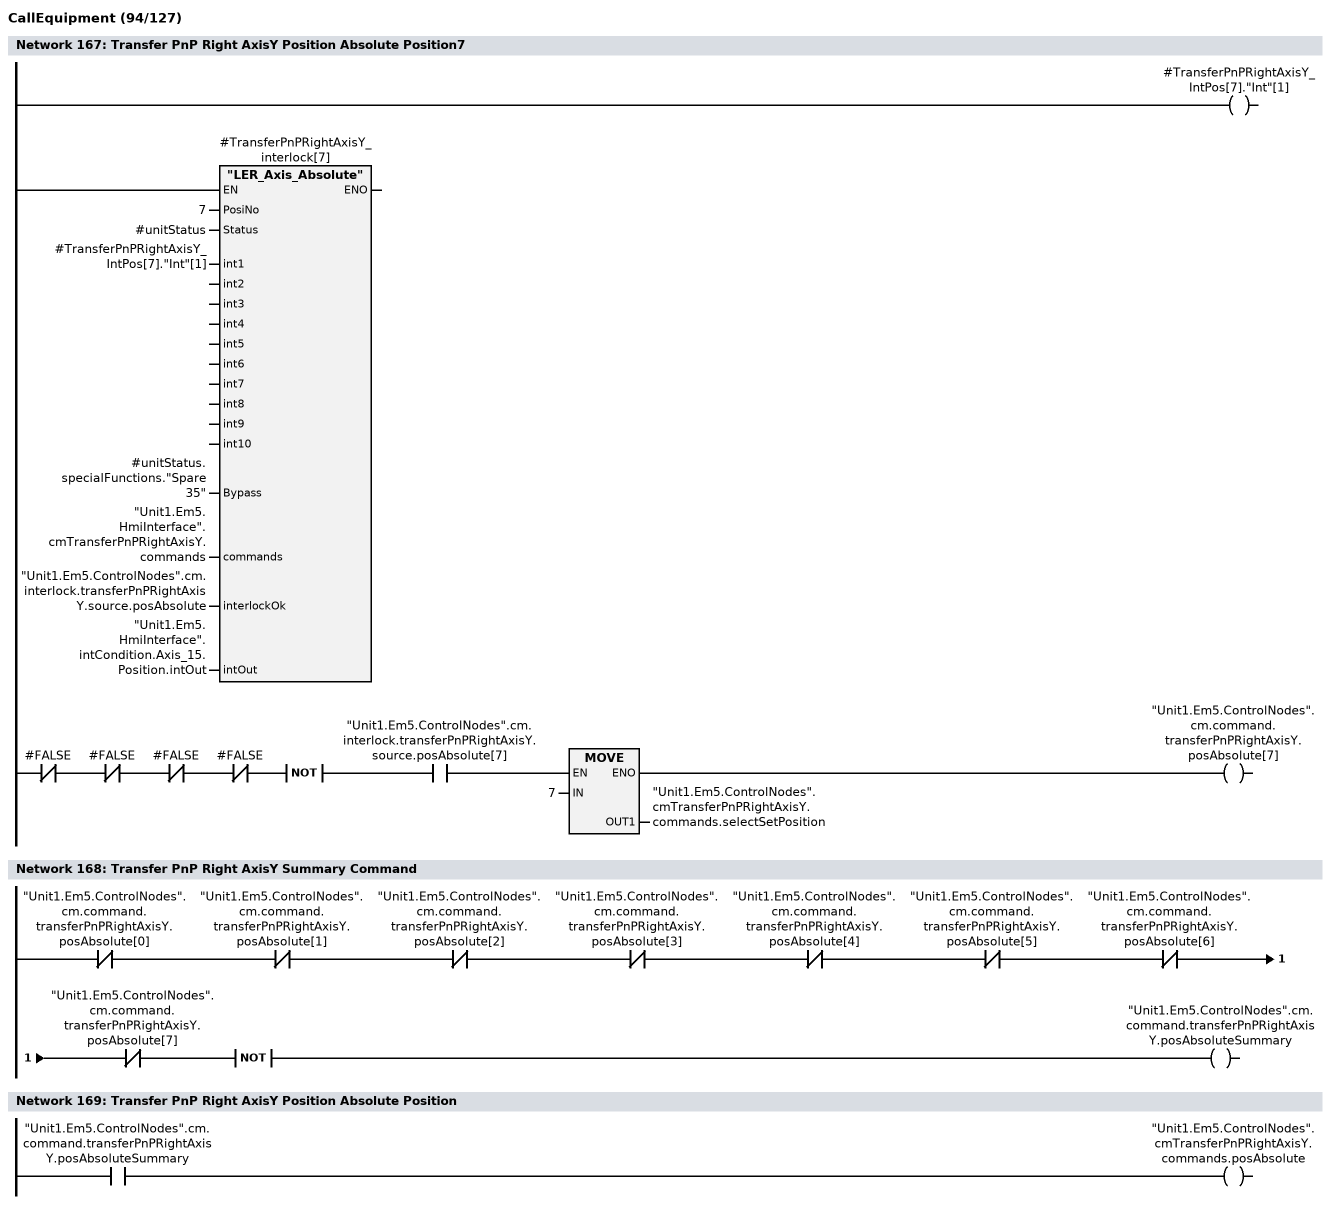
   RUNG wire#powerrail
      Coil( #TransferPnPRightAxisY_IntPos[7]."Int"[1] )
   END_RUNG
   RUNG wire#powerrail
      #TransferPnPRightAxisY_interlock[7](PosiNo := 7, Status := #unitStatus, int1 := #TransferPnPRightAxisY_IntPos[7]."Int"[1], int2 :=, int3 :=, int4 :=, int5 :=, int6 :=, int7 :=, int8 :=, int9 :=, int10 :=, Bypass := #unitStatus.specialFunctions."Spare 35", commands := "Unit1.Em5.HmiInterface".cmTransferPnPRightAxisY.commands, interlockOk := "Unit1.Em5.ControlNodes".cm.interlock.transferPnPRightAxisY.source.posAbsolute, intOut := "Unit1.Em5.HmiInterface".intCondition.Axis_15.Position.intOut)
   END_RUNG
   RUNG wire#powerrail
      I_Contact( #FALSE )
      I_Contact( #FALSE )
      I_Contact( #FALSE )
      I_Contact( #FALSE )
      Not()
      Contact( "Unit1.Em5.ControlNodes".cm.interlock.transferPnPRightAxisY.source.posAbsolute[7] )
      Move(in := 7, out1 => "Unit1.Em5.ControlNodes".cmTransferPnPRightAxisY.commands.selectSetPosition)
      Coil( "Unit1.Em5.ControlNodes".cm.command.transferPnPRightAxisY.posAbsolute[7] )
   END_RUNG
   // the same network as SCL:
   #TransferPnPRightAxisY_IntPos[7]."Int"[1] := TRUE;
   #TransferPnPRightAxisY_interlock[7](PosiNo := 7,   // "LER_Axis_Absolute"
                           Status := #unitStatus,
                           int1 := #TransferPnPRightAxisY_IntPos[7]."Int"[1],
                           Bypass := #unitStatus.specialFunctions."Spare 35",
                           commands := "Unit1.Em5.HmiInterface".cmTransferPnPRightAxisY.commands,
                           interlockOk := "Unit1.Em5.ControlNodes".cm.interlock.transferPnPRightAxisY.source.posAbsolute,
                           intOut := "Unit1.Em5.HmiInterface".intCondition.Axis_15.Position.intOut);
   #_w1 := NOT (NOT #FALSE AND NOT #FALSE AND NOT #FALSE AND NOT #FALSE) AND "Unit1.Em5.ControlNodes".cm.interlock.transferPnPRightAxisY.source.posAbsolute[7];
   IF #_w1 THEN "Unit1.Em5.ControlNodes".cmTransferPnPRightAxisY.commands.selectSetPosition := 7; END_IF;
   "Unit1.Em5.ControlNodes".cm.command.transferPnPRightAxisY.posAbsolute[7] := #_w1;
END_REGION

REGION Network 168: Transfer PnP Right AxisY Summary Command
   RUNG wire#powerrail
      I_Contact( "Unit1.Em5.ControlNodes".cm.command.transferPnPRightAxisY.posAbsolute[0] )
      I_Contact( "Unit1.Em5.ControlNodes".cm.command.transferPnPRightAxisY.posAbsolute[1] )
      I_Contact( "Unit1.Em5.ControlNodes".cm.command.transferPnPRightAxisY.posAbsolute[2] )
      I_Contact( "Unit1.Em5.ControlNodes".cm.command.transferPnPRightAxisY.posAbsolute[3] )
      I_Contact( "Unit1.Em5.ControlNodes".cm.command.transferPnPRightAxisY.posAbsolute[4] )
      I_Contact( "Unit1.Em5.ControlNodes".cm.command.transferPnPRightAxisY.posAbsolute[5] )
      I_Contact( "Unit1.Em5.ControlNodes".cm.command.transferPnPRightAxisY.posAbsolute[6] )
      I_Contact( "Unit1.Em5.ControlNodes".cm.command.transferPnPRightAxisY.posAbsolute[7] )
      Not()
      Coil( "Unit1.Em5.ControlNodes".cm.command.transferPnPRightAxisY.posAbsoluteSummary )
   END_RUNG
   // the same network as SCL:
   "Unit1.Em5.ControlNodes".cm.command.transferPnPRightAxisY.posAbsoluteSummary := NOT (NOT "Unit1.Em5.ControlNodes".cm.command.transferPnPRightAxisY.posAbsolute[0] AND NOT "Unit1.Em5.ControlNodes".cm.command.transferPnPRightAxisY.posAbsolute[1] AND NOT "Unit1.Em5.ControlNodes".cm.command.transferPnPRightAxisY.posAbsolute[2] AND NOT "Unit1.Em5.ControlNodes".cm.command.transferPnPRightAxisY.posAbsolute[3] AND NOT "Unit1.Em5.ControlNodes".cm.command.transferPnPRightAxisY.posAbsolute[4] AND NOT "Unit1.Em5.ControlNodes".cm.command.transferPnPRightAxisY.posAbsolute[5] AND NOT "Unit1.Em5.ControlNodes".cm.command.transferPnPRightAxisY.posAbsolute[6] AND NOT "Unit1.Em5.ControlNodes".cm.command.transferPnPRightAxisY.posAbsolute[7]);
END_REGION

REGION Network 169: Transfer PnP Right AxisY Position Absolute Position
   RUNG wire#powerrail
      Contact( "Unit1.Em5.ControlNodes".cm.command.transferPnPRightAxisY.posAbsoluteSummary )
      Coil( "Unit1.Em5.ControlNodes".cmTransferPnPRightAxisY.commands.posAbsolute )
   END_RUNG
   // the same network as SCL:
   "Unit1.Em5.ControlNodes".cmTransferPnPRightAxisY.commands.posAbsolute := "Unit1.Em5.ControlNodes".cm.command.transferPnPRightAxisY.posAbsoluteSummary;
END_REGION

REGION Network 170: Transfer PnP Right AxisY Interlock Summary
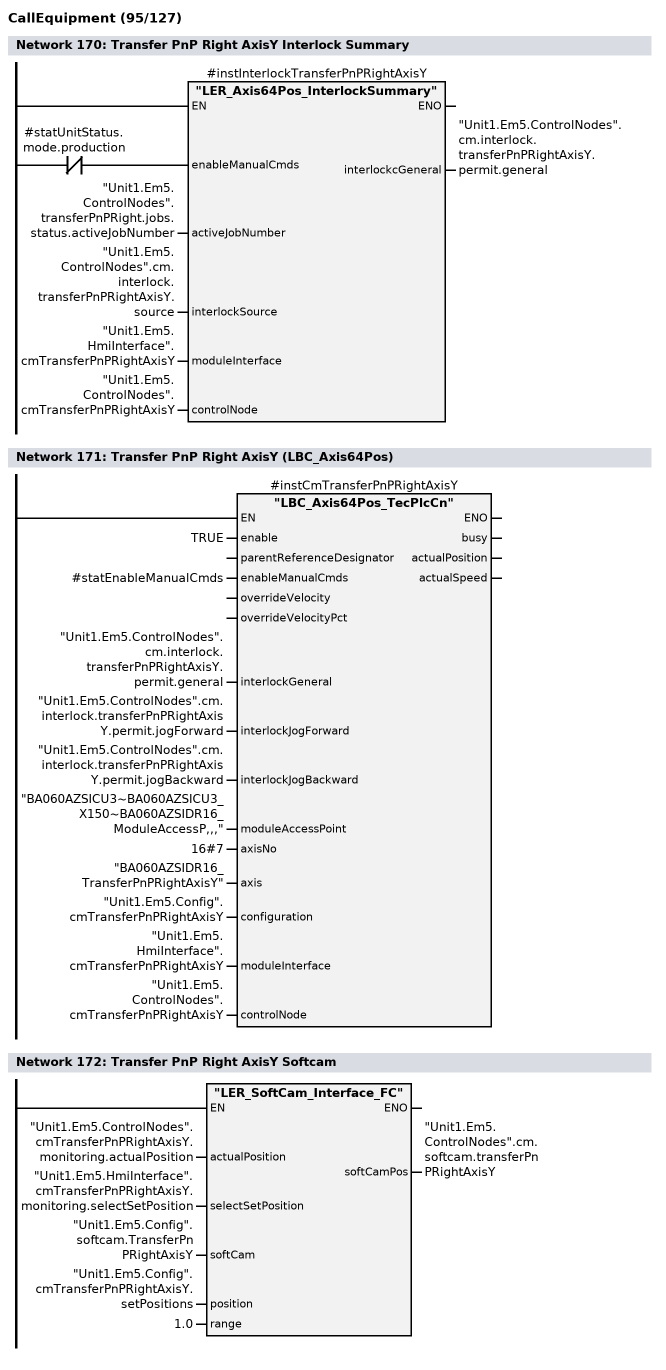
   RUNG wire#powerrail
      #instInterlockTransferPnPRightAxisY(enableManualCmds := wire#w1, activeJobNumber := "Unit1.Em5.ControlNodes".transferPnPRight.jobs.status.activeJobNumber, interlockSource := "Unit1.Em5.ControlNodes".cm.interlock.transferPnPRightAxisY.source, moduleInterface := "Unit1.Em5.HmiInterface".cmTransferPnPRightAxisY, controlNode := "Unit1.Em5.ControlNodes".cmTransferPnPRightAxisY, interlockcGeneral => "Unit1.Em5.ControlNodes".cm.interlock.transferPnPRightAxisY.permit.general)
   END_RUNG
   RUNG wire#powerrail
      I_Contact( #statUnitStatus.mode.production )
   END_RUNG wire#w1
   // the same network as SCL:
   #instInterlockTransferPnPRightAxisY(enableManualCmds := NOT #statUnitStatus.mode.production,   // "LER_Axis64Pos_InterlockSummary"
                           activeJobNumber := "Unit1.Em5.ControlNodes".transferPnPRight.jobs.status.activeJobNumber,
                           interlockSource := "Unit1.Em5.ControlNodes".cm.interlock.transferPnPRightAxisY.source,
                           moduleInterface := "Unit1.Em5.HmiInterface".cmTransferPnPRightAxisY,
                           controlNode := "Unit1.Em5.ControlNodes".cmTransferPnPRightAxisY,
                           interlockcGeneral => "Unit1.Em5.ControlNodes".cm.interlock.transferPnPRightAxisY.permit.general);
END_REGION

REGION Network 171: Transfer PnP Right AxisY (LBC_Axis64Pos)
   RUNG wire#powerrail
      #instCmTransferPnPRightAxisY(enable := TRUE, parentReferenceDesignator :=, enableManualCmds := #statEnableManualCmds, overrideVelocity :=, overrideVelocityPct :=, interlockGeneral := "Unit1.Em5.ControlNodes".cm.interlock.transferPnPRightAxisY.permit.general, interlockJogForward := "Unit1.Em5.ControlNodes".cm.interlock.transferPnPRightAxisY.permit.jogForward, interlockJogBackward := "Unit1.Em5.ControlNodes".cm.interlock.transferPnPRightAxisY.permit.jogBackward, moduleAccessPoint := "BA060AZSICU3~BA060AZSICU3_X150~BA060AZSIDR16_ModuleAccessP,,,", axisNo := 16#7, axis := "BA060AZSIDR16_TransferPnPRightAxisY", configuration := "Unit1.Em5.Config".cmTransferPnPRightAxisY, moduleInterface := "Unit1.Em5.HmiInterface".cmTransferPnPRightAxisY, controlNode := "Unit1.Em5.ControlNodes".cmTransferPnPRightAxisY, busy =>, actualPosition =>, actualSpeed =>)
   END_RUNG
   // the same network as SCL:
   #instCmTransferPnPRightAxisY(enable := TRUE,   // "LBC_Axis64Pos_TecPlcCn"
                           enableManualCmds := #statEnableManualCmds,
                           interlockGeneral := "Unit1.Em5.ControlNodes".cm.interlock.transferPnPRightAxisY.permit.general,
                           interlockJogForward := "Unit1.Em5.ControlNodes".cm.interlock.transferPnPRightAxisY.permit.jogForward,
                           interlockJogBackward := "Unit1.Em5.ControlNodes".cm.interlock.transferPnPRightAxisY.permit.jogBackward,
                           moduleAccessPoint := "BA060AZSICU3~BA060AZSICU3_X150~BA060AZSIDR16_ModuleAccessP,,,",
                           axisNo := 16#7,
                           axis := "BA060AZSIDR16_TransferPnPRightAxisY",
                           configuration := "Unit1.Em5.Config".cmTransferPnPRightAxisY,
                           moduleInterface := "Unit1.Em5.HmiInterface".cmTransferPnPRightAxisY,
                           controlNode := "Unit1.Em5.ControlNodes".cmTransferPnPRightAxisY);
END_REGION

REGION Network 172: Transfer PnP Right AxisY Softcam
   RUNG wire#powerrail
      "LER_SoftCam_Interface_FC"(actualPosition := "Unit1.Em5.ControlNodes".cmTransferPnPRightAxisY.monitoring.actualPosition, selectSetPosition := "Unit1.Em5.HmiInterface".cmTransferPnPRightAxisY.monitoring.selectSetPosition, softCam := "Unit1.Em5.Config".softcam.TransferPnPRightAxisY, position := "Unit1.Em5.Config".cmTransferPnPRightAxisY.setPositions, range := 1.0, softCamPos => "Unit1.Em5.ControlNodes".cm.softcam.transferPnPRightAxisY)
   END_RUNG
   // the same network as SCL:
   "LER_SoftCam_Interface_FC"(actualPosition := "Unit1.Em5.ControlNodes".cmTransferPnPRightAxisY.monitoring.actualPosition,
                           selectSetPosition := "Unit1.Em5.HmiInterface".cmTransferPnPRightAxisY.monitoring.selectSetPosition,
                           softCam := "Unit1.Em5.Config".softcam.TransferPnPRightAxisY,
                           position := "Unit1.Em5.Config".cmTransferPnPRightAxisY.setPositions,
                           range := 1.0,
                           softCamPos => "Unit1.Em5.ControlNodes".cm.softcam.transferPnPRightAxisY);
END_REGION

REGION Network 174: Transfer P&P Right Z-Axis Upload Actual Current And Torque Values
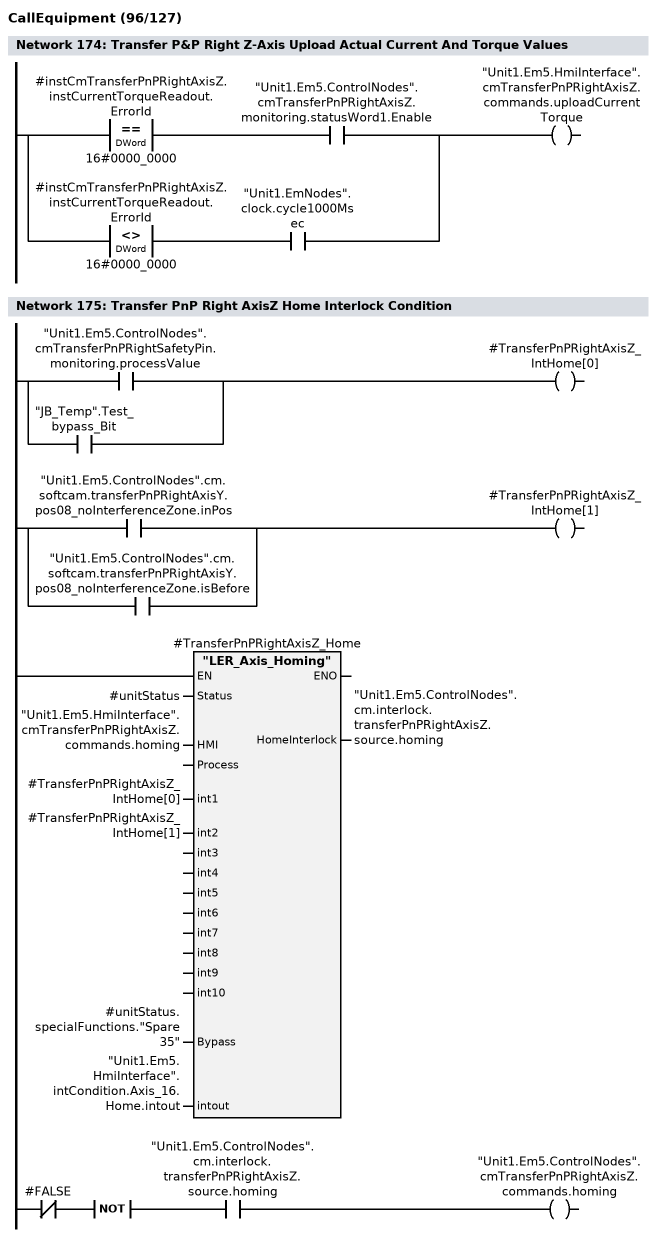
   RUNG wire#powerrail
      { S7_Templates := "SrcType := DWord" } EQ_Contact(in1 := #instCmTransferPnPRightAxisZ.instCurrentTorqueReadout.ErrorId, in2 := 16#0000_0000)
      Contact( "Unit1.Em5.ControlNodes".cmTransferPnPRightAxisZ.monitoring.statusWord1.Enable )
      wire#w1
      Coil( "Unit1.Em5.HmiInterface".cmTransferPnPRightAxisZ.commands.uploadCurrentTorque )
   END_RUNG
   RUNG wire#powerrail
      { S7_Templates := "SrcType := DWord" } NE_Contact(in1 := #instCmTransferPnPRightAxisZ.instCurrentTorqueReadout.ErrorId, in2 := 16#0000_0000)
      Contact( "Unit1.EmNodes".clock.cycle1000Msec )
   END_RUNG wire#w1
   // the same network as SCL:
   "Unit1.Em5.HmiInterface".cmTransferPnPRightAxisZ.commands.uploadCurrentTorque := ((#instCmTransferPnPRightAxisZ.instCurrentTorqueReadout.ErrorId = 16#0000_0000) AND "Unit1.Em5.ControlNodes".cmTransferPnPRightAxisZ.monitoring.statusWord1.Enable) OR ((#instCmTransferPnPRightAxisZ.instCurrentTorqueReadout.ErrorId <> 16#0000_0000) AND "Unit1.EmNodes".clock.cycle1000Msec);
END_REGION

REGION Network 175: Transfer PnP Right AxisZ Home Interlock Condition
   RUNG wire#powerrail
      Contact( "Unit1.Em5.ControlNodes".cmTransferPnPRightSafetyPin.monitoring.processValue )
      wire#w1
      Coil( #TransferPnPRightAxisZ_IntHome[0] )
   END_RUNG
   RUNG wire#powerrail
      Contact( "JB_Temp".Test_bypass_Bit )
   END_RUNG wire#w1
   RUNG wire#powerrail
      Contact( "Unit1.Em5.ControlNodes".cm.softcam.transferPnPRightAxisY.pos08_noInterferenceZone.inPos )
      wire#w2
      Coil( #TransferPnPRightAxisZ_IntHome[1] )
   END_RUNG
   RUNG wire#powerrail
      Contact( "Unit1.Em5.ControlNodes".cm.softcam.transferPnPRightAxisY.pos08_noInterferenceZone.isBefore )
   END_RUNG wire#w2
   RUNG wire#powerrail
      #TransferPnPRightAxisZ_Home(Status := #unitStatus, HMI := "Unit1.Em5.HmiInterface".cmTransferPnPRightAxisZ.commands.homing, Process :=, int1 := #TransferPnPRightAxisZ_IntHome[0], int2 := #TransferPnPRightAxisZ_IntHome[1], int3 :=, int4 :=, int5 :=, int6 :=, int7 :=, int8 :=, int9 :=, int10 :=, Bypass := #unitStatus.specialFunctions."Spare 35", intout := "Unit1.Em5.HmiInterface".intCondition.Axis_16.Home.intout, HomeInterlock => "Unit1.Em5.ControlNodes".cm.interlock.transferPnPRightAxisZ.source.homing)
   END_RUNG
   RUNG wire#powerrail
      I_Contact( #FALSE )
      Not()
      Contact( "Unit1.Em5.ControlNodes".cm.interlock.transferPnPRightAxisZ.source.homing )
      Coil( "Unit1.Em5.ControlNodes".cmTransferPnPRightAxisZ.commands.homing )
   END_RUNG
   // the same network as SCL:
   #TransferPnPRightAxisZ_IntHome[0] := "Unit1.Em5.ControlNodes".cmTransferPnPRightSafetyPin.monitoring.processValue OR "JB_Temp".Test_bypass_Bit;
   #TransferPnPRightAxisZ_IntHome[1] := "Unit1.Em5.ControlNodes".cm.softcam.transferPnPRightAxisY.pos08_noInterferenceZone.inPos OR "Unit1.Em5.ControlNodes".cm.softcam.transferPnPRightAxisY.pos08_noInterferenceZone.isBefore;
   #TransferPnPRightAxisZ_Home(Status := #unitStatus,   // "LER_Axis_Homing"
                           HMI := "Unit1.Em5.HmiInterface".cmTransferPnPRightAxisZ.commands.homing,
                           int1 := #TransferPnPRightAxisZ_IntHome[0],
                           int2 := #TransferPnPRightAxisZ_IntHome[1],
                           Bypass := #unitStatus.specialFunctions."Spare 35",
                           intout := "Unit1.Em5.HmiInterface".intCondition.Axis_16.Home.intout,
                           HomeInterlock => "Unit1.Em5.ControlNodes".cm.interlock.transferPnPRightAxisZ.source.homing);
   "Unit1.Em5.ControlNodes".cmTransferPnPRightAxisZ.commands.homing := NOT (NOT #FALSE) AND "Unit1.Em5.ControlNodes".cm.interlock.transferPnPRightAxisZ.source.homing;
END_REGION

REGION Network 176: Transfer PnP Right AxisZ JOG Interlock Condition
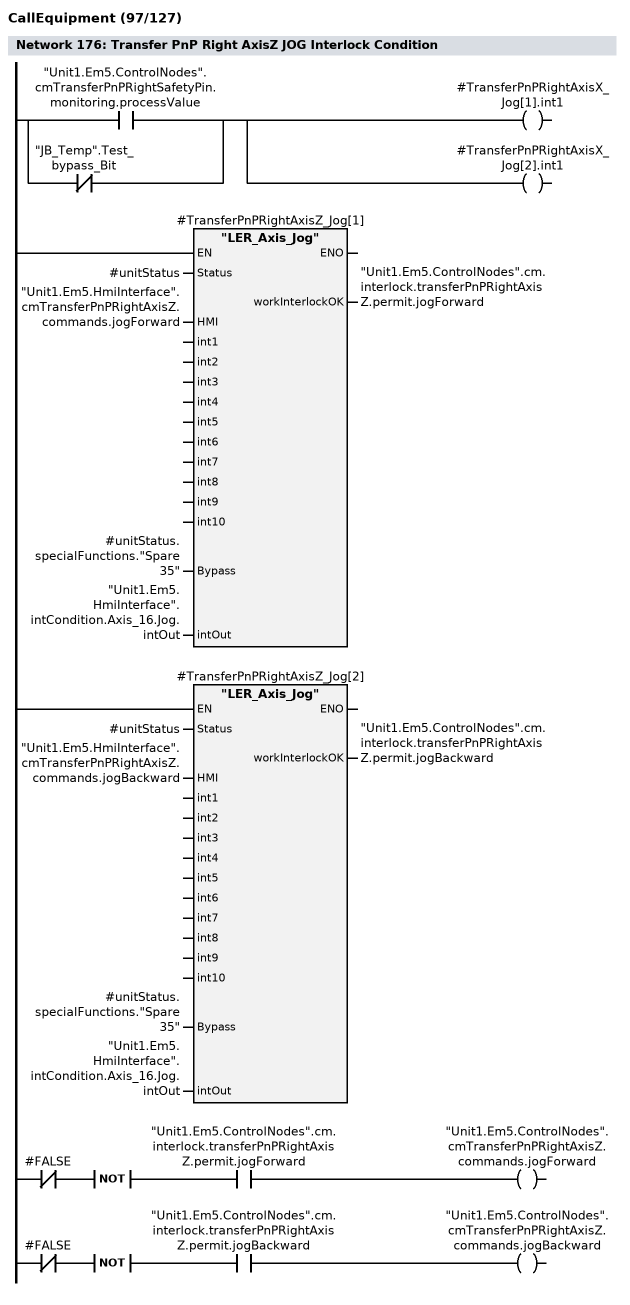
   RUNG wire#powerrail
      Contact( "Unit1.Em5.ControlNodes".cmTransferPnPRightSafetyPin.monitoring.processValue )
      wire#w1
      Coil( #TransferPnPRightAxisX_Jog[1].int1 )
   END_RUNG
   RUNG wire#powerrail
      I_Contact( "JB_Temp".Test_bypass_Bit )
   END_RUNG wire#w1
   RUNG wire#w1
      Coil( #TransferPnPRightAxisX_Jog[2].int1 )
   END_RUNG
   RUNG wire#powerrail
      #TransferPnPRightAxisZ_Jog[1](Status := #unitStatus, HMI := "Unit1.Em5.HmiInterface".cmTransferPnPRightAxisZ.commands.jogForward, int1 :=, int2 :=, int3 :=, int4 :=, int5 :=, int6 :=, int7 :=, int8 :=, int9 :=, int10 :=, Bypass := #unitStatus.specialFunctions."Spare 35", intOut := "Unit1.Em5.HmiInterface".intCondition.Axis_16.Jog.intOut, workInterlockOK => "Unit1.Em5.ControlNodes".cm.interlock.transferPnPRightAxisZ.permit.jogForward)
   END_RUNG
   RUNG wire#powerrail
      #TransferPnPRightAxisZ_Jog[2](Status := #unitStatus, HMI := "Unit1.Em5.HmiInterface".cmTransferPnPRightAxisZ.commands.jogBackward, int1 :=, int2 :=, int3 :=, int4 :=, int5 :=, int6 :=, int7 :=, int8 :=, int9 :=, int10 :=, Bypass := #unitStatus.specialFunctions."Spare 35", intOut := "Unit1.Em5.HmiInterface".intCondition.Axis_16.Jog.intOut, workInterlockOK => "Unit1.Em5.ControlNodes".cm.interlock.transferPnPRightAxisZ.permit.jogBackward)
   END_RUNG
   RUNG wire#powerrail
      I_Contact( #FALSE )
      Not()
      Contact( "Unit1.Em5.ControlNodes".cm.interlock.transferPnPRightAxisZ.permit.jogForward )
      Coil( "Unit1.Em5.ControlNodes".cmTransferPnPRightAxisZ.commands.jogForward )
   END_RUNG
   RUNG wire#powerrail
      I_Contact( #FALSE )
      Not()
      Contact( "Unit1.Em5.ControlNodes".cm.interlock.transferPnPRightAxisZ.permit.jogBackward )
      Coil( "Unit1.Em5.ControlNodes".cmTransferPnPRightAxisZ.commands.jogBackward )
   END_RUNG
   // the same network as SCL:
   #TransferPnPRightAxisX_Jog[1].int1 := "Unit1.Em5.ControlNodes".cmTransferPnPRightSafetyPin.monitoring.processValue OR NOT "JB_Temp".Test_bypass_Bit;
   #TransferPnPRightAxisX_Jog[2].int1 := "Unit1.Em5.ControlNodes".cmTransferPnPRightSafetyPin.monitoring.processValue OR NOT "JB_Temp".Test_bypass_Bit;
   #TransferPnPRightAxisZ_Jog[1](Status := #unitStatus,   // "LER_Axis_Jog"
                           HMI := "Unit1.Em5.HmiInterface".cmTransferPnPRightAxisZ.commands.jogForward,
                           Bypass := #unitStatus.specialFunctions."Spare 35",
                           intOut := "Unit1.Em5.HmiInterface".intCondition.Axis_16.Jog.intOut,
                           workInterlockOK => "Unit1.Em5.ControlNodes".cm.interlock.transferPnPRightAxisZ.permit.jogForward);
   #TransferPnPRightAxisZ_Jog[2](Status := #unitStatus,   // "LER_Axis_Jog"
                           HMI := "Unit1.Em5.HmiInterface".cmTransferPnPRightAxisZ.commands.jogBackward,
                           Bypass := #unitStatus.specialFunctions."Spare 35",
                           intOut := "Unit1.Em5.HmiInterface".intCondition.Axis_16.Jog.intOut,
                           workInterlockOK => "Unit1.Em5.ControlNodes".cm.interlock.transferPnPRightAxisZ.permit.jogBackward);
   "Unit1.Em5.ControlNodes".cmTransferPnPRightAxisZ.commands.jogForward := NOT (NOT #FALSE) AND "Unit1.Em5.ControlNodes".cm.interlock.transferPnPRightAxisZ.permit.jogForward;
   "Unit1.Em5.ControlNodes".cmTransferPnPRightAxisZ.commands.jogBackward := NOT (NOT #FALSE) AND "Unit1.Em5.ControlNodes".cm.interlock.transferPnPRightAxisZ.permit.jogBackward;
END_REGION

REGION Network 177: Transfer PnP Right AxisZ Position Absolute Position0
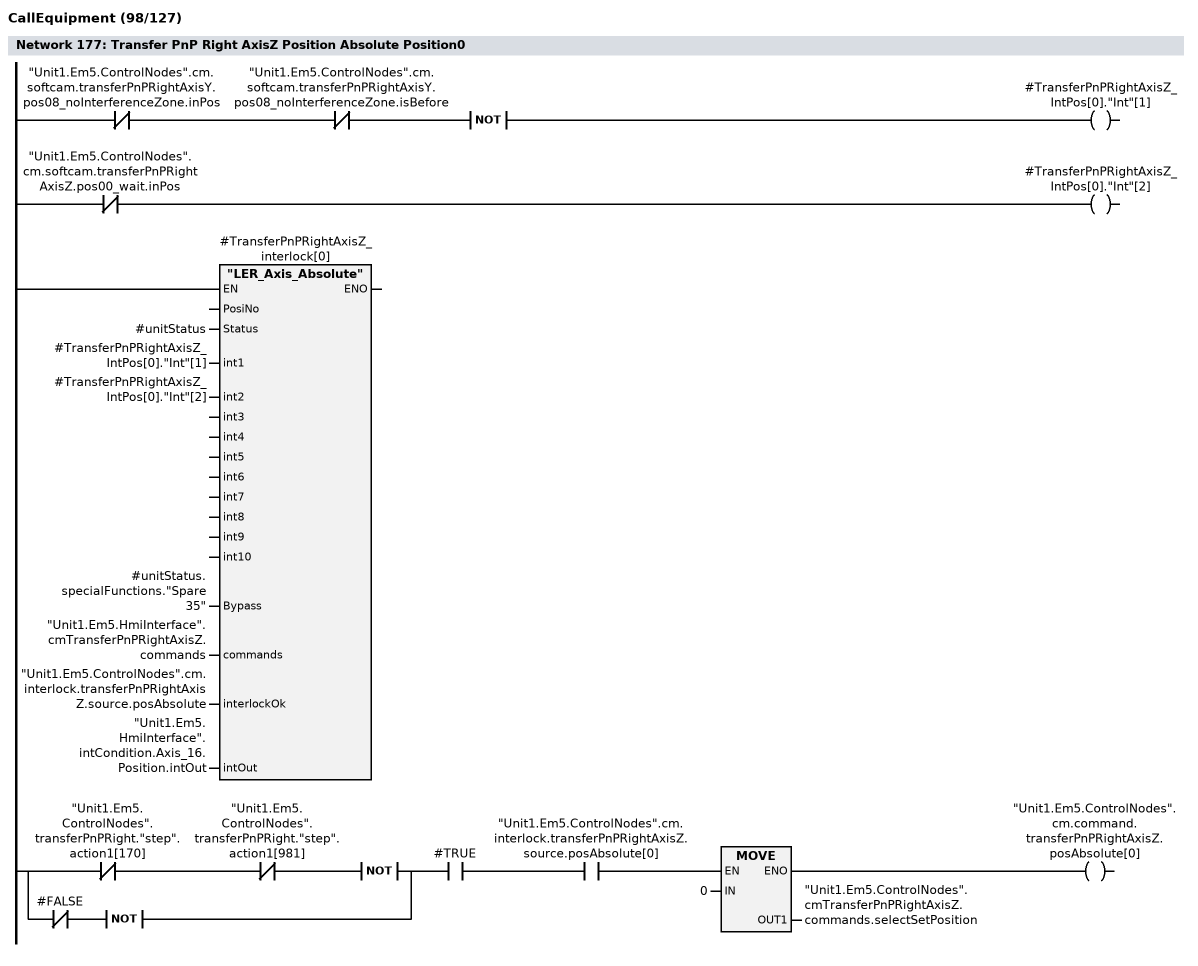
   RUNG wire#powerrail
      I_Contact( "Unit1.Em5.ControlNodes".cm.softcam.transferPnPRightAxisY.pos08_noInterferenceZone.inPos )
      I_Contact( "Unit1.Em5.ControlNodes".cm.softcam.transferPnPRightAxisY.pos08_noInterferenceZone.isBefore )
      Not()
      Coil( #TransferPnPRightAxisZ_IntPos[0]."Int"[1] )
   END_RUNG
   RUNG wire#powerrail
      I_Contact( "Unit1.Em5.ControlNodes".cm.softcam.transferPnPRightAxisZ.pos00_wait.inPos )
      Coil( #TransferPnPRightAxisZ_IntPos[0]."Int"[2] )
   END_RUNG
   RUNG wire#powerrail
      #TransferPnPRightAxisZ_interlock[0](PosiNo :=, Status := #unitStatus, int1 := #TransferPnPRightAxisZ_IntPos[0]."Int"[1], int2 := #TransferPnPRightAxisZ_IntPos[0]."Int"[2], int3 :=, int4 :=, int5 :=, int6 :=, int7 :=, int8 :=, int9 :=, int10 :=, Bypass := #unitStatus.specialFunctions."Spare 35", commands := "Unit1.Em5.HmiInterface".cmTransferPnPRightAxisZ.commands, interlockOk := "Unit1.Em5.ControlNodes".cm.interlock.transferPnPRightAxisZ.source.posAbsolute, intOut := "Unit1.Em5.HmiInterface".intCondition.Axis_16.Position.intOut)
   END_RUNG
   RUNG wire#powerrail
      I_Contact( "Unit1.Em5.ControlNodes".transferPnPRight."step".action1[170] )
      I_Contact( "Unit1.Em5.ControlNodes".transferPnPRight."step".action1[981] )
      Not()
      wire#w1
      Contact( #TRUE )
      Contact( "Unit1.Em5.ControlNodes".cm.interlock.transferPnPRightAxisZ.source.posAbsolute[0] )
      Move(in := 0, out1 => "Unit1.Em5.ControlNodes".cmTransferPnPRightAxisZ.commands.selectSetPosition)
      Coil( "Unit1.Em5.ControlNodes".cm.command.transferPnPRightAxisZ.posAbsolute[0] )
   END_RUNG
   RUNG wire#powerrail
      I_Contact( #FALSE )
      Not()
   END_RUNG wire#w1
   // the same network as SCL:
   #TransferPnPRightAxisZ_IntPos[0]."Int"[1] := NOT (NOT "Unit1.Em5.ControlNodes".cm.softcam.transferPnPRightAxisY.pos08_noInterferenceZone.inPos AND NOT "Unit1.Em5.ControlNodes".cm.softcam.transferPnPRightAxisY.pos08_noInterferenceZone.isBefore);
   #TransferPnPRightAxisZ_IntPos[0]."Int"[2] := NOT "Unit1.Em5.ControlNodes".cm.softcam.transferPnPRightAxisZ.pos00_wait.inPos;
   #TransferPnPRightAxisZ_interlock[0](Status := #unitStatus,   // "LER_Axis_Absolute"
                           int1 := #TransferPnPRightAxisZ_IntPos[0]."Int"[1],
                           int2 := #TransferPnPRightAxisZ_IntPos[0]."Int"[2],
                           Bypass := #unitStatus.specialFunctions."Spare 35",
                           commands := "Unit1.Em5.HmiInterface".cmTransferPnPRightAxisZ.commands,
                           interlockOk := "Unit1.Em5.ControlNodes".cm.interlock.transferPnPRightAxisZ.source.posAbsolute,
                           intOut := "Unit1.Em5.HmiInterface".intCondition.Axis_16.Position.intOut);
   #_w1 := (NOT (NOT "Unit1.Em5.ControlNodes".transferPnPRight."step".action1[170] AND NOT "Unit1.Em5.ControlNodes".transferPnPRight."step".action1[981]) OR NOT (NOT #FALSE)) AND #TRUE AND "Unit1.Em5.ControlNodes".cm.interlock.transferPnPRightAxisZ.source.posAbsolute[0];
   IF #_w1 THEN "Unit1.Em5.ControlNodes".cmTransferPnPRightAxisZ.commands.selectSetPosition := 0; END_IF;
   "Unit1.Em5.ControlNodes".cm.command.transferPnPRightAxisZ.posAbsolute[0] := #_w1;
END_REGION

REGION Network 178: Transfer PnP Right AxisZ Position Absolute Position1
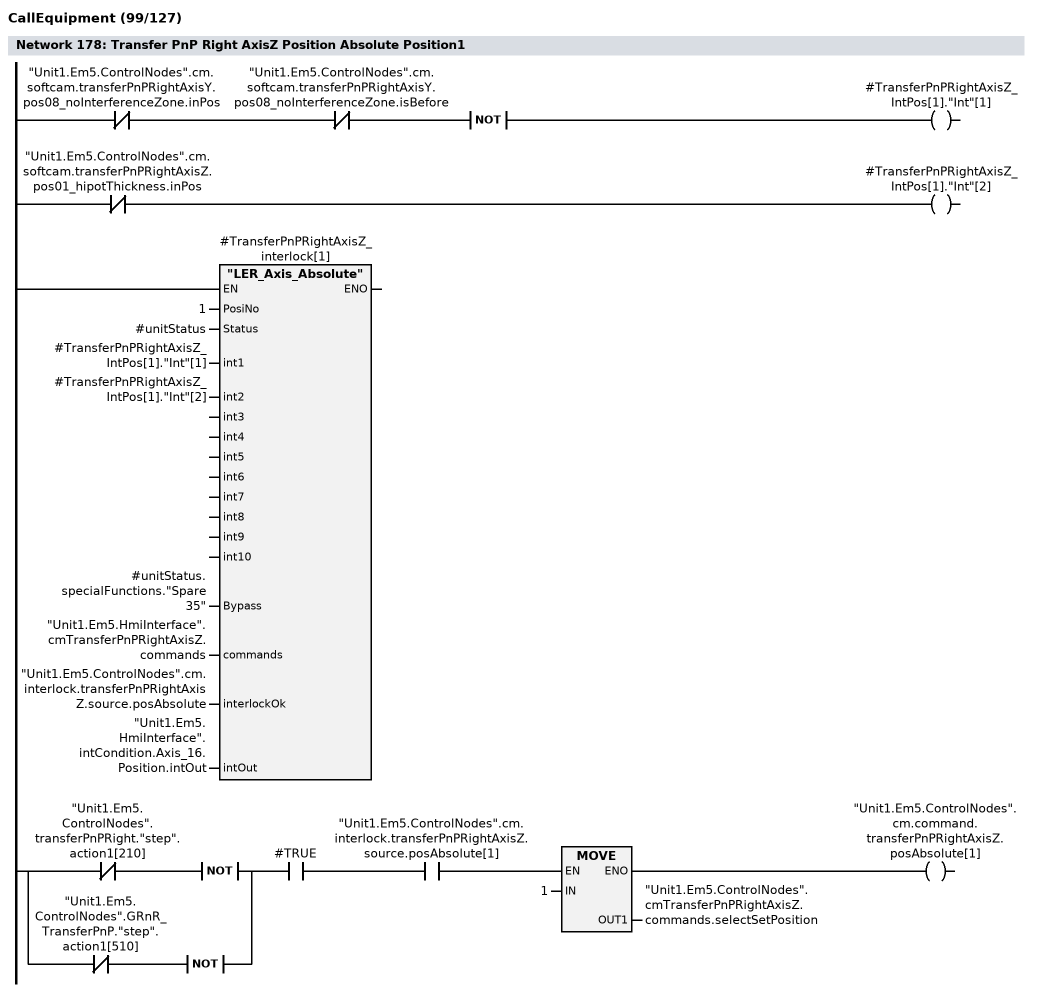
   RUNG wire#powerrail
      I_Contact( "Unit1.Em5.ControlNodes".cm.softcam.transferPnPRightAxisY.pos08_noInterferenceZone.inPos )
      I_Contact( "Unit1.Em5.ControlNodes".cm.softcam.transferPnPRightAxisY.pos08_noInterferenceZone.isBefore )
      Not()
      Coil( #TransferPnPRightAxisZ_IntPos[1]."Int"[1] )
   END_RUNG
   RUNG wire#powerrail
      I_Contact( "Unit1.Em5.ControlNodes".cm.softcam.transferPnPRightAxisZ.pos01_hipotThickness.inPos )
      Coil( #TransferPnPRightAxisZ_IntPos[1]."Int"[2] )
   END_RUNG
   RUNG wire#powerrail
      #TransferPnPRightAxisZ_interlock[1](PosiNo := 1, Status := #unitStatus, int1 := #TransferPnPRightAxisZ_IntPos[1]."Int"[1], int2 := #TransferPnPRightAxisZ_IntPos[1]."Int"[2], int3 :=, int4 :=, int5 :=, int6 :=, int7 :=, int8 :=, int9 :=, int10 :=, Bypass := #unitStatus.specialFunctions."Spare 35", commands := "Unit1.Em5.HmiInterface".cmTransferPnPRightAxisZ.commands, interlockOk := "Unit1.Em5.ControlNodes".cm.interlock.transferPnPRightAxisZ.source.posAbsolute, intOut := "Unit1.Em5.HmiInterface".intCondition.Axis_16.Position.intOut)
   END_RUNG
   RUNG wire#powerrail
      I_Contact( "Unit1.Em5.ControlNodes".transferPnPRight."step".action1[210] )
      Not()
      wire#w1
      Contact( #TRUE )
      Contact( "Unit1.Em5.ControlNodes".cm.interlock.transferPnPRightAxisZ.source.posAbsolute[1] )
      Move(in := 1, out1 => "Unit1.Em5.ControlNodes".cmTransferPnPRightAxisZ.commands.selectSetPosition)
      Coil( "Unit1.Em5.ControlNodes".cm.command.transferPnPRightAxisZ.posAbsolute[1] )
   END_RUNG
   RUNG wire#powerrail
      I_Contact( "Unit1.Em5.ControlNodes".GRnR_TransferPnP."step".action1[510] )
      Not()
   END_RUNG wire#w1
   // the same network as SCL:
   #TransferPnPRightAxisZ_IntPos[1]."Int"[1] := NOT (NOT "Unit1.Em5.ControlNodes".cm.softcam.transferPnPRightAxisY.pos08_noInterferenceZone.inPos AND NOT "Unit1.Em5.ControlNodes".cm.softcam.transferPnPRightAxisY.pos08_noInterferenceZone.isBefore);
   #TransferPnPRightAxisZ_IntPos[1]."Int"[2] := NOT "Unit1.Em5.ControlNodes".cm.softcam.transferPnPRightAxisZ.pos01_hipotThickness.inPos;
   #TransferPnPRightAxisZ_interlock[1](PosiNo := 1,   // "LER_Axis_Absolute"
                           Status := #unitStatus,
                           int1 := #TransferPnPRightAxisZ_IntPos[1]."Int"[1],
                           int2 := #TransferPnPRightAxisZ_IntPos[1]."Int"[2],
                           Bypass := #unitStatus.specialFunctions."Spare 35",
                           commands := "Unit1.Em5.HmiInterface".cmTransferPnPRightAxisZ.commands,
                           interlockOk := "Unit1.Em5.ControlNodes".cm.interlock.transferPnPRightAxisZ.source.posAbsolute,
                           intOut := "Unit1.Em5.HmiInterface".intCondition.Axis_16.Position.intOut);
   #_w1 := (NOT (NOT "Unit1.Em5.ControlNodes".transferPnPRight."step".action1[210]) OR NOT (NOT "Unit1.Em5.ControlNodes".GRnR_TransferPnP."step".action1[510])) AND #TRUE AND "Unit1.Em5.ControlNodes".cm.interlock.transferPnPRightAxisZ.source.posAbsolute[1];
   IF #_w1 THEN "Unit1.Em5.ControlNodes".cmTransferPnPRightAxisZ.commands.selectSetPosition := 1; END_IF;
   "Unit1.Em5.ControlNodes".cm.command.transferPnPRightAxisZ.posAbsolute[1] := #_w1;
END_REGION

REGION Network 179: Transfer PnP Right AxisZ Position Absolute Position2
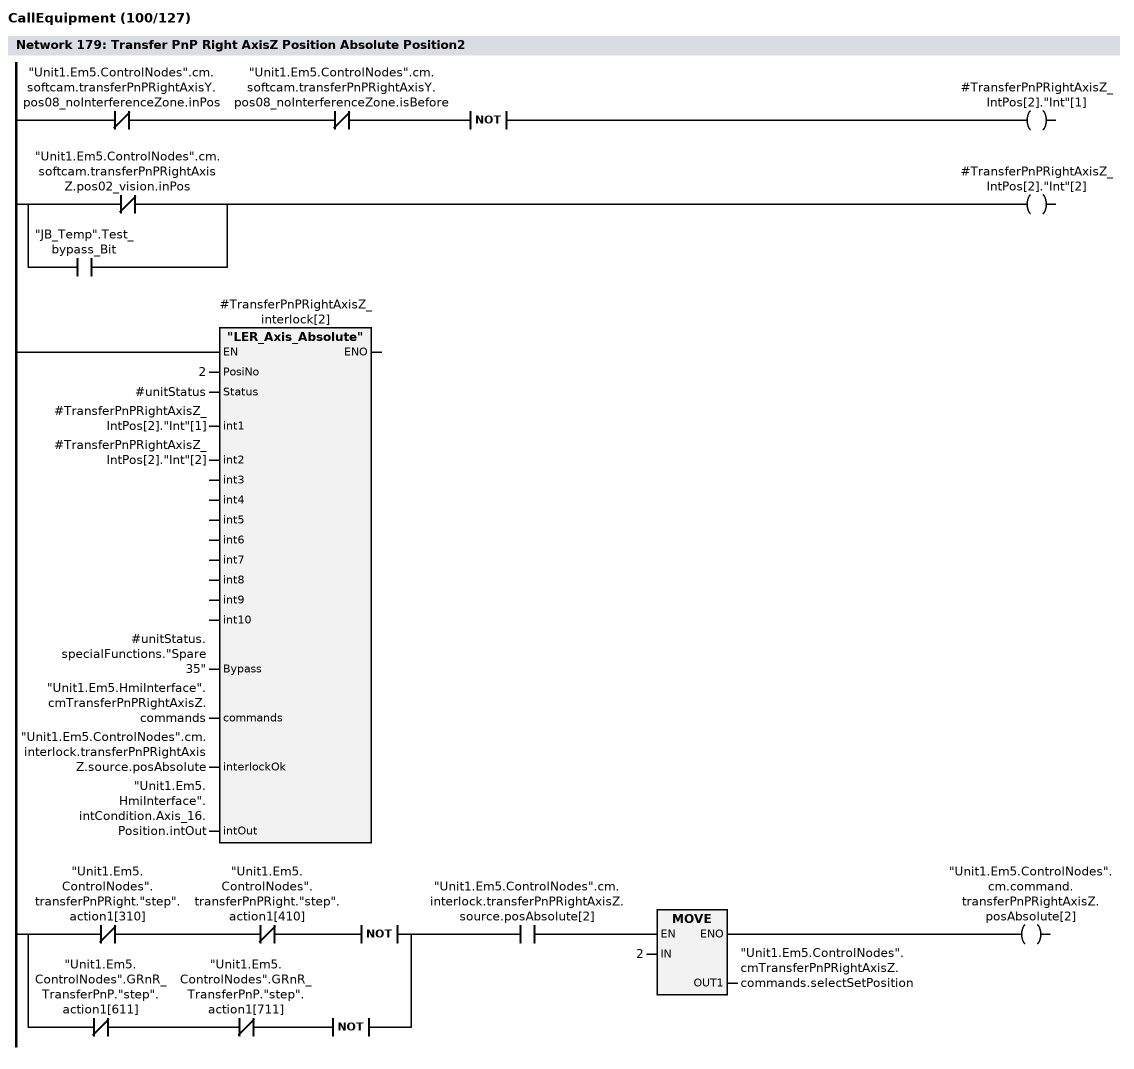
   RUNG wire#powerrail
      I_Contact( "Unit1.Em5.ControlNodes".cm.softcam.transferPnPRightAxisY.pos08_noInterferenceZone.inPos )
      I_Contact( "Unit1.Em5.ControlNodes".cm.softcam.transferPnPRightAxisY.pos08_noInterferenceZone.isBefore )
      Not()
      Coil( #TransferPnPRightAxisZ_IntPos[2]."Int"[1] )
   END_RUNG
   RUNG wire#powerrail
      I_Contact( "Unit1.Em5.ControlNodes".cm.softcam.transferPnPRightAxisZ.pos02_vision.inPos )
      wire#w1
      Coil( #TransferPnPRightAxisZ_IntPos[2]."Int"[2] )
   END_RUNG
   RUNG wire#powerrail
      Contact( "JB_Temp".Test_bypass_Bit )
   END_RUNG wire#w1
   RUNG wire#powerrail
      #TransferPnPRightAxisZ_interlock[2](PosiNo := 2, Status := #unitStatus, int1 := #TransferPnPRightAxisZ_IntPos[2]."Int"[1], int2 := #TransferPnPRightAxisZ_IntPos[2]."Int"[2], int3 :=, int4 :=, int5 :=, int6 :=, int7 :=, int8 :=, int9 :=, int10 :=, Bypass := #unitStatus.specialFunctions."Spare 35", commands := "Unit1.Em5.HmiInterface".cmTransferPnPRightAxisZ.commands, interlockOk := "Unit1.Em5.ControlNodes".cm.interlock.transferPnPRightAxisZ.source.posAbsolute, intOut := "Unit1.Em5.HmiInterface".intCondition.Axis_16.Position.intOut)
   END_RUNG
   RUNG wire#powerrail
      I_Contact( "Unit1.Em5.ControlNodes".transferPnPRight."step".action1[310] )
      I_Contact( "Unit1.Em5.ControlNodes".transferPnPRight."step".action1[410] )
      Not()
      wire#w2
      Contact( "Unit1.Em5.ControlNodes".cm.interlock.transferPnPRightAxisZ.source.posAbsolute[2] )
      Move(in := 2, out1 => "Unit1.Em5.ControlNodes".cmTransferPnPRightAxisZ.commands.selectSetPosition)
      Coil( "Unit1.Em5.ControlNodes".cm.command.transferPnPRightAxisZ.posAbsolute[2] )
   END_RUNG
   RUNG wire#powerrail
      I_Contact( "Unit1.Em5.ControlNodes".GRnR_TransferPnP."step".action1[611] )
      I_Contact( "Unit1.Em5.ControlNodes".GRnR_TransferPnP."step".action1[711] )
      Not()
   END_RUNG wire#w2
   // the same network as SCL:
   #TransferPnPRightAxisZ_IntPos[2]."Int"[1] := NOT (NOT "Unit1.Em5.ControlNodes".cm.softcam.transferPnPRightAxisY.pos08_noInterferenceZone.inPos AND NOT "Unit1.Em5.ControlNodes".cm.softcam.transferPnPRightAxisY.pos08_noInterferenceZone.isBefore);
   #TransferPnPRightAxisZ_IntPos[2]."Int"[2] := NOT "Unit1.Em5.ControlNodes".cm.softcam.transferPnPRightAxisZ.pos02_vision.inPos OR "JB_Temp".Test_bypass_Bit;
   #TransferPnPRightAxisZ_interlock[2](PosiNo := 2,   // "LER_Axis_Absolute"
                           Status := #unitStatus,
                           int1 := #TransferPnPRightAxisZ_IntPos[2]."Int"[1],
                           int2 := #TransferPnPRightAxisZ_IntPos[2]."Int"[2],
                           Bypass := #unitStatus.specialFunctions."Spare 35",
                           commands := "Unit1.Em5.HmiInterface".cmTransferPnPRightAxisZ.commands,
                           interlockOk := "Unit1.Em5.ControlNodes".cm.interlock.transferPnPRightAxisZ.source.posAbsolute,
                           intOut := "Unit1.Em5.HmiInterface".intCondition.Axis_16.Position.intOut);
   #_w1 := (NOT (NOT "Unit1.Em5.ControlNodes".transferPnPRight."step".action1[310] AND NOT "Unit1.Em5.ControlNodes".transferPnPRight."step".action1[410]) OR NOT (NOT "Unit1.Em5.ControlNodes".GRnR_TransferPnP."step".action1[611] AND NOT "Unit1.Em5.ControlNodes".GRnR_TransferPnP."step".action1[711])) AND "Unit1.Em5.ControlNodes".cm.interlock.transferPnPRightAxisZ.source.posAbsolute[2];
   IF #_w1 THEN "Unit1.Em5.ControlNodes".cmTransferPnPRightAxisZ.commands.selectSetPosition := 2; END_IF;
   "Unit1.Em5.ControlNodes".cm.command.transferPnPRightAxisZ.posAbsolute[2] := #_w1;
END_REGION

REGION Network 180: Transfer PnP Right AxisZ Position Absolute Position3
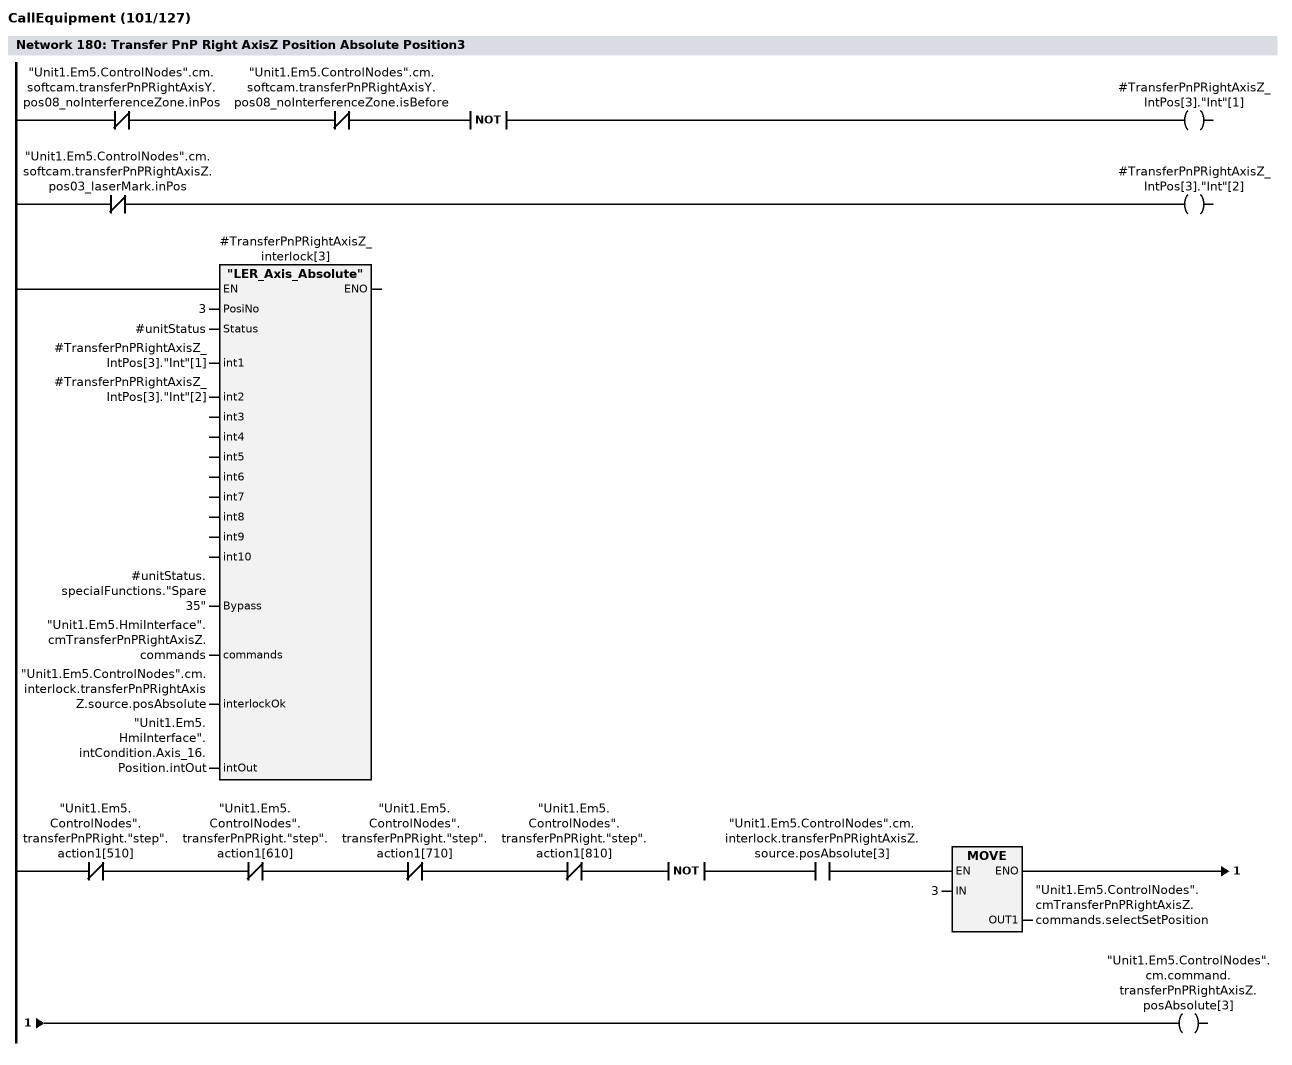
   RUNG wire#powerrail
      I_Contact( "Unit1.Em5.ControlNodes".cm.softcam.transferPnPRightAxisY.pos08_noInterferenceZone.inPos )
      I_Contact( "Unit1.Em5.ControlNodes".cm.softcam.transferPnPRightAxisY.pos08_noInterferenceZone.isBefore )
      Not()
      Coil( #TransferPnPRightAxisZ_IntPos[3]."Int"[1] )
   END_RUNG
   RUNG wire#powerrail
      I_Contact( "Unit1.Em5.ControlNodes".cm.softcam.transferPnPRightAxisZ.pos03_laserMark.inPos )
      Coil( #TransferPnPRightAxisZ_IntPos[3]."Int"[2] )
   END_RUNG
   RUNG wire#powerrail
      #TransferPnPRightAxisZ_interlock[3](PosiNo := 3, Status := #unitStatus, int1 := #TransferPnPRightAxisZ_IntPos[3]."Int"[1], int2 := #TransferPnPRightAxisZ_IntPos[3]."Int"[2], int3 :=, int4 :=, int5 :=, int6 :=, int7 :=, int8 :=, int9 :=, int10 :=, Bypass := #unitStatus.specialFunctions."Spare 35", commands := "Unit1.Em5.HmiInterface".cmTransferPnPRightAxisZ.commands, interlockOk := "Unit1.Em5.ControlNodes".cm.interlock.transferPnPRightAxisZ.source.posAbsolute, intOut := "Unit1.Em5.HmiInterface".intCondition.Axis_16.Position.intOut)
   END_RUNG
   RUNG wire#powerrail
      I_Contact( "Unit1.Em5.ControlNodes".transferPnPRight."step".action1[510] )
      I_Contact( "Unit1.Em5.ControlNodes".transferPnPRight."step".action1[610] )
      I_Contact( "Unit1.Em5.ControlNodes".transferPnPRight."step".action1[710] )
      I_Contact( "Unit1.Em5.ControlNodes".transferPnPRight."step".action1[810] )
      Not()
      Contact( "Unit1.Em5.ControlNodes".cm.interlock.transferPnPRightAxisZ.source.posAbsolute[3] )
      Move(in := 3, out1 => "Unit1.Em5.ControlNodes".cmTransferPnPRightAxisZ.commands.selectSetPosition)
      Coil( "Unit1.Em5.ControlNodes".cm.command.transferPnPRightAxisZ.posAbsolute[3] )
   END_RUNG
   // the same network as SCL:
   #TransferPnPRightAxisZ_IntPos[3]."Int"[1] := NOT (NOT "Unit1.Em5.ControlNodes".cm.softcam.transferPnPRightAxisY.pos08_noInterferenceZone.inPos AND NOT "Unit1.Em5.ControlNodes".cm.softcam.transferPnPRightAxisY.pos08_noInterferenceZone.isBefore);
   #TransferPnPRightAxisZ_IntPos[3]."Int"[2] := NOT "Unit1.Em5.ControlNodes".cm.softcam.transferPnPRightAxisZ.pos03_laserMark.inPos;
   #TransferPnPRightAxisZ_interlock[3](PosiNo := 3,   // "LER_Axis_Absolute"
                           Status := #unitStatus,
                           int1 := #TransferPnPRightAxisZ_IntPos[3]."Int"[1],
                           int2 := #TransferPnPRightAxisZ_IntPos[3]."Int"[2],
                           Bypass := #unitStatus.specialFunctions."Spare 35",
                           commands := "Unit1.Em5.HmiInterface".cmTransferPnPRightAxisZ.commands,
                           interlockOk := "Unit1.Em5.ControlNodes".cm.interlock.transferPnPRightAxisZ.source.posAbsolute,
                           intOut := "Unit1.Em5.HmiInterface".intCondition.Axis_16.Position.intOut);
   #_w1 := NOT (NOT "Unit1.Em5.ControlNodes".transferPnPRight."step".action1[510] AND NOT "Unit1.Em5.ControlNodes".transferPnPRight."step".action1[610] AND NOT "Unit1.Em5.ControlNodes".transferPnPRight."step".action1[710] AND NOT "Unit1.Em5.ControlNodes".transferPnPRight."step".action1[810]) AND "Unit1.Em5.ControlNodes".cm.interlock.transferPnPRightAxisZ.source.posAbsolute[3];
   IF #_w1 THEN "Unit1.Em5.ControlNodes".cmTransferPnPRightAxisZ.commands.selectSetPosition := 3; END_IF;
   "Unit1.Em5.ControlNodes".cm.command.transferPnPRightAxisZ.posAbsolute[3] := #_w1;
END_REGION

REGION Network 181: Transfer PnP Right AxisZ Position Absolute Position4
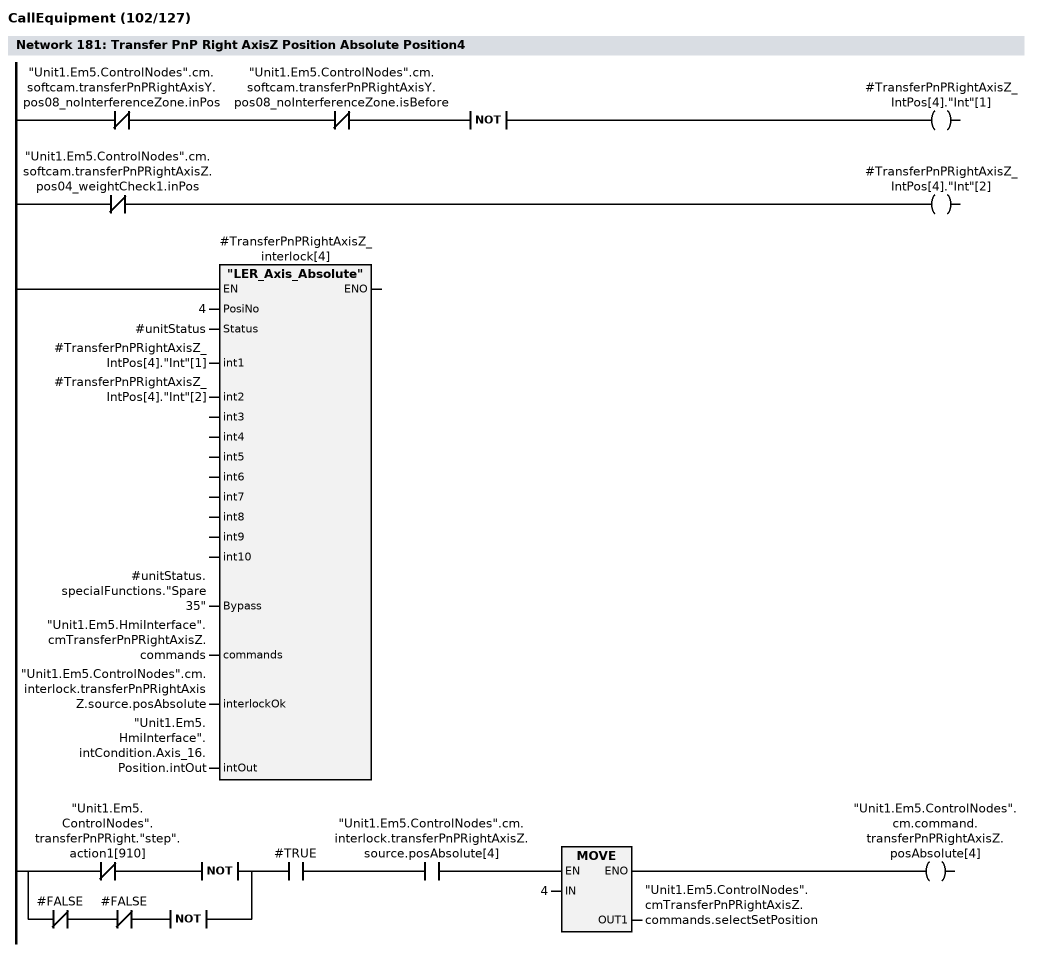
   RUNG wire#powerrail
      I_Contact( "Unit1.Em5.ControlNodes".cm.softcam.transferPnPRightAxisY.pos08_noInterferenceZone.inPos )
      I_Contact( "Unit1.Em5.ControlNodes".cm.softcam.transferPnPRightAxisY.pos08_noInterferenceZone.isBefore )
      Not()
      Coil( #TransferPnPRightAxisZ_IntPos[4]."Int"[1] )
   END_RUNG
   RUNG wire#powerrail
      I_Contact( "Unit1.Em5.ControlNodes".cm.softcam.transferPnPRightAxisZ.pos04_weightCheck1.inPos )
      Coil( #TransferPnPRightAxisZ_IntPos[4]."Int"[2] )
   END_RUNG
   RUNG wire#powerrail
      #TransferPnPRightAxisZ_interlock[4](PosiNo := 4, Status := #unitStatus, int1 := #TransferPnPRightAxisZ_IntPos[4]."Int"[1], int2 := #TransferPnPRightAxisZ_IntPos[4]."Int"[2], int3 :=, int4 :=, int5 :=, int6 :=, int7 :=, int8 :=, int9 :=, int10 :=, Bypass := #unitStatus.specialFunctions."Spare 35", commands := "Unit1.Em5.HmiInterface".cmTransferPnPRightAxisZ.commands, interlockOk := "Unit1.Em5.ControlNodes".cm.interlock.transferPnPRightAxisZ.source.posAbsolute, intOut := "Unit1.Em5.HmiInterface".intCondition.Axis_16.Position.intOut)
   END_RUNG
   RUNG wire#powerrail
      I_Contact( "Unit1.Em5.ControlNodes".transferPnPRight."step".action1[910] )
      Not()
      wire#w1
      Contact( #TRUE )
      Contact( "Unit1.Em5.ControlNodes".cm.interlock.transferPnPRightAxisZ.source.posAbsolute[4] )
      Move(in := 4, out1 => "Unit1.Em5.ControlNodes".cmTransferPnPRightAxisZ.commands.selectSetPosition)
      Coil( "Unit1.Em5.ControlNodes".cm.command.transferPnPRightAxisZ.posAbsolute[4] )
   END_RUNG
   RUNG wire#powerrail
      I_Contact( #FALSE )
      I_Contact( #FALSE )
      Not()
   END_RUNG wire#w1
   // the same network as SCL:
   #TransferPnPRightAxisZ_IntPos[4]."Int"[1] := NOT (NOT "Unit1.Em5.ControlNodes".cm.softcam.transferPnPRightAxisY.pos08_noInterferenceZone.inPos AND NOT "Unit1.Em5.ControlNodes".cm.softcam.transferPnPRightAxisY.pos08_noInterferenceZone.isBefore);
   #TransferPnPRightAxisZ_IntPos[4]."Int"[2] := NOT "Unit1.Em5.ControlNodes".cm.softcam.transferPnPRightAxisZ.pos04_weightCheck1.inPos;
   #TransferPnPRightAxisZ_interlock[4](PosiNo := 4,   // "LER_Axis_Absolute"
                           Status := #unitStatus,
                           int1 := #TransferPnPRightAxisZ_IntPos[4]."Int"[1],
                           int2 := #TransferPnPRightAxisZ_IntPos[4]."Int"[2],
                           Bypass := #unitStatus.specialFunctions."Spare 35",
                           commands := "Unit1.Em5.HmiInterface".cmTransferPnPRightAxisZ.commands,
                           interlockOk := "Unit1.Em5.ControlNodes".cm.interlock.transferPnPRightAxisZ.source.posAbsolute,
                           intOut := "Unit1.Em5.HmiInterface".intCondition.Axis_16.Position.intOut);
   #_w1 := (NOT (NOT "Unit1.Em5.ControlNodes".transferPnPRight."step".action1[910]) OR NOT (NOT #FALSE AND NOT #FALSE)) AND #TRUE AND "Unit1.Em5.ControlNodes".cm.interlock.transferPnPRightAxisZ.source.posAbsolute[4];
   IF #_w1 THEN "Unit1.Em5.ControlNodes".cmTransferPnPRightAxisZ.commands.selectSetPosition := 4; END_IF;
   "Unit1.Em5.ControlNodes".cm.command.transferPnPRightAxisZ.posAbsolute[4] := #_w1;
END_REGION

REGION Network 182: Transfer PnP Right AxisZ Position Absolute Position5
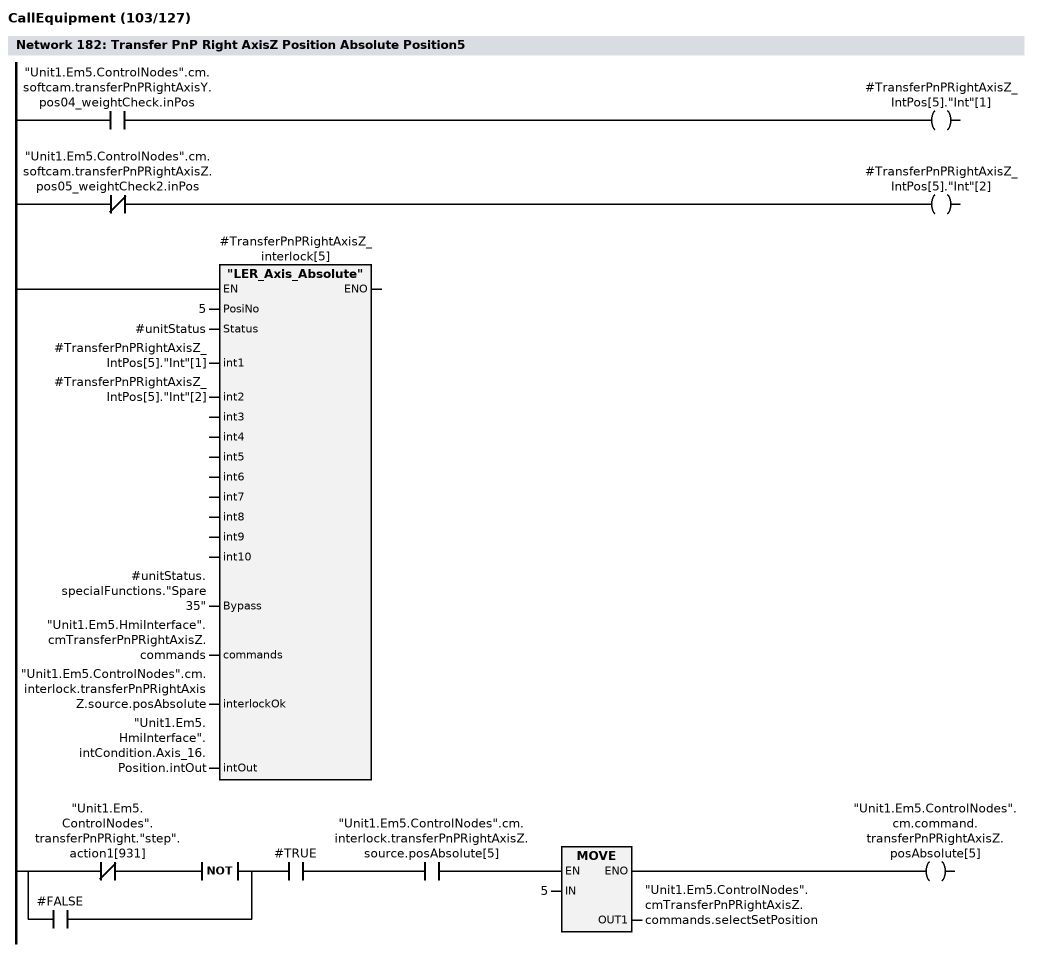
   RUNG wire#powerrail
      Contact( "Unit1.Em5.ControlNodes".cm.softcam.transferPnPRightAxisY.pos04_weightCheck.inPos )
      Coil( #TransferPnPRightAxisZ_IntPos[5]."Int"[1] )
   END_RUNG
   RUNG wire#powerrail
      I_Contact( "Unit1.Em5.ControlNodes".cm.softcam.transferPnPRightAxisZ.pos05_weightCheck2.inPos )
      Coil( #TransferPnPRightAxisZ_IntPos[5]."Int"[2] )
   END_RUNG
   RUNG wire#powerrail
      #TransferPnPRightAxisZ_interlock[5](PosiNo := 5, Status := #unitStatus, int1 := #TransferPnPRightAxisZ_IntPos[5]."Int"[1], int2 := #TransferPnPRightAxisZ_IntPos[5]."Int"[2], int3 :=, int4 :=, int5 :=, int6 :=, int7 :=, int8 :=, int9 :=, int10 :=, Bypass := #unitStatus.specialFunctions."Spare 35", commands := "Unit1.Em5.HmiInterface".cmTransferPnPRightAxisZ.commands, interlockOk := "Unit1.Em5.ControlNodes".cm.interlock.transferPnPRightAxisZ.source.posAbsolute, intOut := "Unit1.Em5.HmiInterface".intCondition.Axis_16.Position.intOut)
   END_RUNG
   RUNG wire#powerrail
      I_Contact( "Unit1.Em5.ControlNodes".transferPnPRight."step".action1[931] )
      Not()
      wire#w1
      Contact( #TRUE )
      Contact( "Unit1.Em5.ControlNodes".cm.interlock.transferPnPRightAxisZ.source.posAbsolute[5] )
      Move(in := 5, out1 => "Unit1.Em5.ControlNodes".cmTransferPnPRightAxisZ.commands.selectSetPosition)
      Coil( "Unit1.Em5.ControlNodes".cm.command.transferPnPRightAxisZ.posAbsolute[5] )
   END_RUNG
   RUNG wire#powerrail
      Contact( #FALSE )
   END_RUNG wire#w1
   // the same network as SCL:
   #TransferPnPRightAxisZ_IntPos[5]."Int"[1] := "Unit1.Em5.ControlNodes".cm.softcam.transferPnPRightAxisY.pos04_weightCheck.inPos;
   #TransferPnPRightAxisZ_IntPos[5]."Int"[2] := NOT "Unit1.Em5.ControlNodes".cm.softcam.transferPnPRightAxisZ.pos05_weightCheck2.inPos;
   #TransferPnPRightAxisZ_interlock[5](PosiNo := 5,   // "LER_Axis_Absolute"
                           Status := #unitStatus,
                           int1 := #TransferPnPRightAxisZ_IntPos[5]."Int"[1],
                           int2 := #TransferPnPRightAxisZ_IntPos[5]."Int"[2],
                           Bypass := #unitStatus.specialFunctions."Spare 35",
                           commands := "Unit1.Em5.HmiInterface".cmTransferPnPRightAxisZ.commands,
                           interlockOk := "Unit1.Em5.ControlNodes".cm.interlock.transferPnPRightAxisZ.source.posAbsolute,
                           intOut := "Unit1.Em5.HmiInterface".intCondition.Axis_16.Position.intOut);
   #_w1 := (NOT (NOT "Unit1.Em5.ControlNodes".transferPnPRight."step".action1[931]) OR #FALSE) AND #TRUE AND "Unit1.Em5.ControlNodes".cm.interlock.transferPnPRightAxisZ.source.posAbsolute[5];
   IF #_w1 THEN "Unit1.Em5.ControlNodes".cmTransferPnPRightAxisZ.commands.selectSetPosition := 5; END_IF;
   "Unit1.Em5.ControlNodes".cm.command.transferPnPRightAxisZ.posAbsolute[5] := #_w1;
END_REGION

REGION Network 183: Transfer PnP Right AxisZ Position Absolute Position7
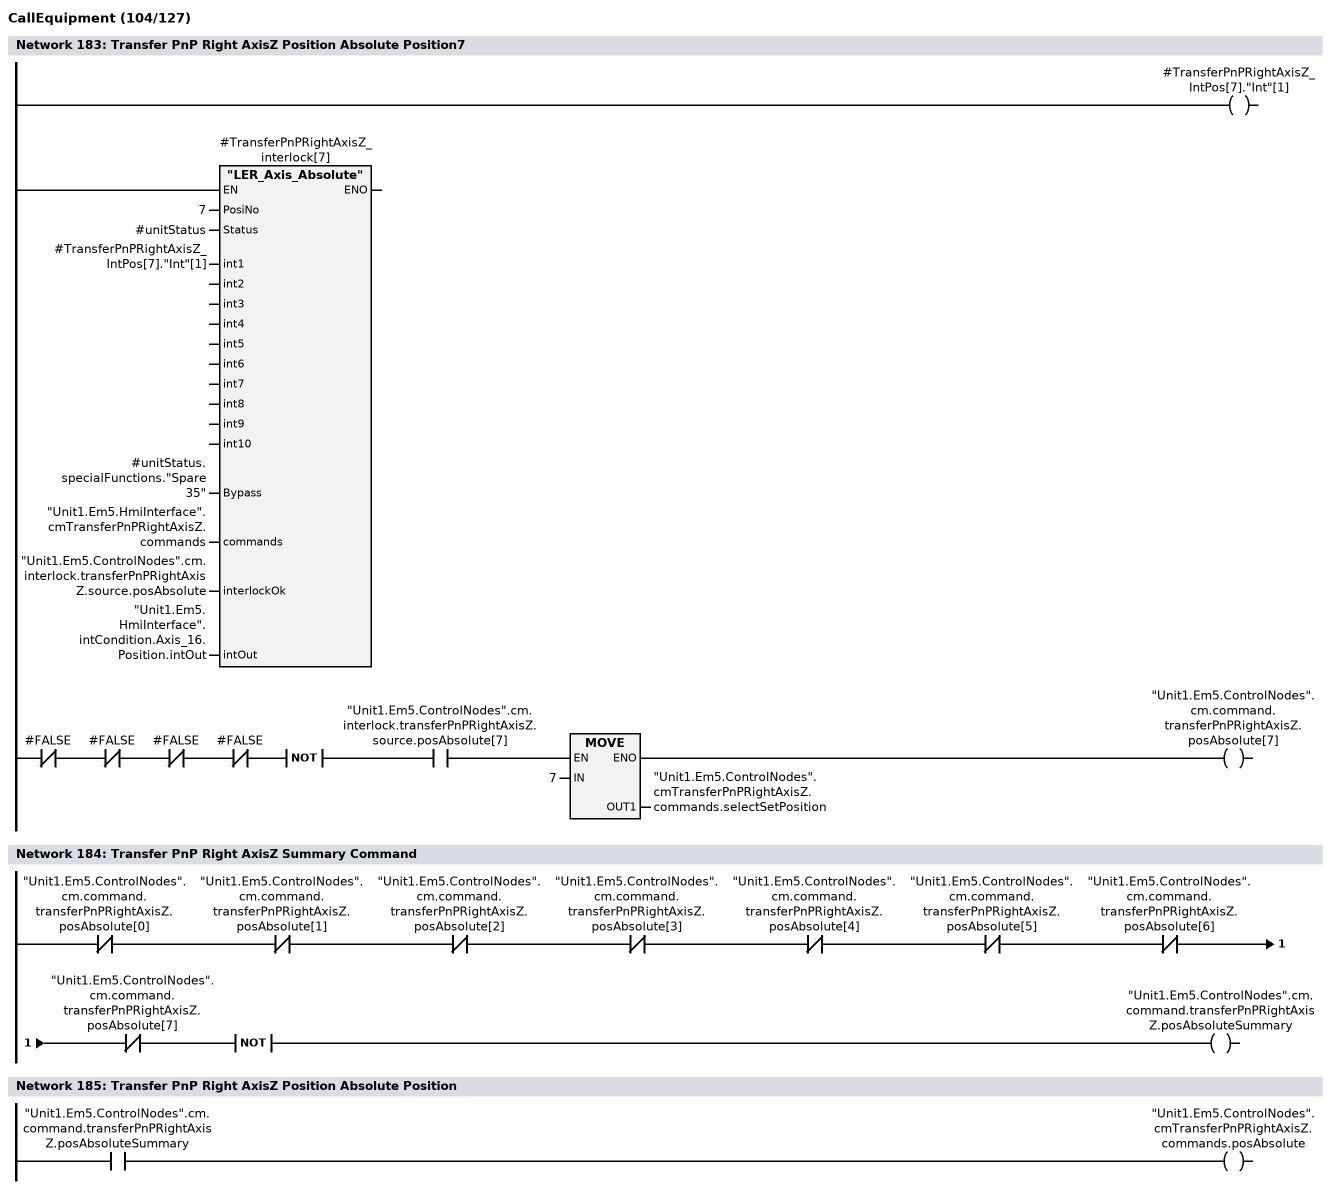
   RUNG wire#powerrail
      Coil( #TransferPnPRightAxisZ_IntPos[7]."Int"[1] )
   END_RUNG
   RUNG wire#powerrail
      #TransferPnPRightAxisZ_interlock[7](PosiNo := 7, Status := #unitStatus, int1 := #TransferPnPRightAxisZ_IntPos[7]."Int"[1], int2 :=, int3 :=, int4 :=, int5 :=, int6 :=, int7 :=, int8 :=, int9 :=, int10 :=, Bypass := #unitStatus.specialFunctions."Spare 35", commands := "Unit1.Em5.HmiInterface".cmTransferPnPRightAxisZ.commands, interlockOk := "Unit1.Em5.ControlNodes".cm.interlock.transferPnPRightAxisZ.source.posAbsolute, intOut := "Unit1.Em5.HmiInterface".intCondition.Axis_16.Position.intOut)
   END_RUNG
   RUNG wire#powerrail
      I_Contact( #FALSE )
      I_Contact( #FALSE )
      I_Contact( #FALSE )
      I_Contact( #FALSE )
      Not()
      Contact( "Unit1.Em5.ControlNodes".cm.interlock.transferPnPRightAxisZ.source.posAbsolute[7] )
      Move(in := 7, out1 => "Unit1.Em5.ControlNodes".cmTransferPnPRightAxisZ.commands.selectSetPosition)
      Coil( "Unit1.Em5.ControlNodes".cm.command.transferPnPRightAxisZ.posAbsolute[7] )
   END_RUNG
   // the same network as SCL:
   #TransferPnPRightAxisZ_IntPos[7]."Int"[1] := TRUE;
   #TransferPnPRightAxisZ_interlock[7](PosiNo := 7,   // "LER_Axis_Absolute"
                           Status := #unitStatus,
                           int1 := #TransferPnPRightAxisZ_IntPos[7]."Int"[1],
                           Bypass := #unitStatus.specialFunctions."Spare 35",
                           commands := "Unit1.Em5.HmiInterface".cmTransferPnPRightAxisZ.commands,
                           interlockOk := "Unit1.Em5.ControlNodes".cm.interlock.transferPnPRightAxisZ.source.posAbsolute,
                           intOut := "Unit1.Em5.HmiInterface".intCondition.Axis_16.Position.intOut);
   #_w1 := NOT (NOT #FALSE AND NOT #FALSE AND NOT #FALSE AND NOT #FALSE) AND "Unit1.Em5.ControlNodes".cm.interlock.transferPnPRightAxisZ.source.posAbsolute[7];
   IF #_w1 THEN "Unit1.Em5.ControlNodes".cmTransferPnPRightAxisZ.commands.selectSetPosition := 7; END_IF;
   "Unit1.Em5.ControlNodes".cm.command.transferPnPRightAxisZ.posAbsolute[7] := #_w1;
END_REGION

REGION Network 184: Transfer PnP Right AxisZ Summary Command
   RUNG wire#powerrail
      I_Contact( "Unit1.Em5.ControlNodes".cm.command.transferPnPRightAxisZ.posAbsolute[0] )
      I_Contact( "Unit1.Em5.ControlNodes".cm.command.transferPnPRightAxisZ.posAbsolute[1] )
      I_Contact( "Unit1.Em5.ControlNodes".cm.command.transferPnPRightAxisZ.posAbsolute[2] )
      I_Contact( "Unit1.Em5.ControlNodes".cm.command.transferPnPRightAxisZ.posAbsolute[3] )
      I_Contact( "Unit1.Em5.ControlNodes".cm.command.transferPnPRightAxisZ.posAbsolute[4] )
      I_Contact( "Unit1.Em5.ControlNodes".cm.command.transferPnPRightAxisZ.posAbsolute[5] )
      I_Contact( "Unit1.Em5.ControlNodes".cm.command.transferPnPRightAxisZ.posAbsolute[6] )
      I_Contact( "Unit1.Em5.ControlNodes".cm.command.transferPnPRightAxisZ.posAbsolute[7] )
      Not()
      Coil( "Unit1.Em5.ControlNodes".cm.command.transferPnPRightAxisZ.posAbsoluteSummary )
   END_RUNG
   // the same network as SCL:
   "Unit1.Em5.ControlNodes".cm.command.transferPnPRightAxisZ.posAbsoluteSummary := NOT (NOT "Unit1.Em5.ControlNodes".cm.command.transferPnPRightAxisZ.posAbsolute[0] AND NOT "Unit1.Em5.ControlNodes".cm.command.transferPnPRightAxisZ.posAbsolute[1] AND NOT "Unit1.Em5.ControlNodes".cm.command.transferPnPRightAxisZ.posAbsolute[2] AND NOT "Unit1.Em5.ControlNodes".cm.command.transferPnPRightAxisZ.posAbsolute[3] AND NOT "Unit1.Em5.ControlNodes".cm.command.transferPnPRightAxisZ.posAbsolute[4] AND NOT "Unit1.Em5.ControlNodes".cm.command.transferPnPRightAxisZ.posAbsolute[5] AND NOT "Unit1.Em5.ControlNodes".cm.command.transferPnPRightAxisZ.posAbsolute[6] AND NOT "Unit1.Em5.ControlNodes".cm.command.transferPnPRightAxisZ.posAbsolute[7]);
END_REGION

REGION Network 185: Transfer PnP Right AxisZ Position Absolute Position
   RUNG wire#powerrail
      Contact( "Unit1.Em5.ControlNodes".cm.command.transferPnPRightAxisZ.posAbsoluteSummary )
      Coil( "Unit1.Em5.ControlNodes".cmTransferPnPRightAxisZ.commands.posAbsolute )
   END_RUNG
   // the same network as SCL:
   "Unit1.Em5.ControlNodes".cmTransferPnPRightAxisZ.commands.posAbsolute := "Unit1.Em5.ControlNodes".cm.command.transferPnPRightAxisZ.posAbsoluteSummary;
END_REGION

REGION Network 186: Transfer PnP Right AxisZ Interlock Summary
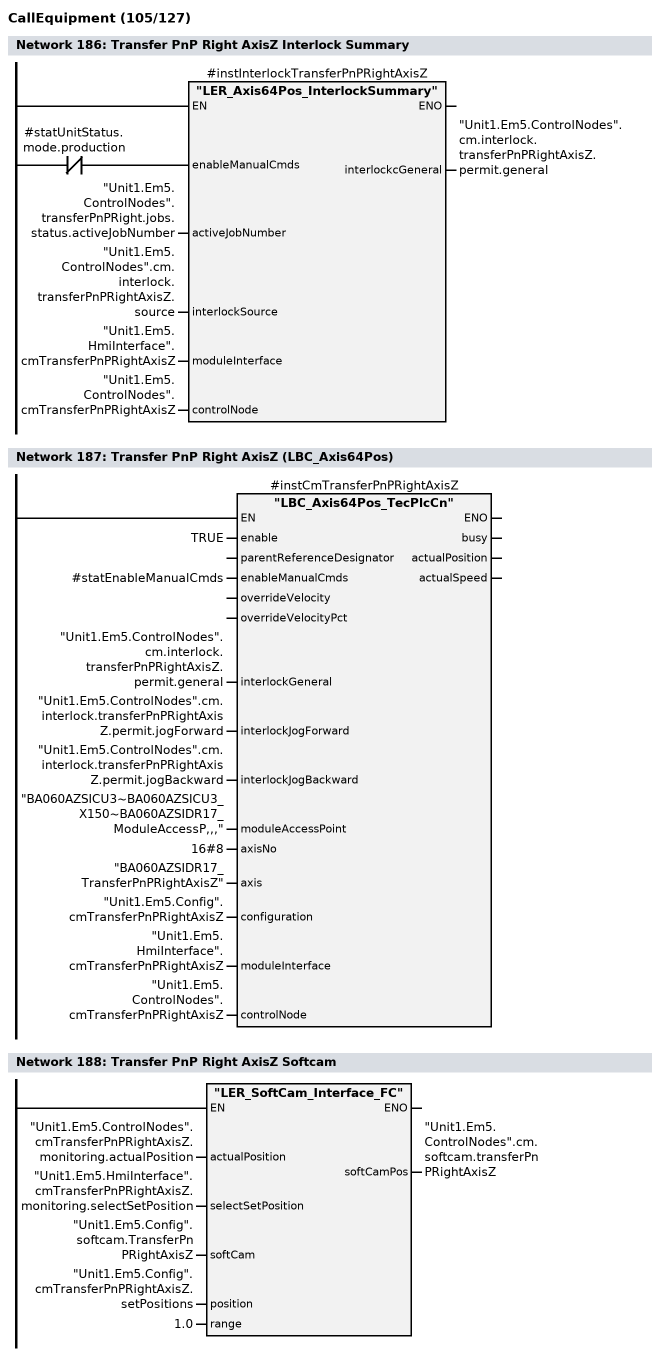
   RUNG wire#powerrail
      #instInterlockTransferPnPRightAxisZ(enableManualCmds := wire#w1, activeJobNumber := "Unit1.Em5.ControlNodes".transferPnPRight.jobs.status.activeJobNumber, interlockSource := "Unit1.Em5.ControlNodes".cm.interlock.transferPnPRightAxisZ.source, moduleInterface := "Unit1.Em5.HmiInterface".cmTransferPnPRightAxisZ, controlNode := "Unit1.Em5.ControlNodes".cmTransferPnPRightAxisZ, interlockcGeneral => "Unit1.Em5.ControlNodes".cm.interlock.transferPnPRightAxisZ.permit.general)
   END_RUNG
   RUNG wire#powerrail
      I_Contact( #statUnitStatus.mode.production )
   END_RUNG wire#w1
   // the same network as SCL:
   #instInterlockTransferPnPRightAxisZ(enableManualCmds := NOT #statUnitStatus.mode.production,   // "LER_Axis64Pos_InterlockSummary"
                           activeJobNumber := "Unit1.Em5.ControlNodes".transferPnPRight.jobs.status.activeJobNumber,
                           interlockSource := "Unit1.Em5.ControlNodes".cm.interlock.transferPnPRightAxisZ.source,
                           moduleInterface := "Unit1.Em5.HmiInterface".cmTransferPnPRightAxisZ,
                           controlNode := "Unit1.Em5.ControlNodes".cmTransferPnPRightAxisZ,
                           interlockcGeneral => "Unit1.Em5.ControlNodes".cm.interlock.transferPnPRightAxisZ.permit.general);
END_REGION

REGION Network 187: Transfer PnP Right AxisZ (LBC_Axis64Pos)
   RUNG wire#powerrail
      #instCmTransferPnPRightAxisZ(enable := TRUE, parentReferenceDesignator :=, enableManualCmds := #statEnableManualCmds, overrideVelocity :=, overrideVelocityPct :=, interlockGeneral := "Unit1.Em5.ControlNodes".cm.interlock.transferPnPRightAxisZ.permit.general, interlockJogForward := "Unit1.Em5.ControlNodes".cm.interlock.transferPnPRightAxisZ.permit.jogForward, interlockJogBackward := "Unit1.Em5.ControlNodes".cm.interlock.transferPnPRightAxisZ.permit.jogBackward, moduleAccessPoint := "BA060AZSICU3~BA060AZSICU3_X150~BA060AZSIDR17_ModuleAccessP,,,", axisNo := 16#8, axis := "BA060AZSIDR17_TransferPnPRightAxisZ", configuration := "Unit1.Em5.Config".cmTransferPnPRightAxisZ, moduleInterface := "Unit1.Em5.HmiInterface".cmTransferPnPRightAxisZ, controlNode := "Unit1.Em5.ControlNodes".cmTransferPnPRightAxisZ, busy =>, actualPosition =>, actualSpeed =>)
   END_RUNG
   // the same network as SCL:
   #instCmTransferPnPRightAxisZ(enable := TRUE,   // "LBC_Axis64Pos_TecPlcCn"
                           enableManualCmds := #statEnableManualCmds,
                           interlockGeneral := "Unit1.Em5.ControlNodes".cm.interlock.transferPnPRightAxisZ.permit.general,
                           interlockJogForward := "Unit1.Em5.ControlNodes".cm.interlock.transferPnPRightAxisZ.permit.jogForward,
                           interlockJogBackward := "Unit1.Em5.ControlNodes".cm.interlock.transferPnPRightAxisZ.permit.jogBackward,
                           moduleAccessPoint := "BA060AZSICU3~BA060AZSICU3_X150~BA060AZSIDR17_ModuleAccessP,,,",
                           axisNo := 16#8,
                           axis := "BA060AZSIDR17_TransferPnPRightAxisZ",
                           configuration := "Unit1.Em5.Config".cmTransferPnPRightAxisZ,
                           moduleInterface := "Unit1.Em5.HmiInterface".cmTransferPnPRightAxisZ,
                           controlNode := "Unit1.Em5.ControlNodes".cmTransferPnPRightAxisZ);
END_REGION

REGION Network 188: Transfer PnP Right AxisZ Softcam
   RUNG wire#powerrail
      "LER_SoftCam_Interface_FC"(actualPosition := "Unit1.Em5.ControlNodes".cmTransferPnPRightAxisZ.monitoring.actualPosition, selectSetPosition := "Unit1.Em5.HmiInterface".cmTransferPnPRightAxisZ.monitoring.selectSetPosition, softCam := "Unit1.Em5.Config".softcam.TransferPnPRightAxisZ, position := "Unit1.Em5.Config".cmTransferPnPRightAxisZ.setPositions, range := 1.0, softCamPos => "Unit1.Em5.ControlNodes".cm.softcam.transferPnPRightAxisZ)
   END_RUNG
   // the same network as SCL:
   "LER_SoftCam_Interface_FC"(actualPosition := "Unit1.Em5.ControlNodes".cmTransferPnPRightAxisZ.monitoring.actualPosition,
                           selectSetPosition := "Unit1.Em5.HmiInterface".cmTransferPnPRightAxisZ.monitoring.selectSetPosition,
                           softCam := "Unit1.Em5.Config".softcam.TransferPnPRightAxisZ,
                           position := "Unit1.Em5.Config".cmTransferPnPRightAxisZ.setPositions,
                           range := 1.0,
                           softCamPos => "Unit1.Em5.ControlNodes".cm.softcam.transferPnPRightAxisZ);
END_REGION

REGION Network 190: Transfer P&P Right Z-Axis Interlock Condition
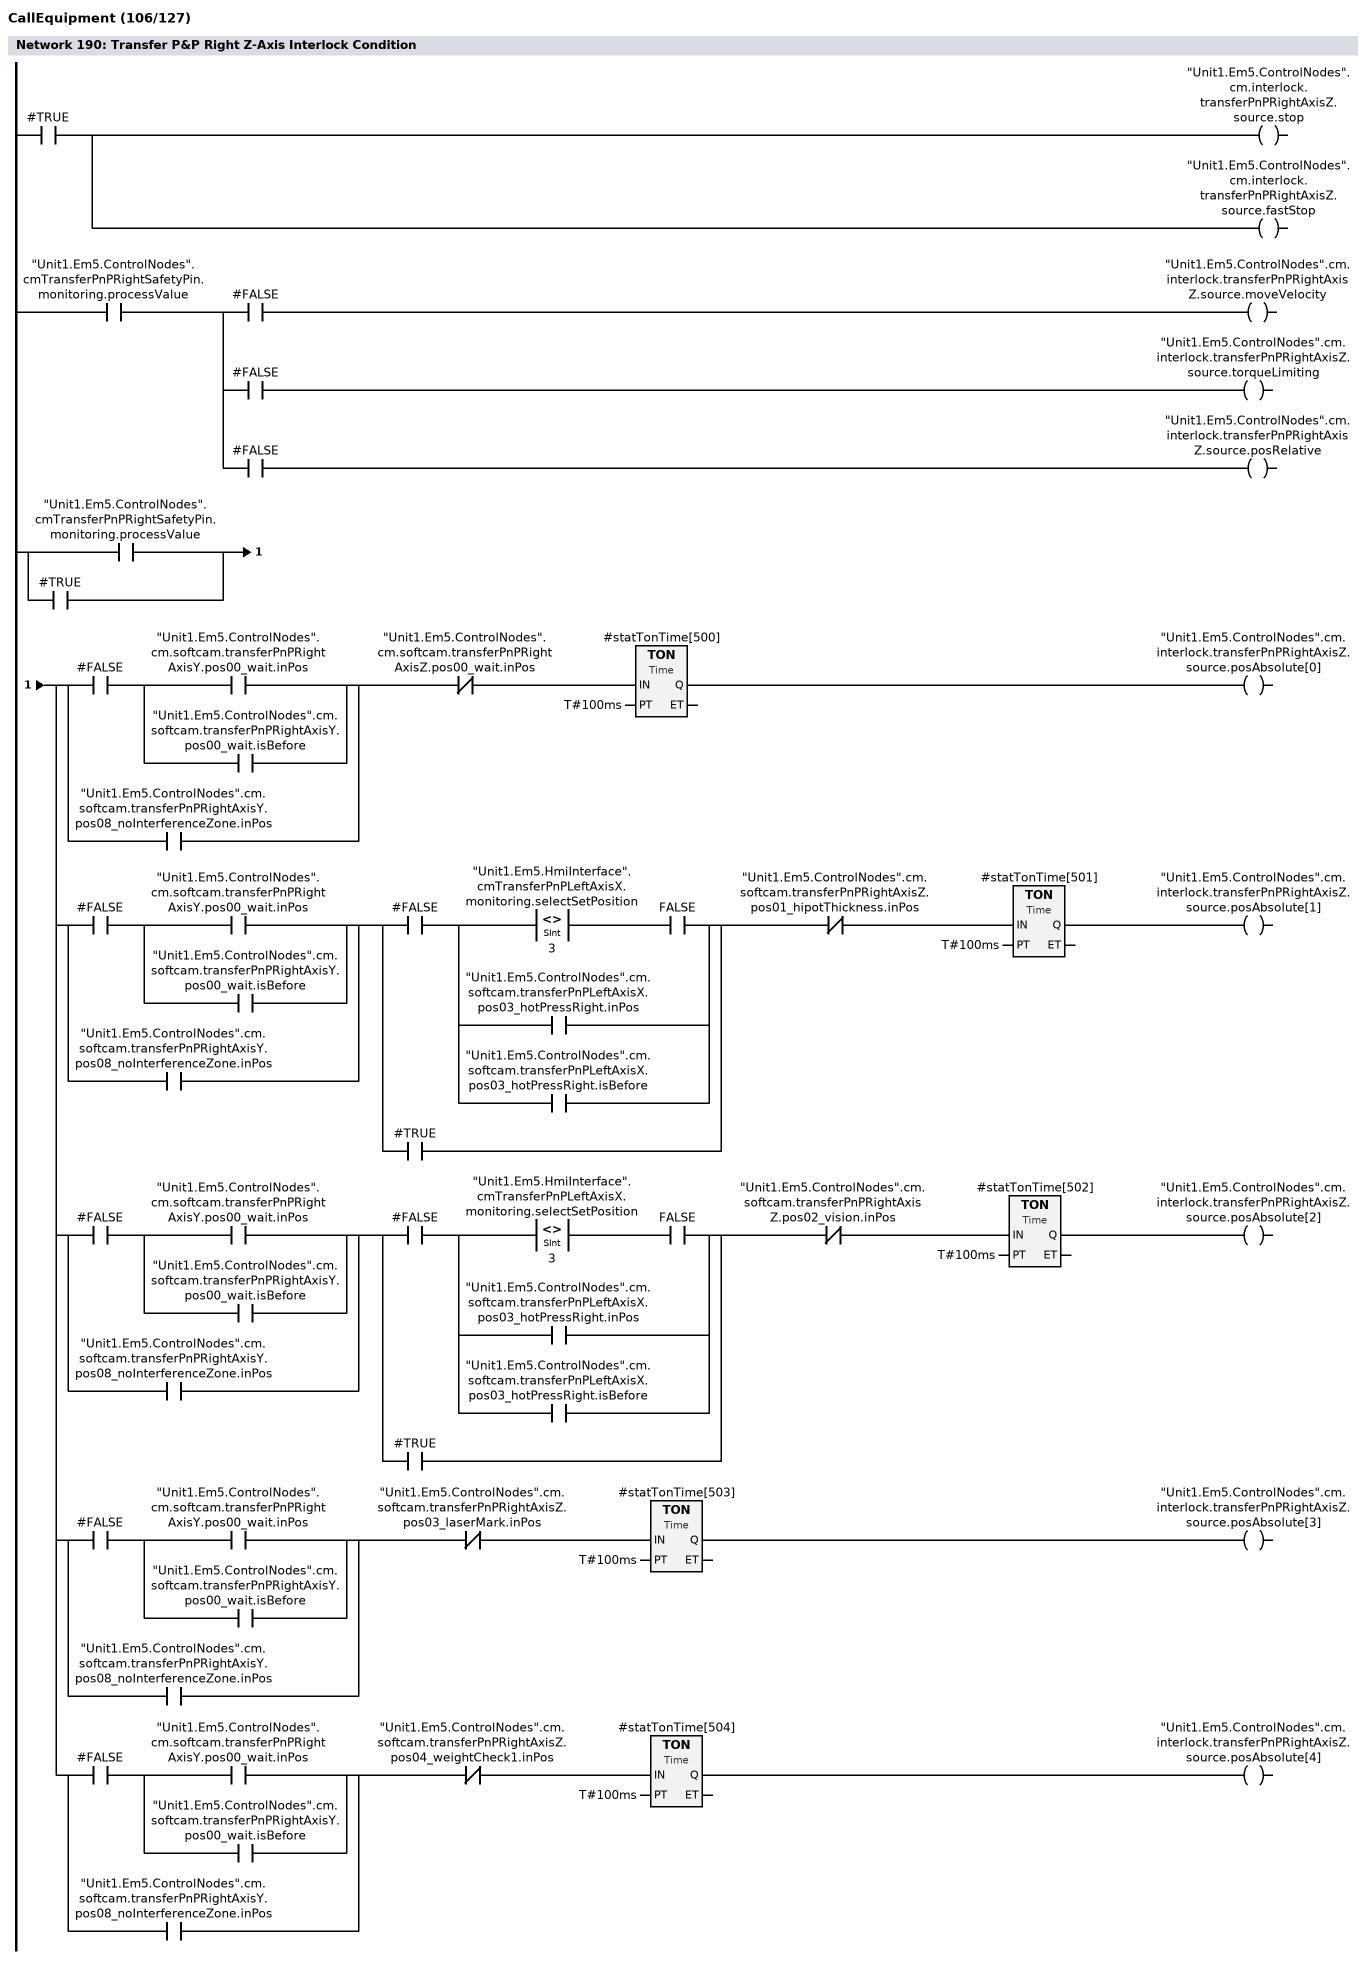
   RUNG wire#powerrail
      Contact( #TRUE )
      wire#w1
      Coil( "Unit1.Em5.ControlNodes".cm.interlock.transferPnPRightAxisZ.source.stop )
   END_RUNG
   RUNG wire#w1
      Coil( "Unit1.Em5.ControlNodes".cm.interlock.transferPnPRightAxisZ.source.fastStop )
   END_RUNG
   RUNG wire#powerrail
      Contact( "Unit1.Em5.ControlNodes".cmTransferPnPRightSafetyPin.monitoring.processValue )
      wire#w2
      Contact( #FALSE )
      Coil( "Unit1.Em5.ControlNodes".cm.interlock.transferPnPRightAxisZ.source.moveVelocity )
   END_RUNG
   RUNG wire#w2
      Contact( #FALSE )
      Coil( "Unit1.Em5.ControlNodes".cm.interlock.transferPnPRightAxisZ.source.torqueLimiting )
   END_RUNG
   RUNG wire#w2
      Contact( #FALSE )
      Coil( "Unit1.Em5.ControlNodes".cm.interlock.transferPnPRightAxisZ.source.posRelative )
   END_RUNG
   RUNG wire#powerrail
      Contact( "Unit1.Em5.ControlNodes".cmTransferPnPRightSafetyPin.monitoring.processValue )
      wire#w3
      Contact( #FALSE )
      wire#w4
      Contact( "Unit1.Em5.ControlNodes".cm.softcam.transferPnPRightAxisY.pos00_wait.inPos )
      wire#w5
      I_Contact( "Unit1.Em5.ControlNodes".cm.softcam.transferPnPRightAxisZ.pos00_wait.inPos )
      { S7_Templates := "time_type := Time" } #statTonTime[500].TON(pt := T#100ms, et =>)
      Coil( "Unit1.Em5.ControlNodes".cm.interlock.transferPnPRightAxisZ.source.posAbsolute[0] )
   END_RUNG
   RUNG wire#powerrail
      Contact( #TRUE )
   END_RUNG wire#w3
   RUNG wire#w4
      Contact( "Unit1.Em5.ControlNodes".cm.softcam.transferPnPRightAxisY.pos00_wait.isBefore )
   END_RUNG wire#w5
   RUNG wire#w3
      Contact( "Unit1.Em5.ControlNodes".cm.softcam.transferPnPRightAxisY.pos08_noInterferenceZone.inPos )
   END_RUNG wire#w5
   RUNG wire#w3
      Contact( #FALSE )
      wire#w6
      Contact( "Unit1.Em5.ControlNodes".cm.softcam.transferPnPRightAxisY.pos00_wait.inPos )
      wire#w7
      Contact( #FALSE )
      wire#w8
      { S7_Templates := "SrcType := SInt" } NE_Contact(in1 := "Unit1.Em5.HmiInterface".cmTransferPnPLeftAxisX.monitoring.selectSetPosition, in2 := 3)
      Contact( FALSE )
      wire#w9
      I_Contact( "Unit1.Em5.ControlNodes".cm.softcam.transferPnPRightAxisZ.pos01_hipotThickness.inPos )
      { S7_Templates := "time_type := Time" } #statTonTime[501].TON(pt := T#100ms, et =>)
      Coil( "Unit1.Em5.ControlNodes".cm.interlock.transferPnPRightAxisZ.source.posAbsolute[1] )
   END_RUNG
   RUNG wire#w6
      Contact( "Unit1.Em5.ControlNodes".cm.softcam.transferPnPRightAxisY.pos00_wait.isBefore )
   END_RUNG wire#w7
   RUNG wire#w3
      Contact( "Unit1.Em5.ControlNodes".cm.softcam.transferPnPRightAxisY.pos08_noInterferenceZone.inPos )
   END_RUNG wire#w7
   RUNG wire#w8
      Contact( "Unit1.Em5.ControlNodes".cm.softcam.transferPnPLeftAxisX.pos03_hotPressRight.inPos )
   END_RUNG wire#w9
   RUNG wire#w8
      Contact( "Unit1.Em5.ControlNodes".cm.softcam.transferPnPLeftAxisX.pos03_hotPressRight.isBefore )
   END_RUNG wire#w9
   RUNG wire#w7
      Contact( #TRUE )
   END_RUNG wire#w9
   RUNG wire#w3
      Contact( #FALSE )
      wire#w10
      Contact( "Unit1.Em5.ControlNodes".cm.softcam.transferPnPRightAxisY.pos00_wait.inPos )
      wire#w11
      Contact( #FALSE )
      wire#w12
      { S7_Templates := "SrcType := SInt" } NE_Contact(in1 := "Unit1.Em5.HmiInterface".cmTransferPnPLeftAxisX.monitoring.selectSetPosition, in2 := 3)
      Contact( FALSE )
      wire#w13
      I_Contact( "Unit1.Em5.ControlNodes".cm.softcam.transferPnPRightAxisZ.pos02_vision.inPos )
      { S7_Templates := "time_type := Time" } #statTonTime[502].TON(pt := T#100ms, et =>)
      Coil( "Unit1.Em5.ControlNodes".cm.interlock.transferPnPRightAxisZ.source.posAbsolute[2] )
   END_RUNG
   RUNG wire#w10
      Contact( "Unit1.Em5.ControlNodes".cm.softcam.transferPnPRightAxisY.pos00_wait.isBefore )
   END_RUNG wire#w11
   RUNG wire#w3
      Contact( "Unit1.Em5.ControlNodes".cm.softcam.transferPnPRightAxisY.pos08_noInterferenceZone.inPos )
   END_RUNG wire#w11
   RUNG wire#w12
      Contact( "Unit1.Em5.ControlNodes".cm.softcam.transferPnPLeftAxisX.pos03_hotPressRight.inPos )
   END_RUNG wire#w13
   RUNG wire#w12
      Contact( "Unit1.Em5.ControlNodes".cm.softcam.transferPnPLeftAxisX.pos03_hotPressRight.isBefore )
   END_RUNG wire#w13
   RUNG wire#w11
      Contact( #TRUE )
   END_RUNG wire#w13
   RUNG wire#w3
      Contact( #FALSE )
      wire#w14
      Contact( "Unit1.Em5.ControlNodes".cm.softcam.transferPnPRightAxisY.pos00_wait.inPos )
      wire#w15
      I_Contact( "Unit1.Em5.ControlNodes".cm.softcam.transferPnPRightAxisZ.pos03_laserMark.inPos )
      { S7_Templates := "time_type := Time" } #statTonTime[503].TON(pt := T#100ms, et =>)
      Coil( "Unit1.Em5.ControlNodes".cm.interlock.transferPnPRightAxisZ.source.posAbsolute[3] )
   END_RUNG
   RUNG wire#w14
      Contact( "Unit1.Em5.ControlNodes".cm.softcam.transferPnPRightAxisY.pos00_wait.isBefore )
   END_RUNG wire#w15
   RUNG wire#w3
      Contact( "Unit1.Em5.ControlNodes".cm.softcam.transferPnPRightAxisY.pos08_noInterferenceZone.inPos )
   END_RUNG wire#w15
   RUNG wire#w3
      Contact( #FALSE )
      wire#w16
      Contact( "Unit1.Em5.ControlNodes".cm.softcam.transferPnPRightAxisY.pos00_wait.inPos )
      wire#w17
      I_Contact( "Unit1.Em5.ControlNodes".cm.softcam.transferPnPRightAxisZ.pos04_weightCheck1.inPos )
      { S7_Templates := "time_type := Time" } #statTonTime[504].TON(pt := T#100ms, et =>)
      Coil( "Unit1.Em5.ControlNodes".cm.interlock.transferPnPRightAxisZ.source.posAbsolute[4] )
   END_RUNG
   RUNG wire#w16
      Contact( "Unit1.Em5.ControlNodes".cm.softcam.transferPnPRightAxisY.pos00_wait.isBefore )
   END_RUNG wire#w17
   RUNG wire#w3
      Contact( "Unit1.Em5.ControlNodes".cm.softcam.transferPnPRightAxisY.pos08_noInterferenceZone.inPos )
   END_RUNG wire#w17
   // the same network as SCL:
   "Unit1.Em5.ControlNodes".cm.interlock.transferPnPRightAxisZ.source.stop := #TRUE;
   "Unit1.Em5.ControlNodes".cm.interlock.transferPnPRightAxisZ.source.fastStop := #TRUE;
   "Unit1.Em5.ControlNodes".cm.interlock.transferPnPRightAxisZ.source.moveVelocity := "Unit1.Em5.ControlNodes".cmTransferPnPRightSafetyPin.monitoring.processValue AND #FALSE;
   "Unit1.Em5.ControlNodes".cm.interlock.transferPnPRightAxisZ.source.torqueLimiting := "Unit1.Em5.ControlNodes".cmTransferPnPRightSafetyPin.monitoring.processValue AND #FALSE;
   "Unit1.Em5.ControlNodes".cm.interlock.transferPnPRightAxisZ.source.posRelative := "Unit1.Em5.ControlNodes".cmTransferPnPRightSafetyPin.monitoring.processValue AND #FALSE;
   #_w1 := "Unit1.Em5.ControlNodes".cmTransferPnPRightSafetyPin.monitoring.processValue OR #TRUE;
   #statTonTime[500].TON(IN := #_w1 AND ((#FALSE AND ("Unit1.Em5.ControlNodes".cm.softcam.transferPnPRightAxisY.pos00_wait.inPos OR "Unit1.Em5.ControlNodes".cm.softcam.transferPnPRightAxisY.pos00_wait.isBefore)) OR "Unit1.Em5.ControlNodes".cm.softcam.transferPnPRightAxisY.pos08_noInterferenceZone.inPos) AND NOT "Unit1.Em5.ControlNodes".cm.softcam.transferPnPRightAxisZ.pos00_wait.inPos,
                         PT := T#100ms);
   "Unit1.Em5.ControlNodes".cm.interlock.transferPnPRightAxisZ.source.posAbsolute[0] := #statTonTime[500].Q;
   #statTonTime[501].TON(IN := #_w1 AND ((#FALSE AND ("Unit1.Em5.ControlNodes".cm.softcam.transferPnPRightAxisY.pos00_wait.inPos OR "Unit1.Em5.ControlNodes".cm.softcam.transferPnPRightAxisY.pos00_wait.isBefore)) OR "Unit1.Em5.ControlNodes".cm.softcam.transferPnPRightAxisY.pos08_noInterferenceZone.inPos) AND ((#FALSE AND ((("Unit1.Em5.HmiInterface".cmTransferPnPLeftAxisX.monitoring.selectSetPosition <> 3) AND FALSE) OR "Unit1.Em5.ControlNodes".cm.softcam.transferPnPLeftAxisX.pos03_hotPressRight.inPos OR "Unit1.Em5.ControlNodes".cm.softcam.transferPnPLeftAxisX.pos03_hotPressRight.isBefore)) OR #TRUE) AND NOT "Unit1.Em5.ControlNodes".cm.softcam.transferPnPRightAxisZ.pos01_hipotThickness.inPos,
                         PT := T#100ms);
   "Unit1.Em5.ControlNodes".cm.interlock.transferPnPRightAxisZ.source.posAbsolute[1] := #statTonTime[501].Q;
   #statTonTime[502].TON(IN := #_w1 AND ((#FALSE AND ("Unit1.Em5.ControlNodes".cm.softcam.transferPnPRightAxisY.pos00_wait.inPos OR "Unit1.Em5.ControlNodes".cm.softcam.transferPnPRightAxisY.pos00_wait.isBefore)) OR "Unit1.Em5.ControlNodes".cm.softcam.transferPnPRightAxisY.pos08_noInterferenceZone.inPos) AND ((#FALSE AND ((("Unit1.Em5.HmiInterface".cmTransferPnPLeftAxisX.monitoring.selectSetPosition <> 3) AND FALSE) OR "Unit1.Em5.ControlNodes".cm.softcam.transferPnPLeftAxisX.pos03_hotPressRight.inPos OR "Unit1.Em5.ControlNodes".cm.softcam.transferPnPLeftAxisX.pos03_hotPressRight.isBefore)) OR #TRUE) AND NOT "Unit1.Em5.ControlNodes".cm.softcam.transferPnPRightAxisZ.pos02_vision.inPos,
                         PT := T#100ms);
   "Unit1.Em5.ControlNodes".cm.interlock.transferPnPRightAxisZ.source.posAbsolute[2] := #statTonTime[502].Q;
   #statTonTime[503].TON(IN := #_w1 AND ((#FALSE AND ("Unit1.Em5.ControlNodes".cm.softcam.transferPnPRightAxisY.pos00_wait.inPos OR "Unit1.Em5.ControlNodes".cm.softcam.transferPnPRightAxisY.pos00_wait.isBefore)) OR "Unit1.Em5.ControlNodes".cm.softcam.transferPnPRightAxisY.pos08_noInterferenceZone.inPos) AND NOT "Unit1.Em5.ControlNodes".cm.softcam.transferPnPRightAxisZ.pos03_laserMark.inPos,
                         PT := T#100ms);
   "Unit1.Em5.ControlNodes".cm.interlock.transferPnPRightAxisZ.source.posAbsolute[3] := #statTonTime[503].Q;
   #statTonTime[504].TON(IN := #_w1 AND ((#FALSE AND ("Unit1.Em5.ControlNodes".cm.softcam.transferPnPRightAxisY.pos00_wait.inPos OR "Unit1.Em5.ControlNodes".cm.softcam.transferPnPRightAxisY.pos00_wait.isBefore)) OR "Unit1.Em5.ControlNodes".cm.softcam.transferPnPRightAxisY.pos08_noInterferenceZone.inPos) AND NOT "Unit1.Em5.ControlNodes".cm.softcam.transferPnPRightAxisZ.pos04_weightCheck1.inPos,
                         PT := T#100ms);
   "Unit1.Em5.ControlNodes".cm.interlock.transferPnPRightAxisZ.source.posAbsolute[4] := #statTonTime[504].Q;
END_REGION

REGION Network 192: ******************** Brake Test (Axis) ********************
END_REGION

REGION Network 193: Transfer P&P Left Z-Axis Brake Test Error
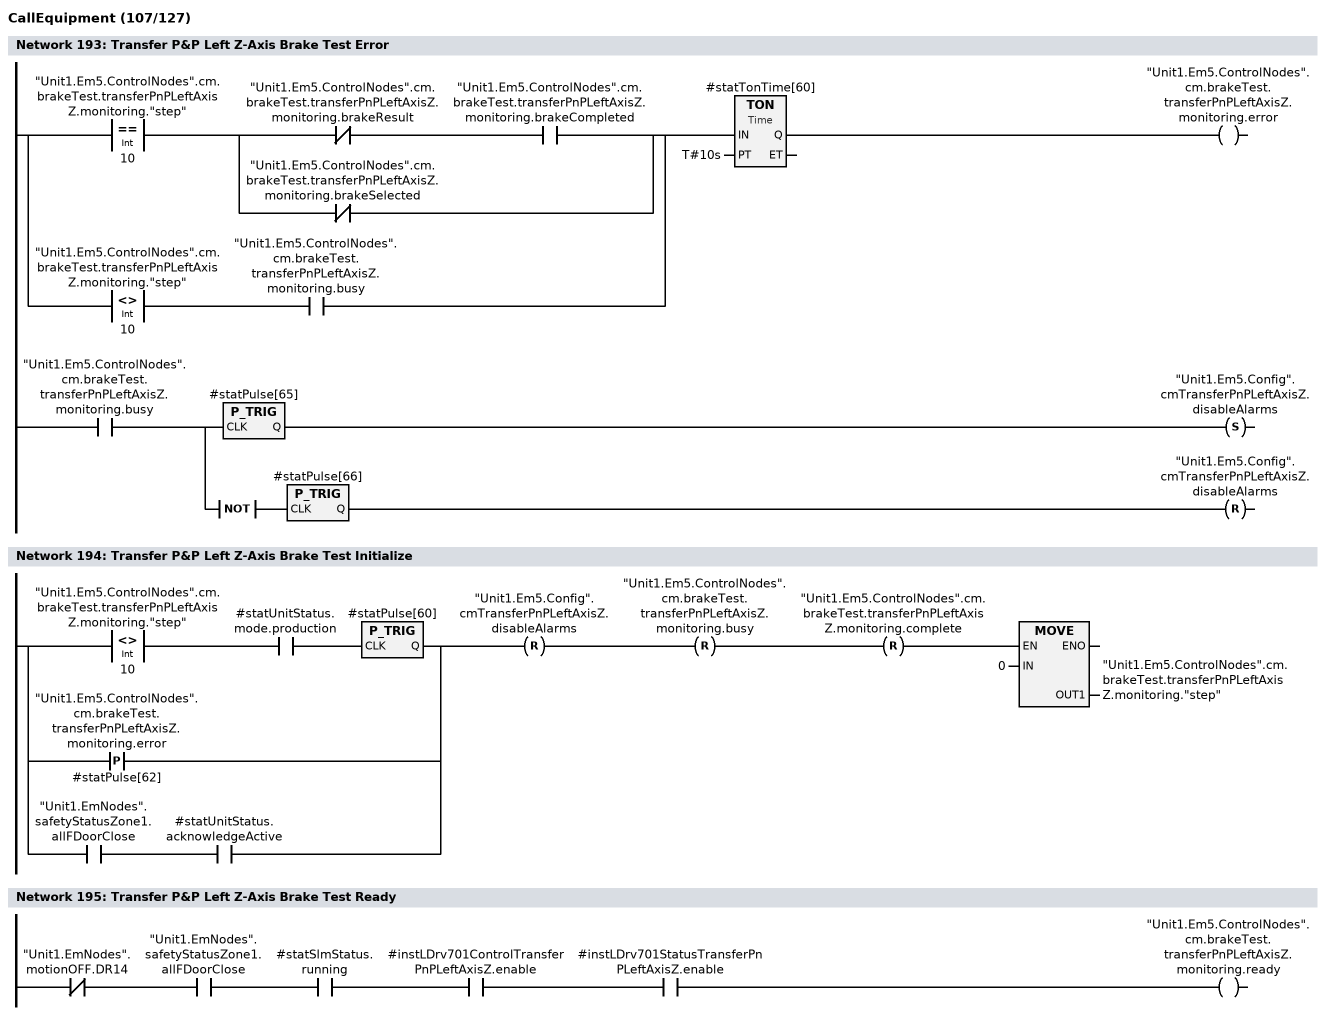
   RUNG wire#powerrail
      { S7_Templates := "SrcType := Int" } EQ_Contact(in1 := "Unit1.Em5.ControlNodes".cm.brakeTest.transferPnPLeftAxisZ.monitoring."step", in2 := 10)
      wire#w1
      I_Contact( "Unit1.Em5.ControlNodes".cm.brakeTest.transferPnPLeftAxisZ.monitoring.brakeResult )
      Contact( "Unit1.Em5.ControlNodes".cm.brakeTest.transferPnPLeftAxisZ.monitoring.brakeCompleted )
      wire#w2
      { S7_Templates := "time_type := Time" } #statTonTime[60].TON(pt := T#10s, et =>)
      Coil( "Unit1.Em5.ControlNodes".cm.brakeTest.transferPnPLeftAxisZ.monitoring.error )
   END_RUNG
   RUNG wire#w1
      I_Contact( "Unit1.Em5.ControlNodes".cm.brakeTest.transferPnPLeftAxisZ.monitoring.brakeSelected )
   END_RUNG wire#w2
   RUNG wire#powerrail
      { S7_Templates := "SrcType := Int" } NE_Contact(in1 := "Unit1.Em5.ControlNodes".cm.brakeTest.transferPnPLeftAxisZ.monitoring."step", in2 := 10)
      Contact( "Unit1.Em5.ControlNodes".cm.brakeTest.transferPnPLeftAxisZ.monitoring.busy )
   END_RUNG wire#w2
   RUNG wire#powerrail
      Contact( "Unit1.Em5.ControlNodes".cm.brakeTest.transferPnPLeftAxisZ.monitoring.busy )
      wire#w3
      P_Trig( #statPulse[65] )
      S_Coil( "Unit1.Em5.Config".cmTransferPnPLeftAxisZ.disableAlarms )
   END_RUNG
   RUNG wire#w3
      Not()
      P_Trig( #statPulse[66] )
      R_Coil( "Unit1.Em5.Config".cmTransferPnPLeftAxisZ.disableAlarms )
   END_RUNG
   // the same network as SCL:
   #statTonTime[60].TON(IN := (("Unit1.Em5.ControlNodes".cm.brakeTest.transferPnPLeftAxisZ.monitoring."step" = 10) AND ((NOT "Unit1.Em5.ControlNodes".cm.brakeTest.transferPnPLeftAxisZ.monitoring.brakeResult AND "Unit1.Em5.ControlNodes".cm.brakeTest.transferPnPLeftAxisZ.monitoring.brakeCompleted) OR NOT "Unit1.Em5.ControlNodes".cm.brakeTest.transferPnPLeftAxisZ.monitoring.brakeSelected)) OR (("Unit1.Em5.ControlNodes".cm.brakeTest.transferPnPLeftAxisZ.monitoring."step" <> 10) AND "Unit1.Em5.ControlNodes".cm.brakeTest.transferPnPLeftAxisZ.monitoring.busy),
                        PT := T#10s);
   "Unit1.Em5.ControlNodes".cm.brakeTest.transferPnPLeftAxisZ.monitoring.error := #statTonTime[60].Q;
   #_w1 := "Unit1.Em5.ControlNodes".cm.brakeTest.transferPnPLeftAxisZ.monitoring.busy AND NOT #statPulse[65];   // rising edge
   #statPulse[65] := "Unit1.Em5.ControlNodes".cm.brakeTest.transferPnPLeftAxisZ.monitoring.busy;
   IF #_w1 THEN "Unit1.Em5.Config".cmTransferPnPLeftAxisZ.disableAlarms := TRUE; END_IF;
   #_w2 := NOT "Unit1.Em5.ControlNodes".cm.brakeTest.transferPnPLeftAxisZ.monitoring.busy AND NOT #statPulse[66];   // rising edge
   #statPulse[66] := NOT "Unit1.Em5.ControlNodes".cm.brakeTest.transferPnPLeftAxisZ.monitoring.busy;
   IF #_w2 THEN "Unit1.Em5.Config".cmTransferPnPLeftAxisZ.disableAlarms := FALSE; END_IF;
END_REGION

REGION Network 194: Transfer P&P Left Z-Axis Brake Test Initialize
   RUNG wire#powerrail
      { S7_Templates := "SrcType := Int" } NE_Contact(in1 := "Unit1.Em5.ControlNodes".cm.brakeTest.transferPnPLeftAxisZ.monitoring."step", in2 := 10)
      Contact( #statUnitStatus.mode.production )
      P_Trig( #statPulse[60] )
      wire#w1
      R_Coil( "Unit1.Em5.Config".cmTransferPnPLeftAxisZ.disableAlarms )
      R_Coil( "Unit1.Em5.ControlNodes".cm.brakeTest.transferPnPLeftAxisZ.monitoring.busy )
      R_Coil( "Unit1.Em5.ControlNodes".cm.brakeTest.transferPnPLeftAxisZ.monitoring.complete )
      Move(in := 0, out1 => "Unit1.Em5.ControlNodes".cm.brakeTest.transferPnPLeftAxisZ.monitoring."step")
   END_RUNG
   RUNG wire#powerrail
      P_Contact(operand := "Unit1.Em5.ControlNodes".cm.brakeTest.transferPnPLeftAxisZ.monitoring.error, bit := #statPulse[62])
   END_RUNG wire#w1
   RUNG wire#powerrail
      Contact( "Unit1.EmNodes".safetyStatusZone1.allFDoorClose )
      Contact( #statUnitStatus.acknowledgeActive )
   END_RUNG wire#w1
   // the same network as SCL:
   #_w1 := ("Unit1.Em5.ControlNodes".cm.brakeTest.transferPnPLeftAxisZ.monitoring."step" <> 10) AND #statUnitStatus.mode.production;
   #_w2 := #_w1 AND NOT #statPulse[60];   // rising edge
   #statPulse[60] := #_w1;
   #_w3 := "Unit1.Em5.ControlNodes".cm.brakeTest.transferPnPLeftAxisZ.monitoring.error AND NOT #statPulse[62];   // rising edge of "Unit1.Em5.ControlNodes".cm.brakeTest.transferPnPLeftAxisZ.monitoring.error
   #statPulse[62] := "Unit1.Em5.ControlNodes".cm.brakeTest.transferPnPLeftAxisZ.monitoring.error;
   IF #_w2 OR #_w3 OR ("Unit1.EmNodes".safetyStatusZone1.allFDoorClose AND #statUnitStatus.acknowledgeActive) THEN
       "Unit1.Em5.Config".cmTransferPnPLeftAxisZ.disableAlarms := FALSE;
       "Unit1.Em5.ControlNodes".cm.brakeTest.transferPnPLeftAxisZ.monitoring.busy := FALSE;
       "Unit1.Em5.ControlNodes".cm.brakeTest.transferPnPLeftAxisZ.monitoring.complete := FALSE;
       "Unit1.Em5.ControlNodes".cm.brakeTest.transferPnPLeftAxisZ.monitoring."step" := 0;
   END_IF;
END_REGION

REGION Network 195: Transfer P&P Left Z-Axis Brake Test Ready
   RUNG wire#powerrail
      I_Contact( "Unit1.EmNodes".motionOFF.DR14 )
      Contact( "Unit1.EmNodes".safetyStatusZone1.allFDoorClose )
      Contact( #statSlmStatus.running )
      Contact( #instLDrv701ControlTransferPnPLeftAxisZ.enable )
      Contact( #instLDrv701StatusTransferPnPLeftAxisZ.enable )
      Coil( "Unit1.Em5.ControlNodes".cm.brakeTest.transferPnPLeftAxisZ.monitoring.ready )
   END_RUNG
   // the same network as SCL:
   "Unit1.Em5.ControlNodes".cm.brakeTest.transferPnPLeftAxisZ.monitoring.ready := NOT "Unit1.EmNodes".motionOFF.DR14 AND "Unit1.EmNodes".safetyStatusZone1.allFDoorClose AND #statSlmStatus.running AND #instLDrv701ControlTransferPnPLeftAxisZ.enable AND #instLDrv701StatusTransferPnPLeftAxisZ.enable;
END_REGION

REGION Network 196: Transfer P&P Left Z-Axis Brake Test Commands
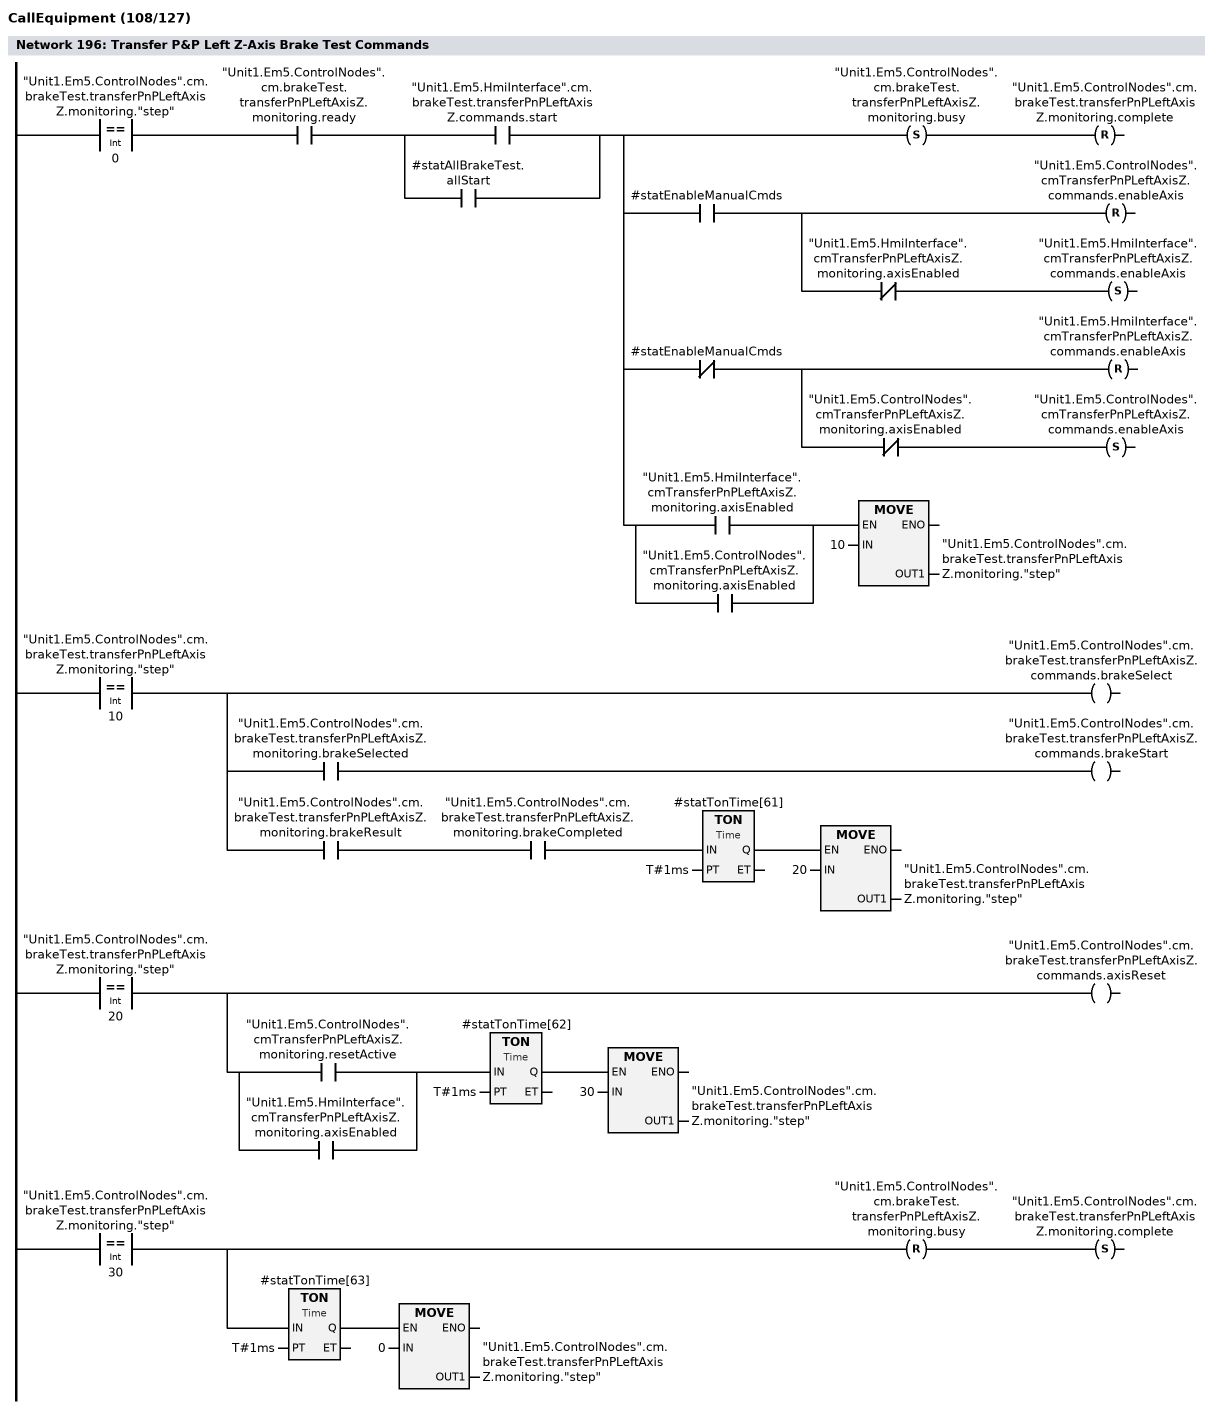
   RUNG wire#powerrail
      { S7_Templates := "SrcType := Int" } EQ_Contact(in1 := "Unit1.Em5.ControlNodes".cm.brakeTest.transferPnPLeftAxisZ.monitoring."step", in2 := 0)
      Contact( "Unit1.Em5.ControlNodes".cm.brakeTest.transferPnPLeftAxisZ.monitoring.ready )
      wire#w1
      Contact( "Unit1.Em5.HmiInterface".cm.brakeTest.transferPnPLeftAxisZ.commands.start )
      wire#w2
      S_Coil( "Unit1.Em5.ControlNodes".cm.brakeTest.transferPnPLeftAxisZ.monitoring.busy )
      R_Coil( "Unit1.Em5.ControlNodes".cm.brakeTest.transferPnPLeftAxisZ.monitoring.complete )
   END_RUNG
   RUNG wire#w1
      Contact( #statAllBrakeTest.allStart )
   END_RUNG wire#w2
   RUNG wire#w2
      Contact( #statEnableManualCmds )
      wire#w3
      R_Coil( "Unit1.Em5.ControlNodes".cmTransferPnPLeftAxisZ.commands.enableAxis )
   END_RUNG
   RUNG wire#w3
      I_Contact( "Unit1.Em5.HmiInterface".cmTransferPnPLeftAxisZ.monitoring.axisEnabled )
      S_Coil( "Unit1.Em5.HmiInterface".cmTransferPnPLeftAxisZ.commands.enableAxis )
   END_RUNG
   RUNG wire#w2
      I_Contact( #statEnableManualCmds )
      wire#w4
      R_Coil( "Unit1.Em5.HmiInterface".cmTransferPnPLeftAxisZ.commands.enableAxis )
   END_RUNG
   RUNG wire#w4
      I_Contact( "Unit1.Em5.ControlNodes".cmTransferPnPLeftAxisZ.monitoring.axisEnabled )
      S_Coil( "Unit1.Em5.ControlNodes".cmTransferPnPLeftAxisZ.commands.enableAxis )
   END_RUNG
   RUNG wire#w2
      Contact( "Unit1.Em5.HmiInterface".cmTransferPnPLeftAxisZ.monitoring.axisEnabled )
      wire#w5
      Move(in := 10, out1 => "Unit1.Em5.ControlNodes".cm.brakeTest.transferPnPLeftAxisZ.monitoring."step")
   END_RUNG
   RUNG wire#w2
      Contact( "Unit1.Em5.ControlNodes".cmTransferPnPLeftAxisZ.monitoring.axisEnabled )
   END_RUNG wire#w5
   RUNG wire#powerrail
      { S7_Templates := "SrcType := Int" } EQ_Contact(in1 := "Unit1.Em5.ControlNodes".cm.brakeTest.transferPnPLeftAxisZ.monitoring."step", in2 := 10)
      wire#w6
      Coil( "Unit1.Em5.ControlNodes".cm.brakeTest.transferPnPLeftAxisZ.commands.brakeSelect )
   END_RUNG
   RUNG wire#w6
      Contact( "Unit1.Em5.ControlNodes".cm.brakeTest.transferPnPLeftAxisZ.monitoring.brakeSelected )
      Coil( "Unit1.Em5.ControlNodes".cm.brakeTest.transferPnPLeftAxisZ.commands.brakeStart )
   END_RUNG
   RUNG wire#w6
      Contact( "Unit1.Em5.ControlNodes".cm.brakeTest.transferPnPLeftAxisZ.monitoring.brakeResult )
      Contact( "Unit1.Em5.ControlNodes".cm.brakeTest.transferPnPLeftAxisZ.monitoring.brakeCompleted )
      { S7_Templates := "time_type := Time" } #statTonTime[61].TON(pt := T#1ms, et =>)
      Move(in := 20, out1 => "Unit1.Em5.ControlNodes".cm.brakeTest.transferPnPLeftAxisZ.monitoring."step")
   END_RUNG
   RUNG wire#powerrail
      { S7_Templates := "SrcType := Int" } EQ_Contact(in1 := "Unit1.Em5.ControlNodes".cm.brakeTest.transferPnPLeftAxisZ.monitoring."step", in2 := 20)
      wire#w7
      Coil( "Unit1.Em5.ControlNodes".cm.brakeTest.transferPnPLeftAxisZ.commands.axisReset )
   END_RUNG
   RUNG wire#w7
      Contact( "Unit1.Em5.ControlNodes".cmTransferPnPLeftAxisZ.monitoring.resetActive )
      wire#w8
      { S7_Templates := "time_type := Time" } #statTonTime[62].TON(pt := T#1ms, et =>)
      Move(in := 30, out1 => "Unit1.Em5.ControlNodes".cm.brakeTest.transferPnPLeftAxisZ.monitoring."step")
   END_RUNG
   RUNG wire#w7
      Contact( "Unit1.Em5.HmiInterface".cmTransferPnPLeftAxisZ.monitoring.axisEnabled )
   END_RUNG wire#w8
   RUNG wire#powerrail
      { S7_Templates := "SrcType := Int" } EQ_Contact(in1 := "Unit1.Em5.ControlNodes".cm.brakeTest.transferPnPLeftAxisZ.monitoring."step", in2 := 30)
      wire#w9
      R_Coil( "Unit1.Em5.ControlNodes".cm.brakeTest.transferPnPLeftAxisZ.monitoring.busy )
      S_Coil( "Unit1.Em5.ControlNodes".cm.brakeTest.transferPnPLeftAxisZ.monitoring.complete )
   END_RUNG
   RUNG wire#w9
      { S7_Templates := "time_type := Time" } #statTonTime[63].TON(pt := T#1ms, et =>)
      Move(in := 0, out1 => "Unit1.Em5.ControlNodes".cm.brakeTest.transferPnPLeftAxisZ.monitoring."step")
   END_RUNG
   // the same network as SCL:
   #_w1 := ("Unit1.Em5.ControlNodes".cm.brakeTest.transferPnPLeftAxisZ.monitoring."step" = 0) AND "Unit1.Em5.ControlNodes".cm.brakeTest.transferPnPLeftAxisZ.monitoring.ready AND ("Unit1.Em5.HmiInterface".cm.brakeTest.transferPnPLeftAxisZ.commands.start OR #statAllBrakeTest.allStart);
   IF #_w1 THEN
       "Unit1.Em5.ControlNodes".cm.brakeTest.transferPnPLeftAxisZ.monitoring.busy := TRUE;
       "Unit1.Em5.ControlNodes".cm.brakeTest.transferPnPLeftAxisZ.monitoring.complete := FALSE;
   END_IF;
   #_w2 := #_w1 AND #statEnableManualCmds;
   IF #_w2 THEN "Unit1.Em5.ControlNodes".cmTransferPnPLeftAxisZ.commands.enableAxis := FALSE; END_IF;
   IF #_w2 AND NOT "Unit1.Em5.HmiInterface".cmTransferPnPLeftAxisZ.monitoring.axisEnabled THEN
       "Unit1.Em5.HmiInterface".cmTransferPnPLeftAxisZ.commands.enableAxis := TRUE;
   END_IF;
   #_w3 := #_w1 AND NOT #statEnableManualCmds;
   IF #_w3 THEN "Unit1.Em5.HmiInterface".cmTransferPnPLeftAxisZ.commands.enableAxis := FALSE; END_IF;
   IF #_w3 AND NOT "Unit1.Em5.ControlNodes".cmTransferPnPLeftAxisZ.monitoring.axisEnabled THEN
       "Unit1.Em5.ControlNodes".cmTransferPnPLeftAxisZ.commands.enableAxis := TRUE;
   END_IF;
   IF #_w1 AND ("Unit1.Em5.HmiInterface".cmTransferPnPLeftAxisZ.monitoring.axisEnabled OR "Unit1.Em5.ControlNodes".cmTransferPnPLeftAxisZ.monitoring.axisEnabled) THEN
       "Unit1.Em5.ControlNodes".cm.brakeTest.transferPnPLeftAxisZ.monitoring."step" := 10;
   END_IF;
   "Unit1.Em5.ControlNodes".cm.brakeTest.transferPnPLeftAxisZ.commands.brakeSelect := "Unit1.Em5.ControlNodes".cm.brakeTest.transferPnPLeftAxisZ.monitoring."step" = 10;
   "Unit1.Em5.ControlNodes".cm.brakeTest.transferPnPLeftAxisZ.commands.brakeStart := "Unit1.Em5.ControlNodes".cm.brakeTest.transferPnPLeftAxisZ.commands.brakeSelect AND "Unit1.Em5.ControlNodes".cm.brakeTest.transferPnPLeftAxisZ.monitoring.brakeSelected;
   #statTonTime[61].TON(IN := "Unit1.Em5.ControlNodes".cm.brakeTest.transferPnPLeftAxisZ.commands.brakeSelect AND "Unit1.Em5.ControlNodes".cm.brakeTest.transferPnPLeftAxisZ.monitoring.brakeResult AND "Unit1.Em5.ControlNodes".cm.brakeTest.transferPnPLeftAxisZ.monitoring.brakeCompleted,
                        PT := T#1ms);
   IF #statTonTime[61].Q THEN
       "Unit1.Em5.ControlNodes".cm.brakeTest.transferPnPLeftAxisZ.monitoring."step" := 20;
   END_IF;
   "Unit1.Em5.ControlNodes".cm.brakeTest.transferPnPLeftAxisZ.commands.axisReset := "Unit1.Em5.ControlNodes".cm.brakeTest.transferPnPLeftAxisZ.monitoring."step" = 20;
   #statTonTime[62].TON(IN := "Unit1.Em5.ControlNodes".cm.brakeTest.transferPnPLeftAxisZ.commands.axisReset AND ("Unit1.Em5.ControlNodes".cmTransferPnPLeftAxisZ.monitoring.resetActive OR "Unit1.Em5.HmiInterface".cmTransferPnPLeftAxisZ.monitoring.axisEnabled),
                        PT := T#1ms);
   IF #statTonTime[62].Q THEN
       "Unit1.Em5.ControlNodes".cm.brakeTest.transferPnPLeftAxisZ.monitoring."step" := 30;
   END_IF;
   #_w4 := "Unit1.Em5.ControlNodes".cm.brakeTest.transferPnPLeftAxisZ.monitoring."step" = 30;
   IF #_w4 THEN
       "Unit1.Em5.ControlNodes".cm.brakeTest.transferPnPLeftAxisZ.monitoring.busy := FALSE;
       "Unit1.Em5.ControlNodes".cm.brakeTest.transferPnPLeftAxisZ.monitoring.complete := TRUE;
   END_IF;
   #statTonTime[63].TON(IN := #_w4, PT := T#1ms);
   IF #statTonTime[63].Q THEN
       "Unit1.Em5.ControlNodes".cm.brakeTest.transferPnPLeftAxisZ.monitoring."step" := 0;
   END_IF;
END_REGION

REGION Network 197: Transfer P&P Left Z-Axis Brake Test Monitoring
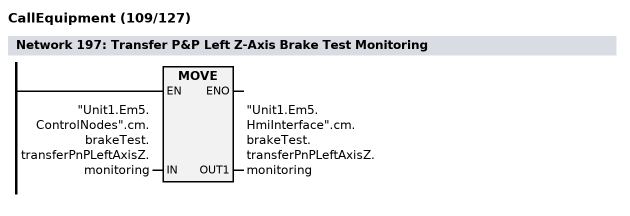
   RUNG wire#powerrail
      Move(in := "Unit1.Em5.ControlNodes".cm.brakeTest.transferPnPLeftAxisZ.monitoring, out1 => "Unit1.Em5.HmiInterface".cm.brakeTest.transferPnPLeftAxisZ.monitoring)
   END_RUNG
   // the same network as SCL:
   "Unit1.Em5.HmiInterface".cm.brakeTest.transferPnPLeftAxisZ.monitoring := "Unit1.Em5.ControlNodes".cm.brakeTest.transferPnPLeftAxisZ.monitoring;
END_REGION

REGION Network 198: Call Transfer Left Z-Axis Telegram 701
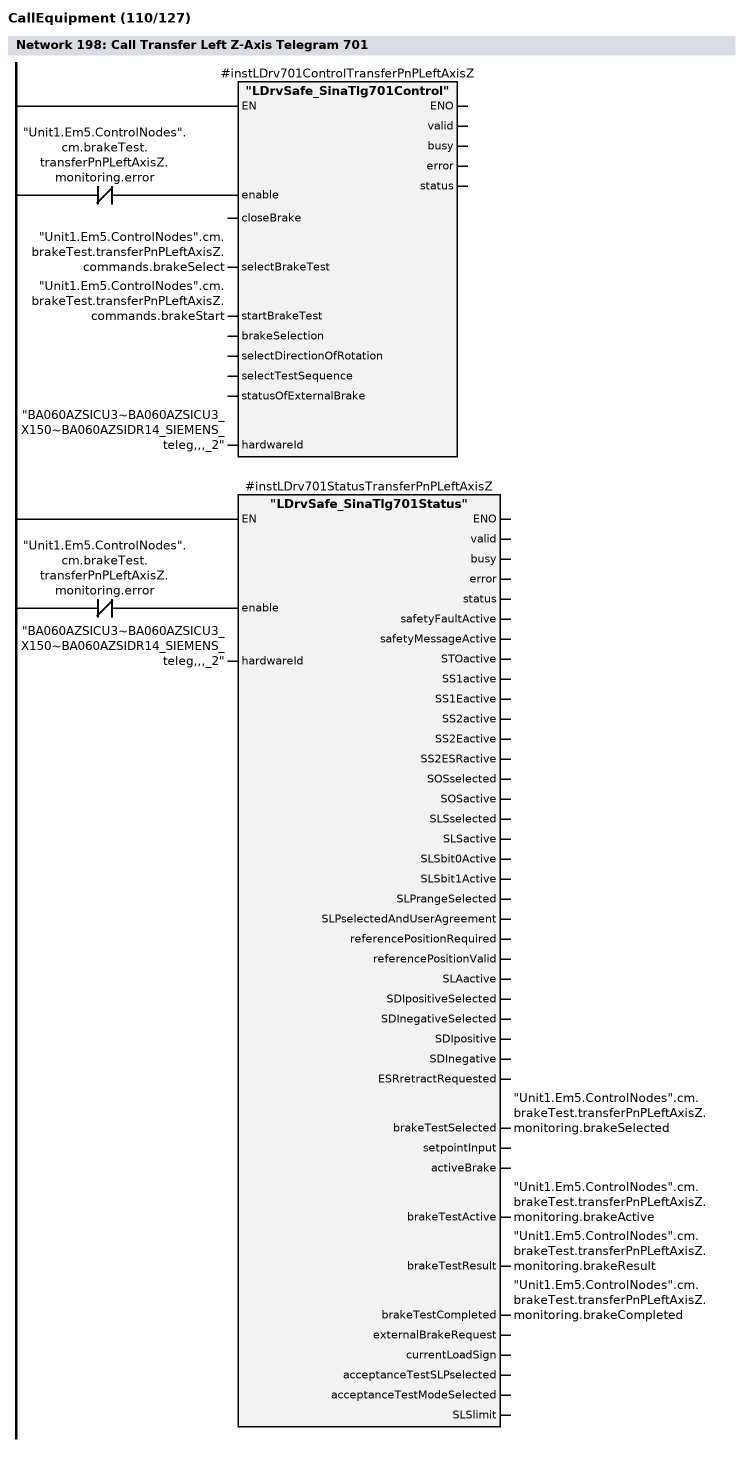
   RUNG wire#powerrail
      #instLDrv701ControlTransferPnPLeftAxisZ(enable := wire#w1, closeBrake :=, selectBrakeTest := "Unit1.Em5.ControlNodes".cm.brakeTest.transferPnPLeftAxisZ.commands.brakeSelect, startBrakeTest := "Unit1.Em5.ControlNodes".cm.brakeTest.transferPnPLeftAxisZ.commands.brakeStart, brakeSelection :=, selectDirectionOfRotation :=, selectTestSequence :=, statusOfExternalBrake :=, hardwareId := "BA060AZSICU3~BA060AZSICU3_X150~BA060AZSIDR14_SIEMENS_teleg,,,_2", valid =>, busy =>, error =>, status =>)
   END_RUNG
   RUNG wire#powerrail
      I_Contact( "Unit1.Em5.ControlNodes".cm.brakeTest.transferPnPLeftAxisZ.monitoring.error )
   END_RUNG wire#w1
   RUNG wire#powerrail
      #instLDrv701StatusTransferPnPLeftAxisZ(enable := wire#w2, hardwareId := "BA060AZSICU3~BA060AZSICU3_X150~BA060AZSIDR14_SIEMENS_teleg,,,_2", valid =>, busy =>, error =>, status =>, safetyFaultActive =>, safetyMessageActive =>, STOactive =>, SS1active =>, SS1Eactive =>, SS2active =>, SS2Eactive =>, SS2ESRactive =>, SOSselected =>, SOSactive =>, SLSselected =>, SLSactive =>, SLSbit0Active =>, SLSbit1Active =>, SLPrangeSelected =>, SLPselectedAndUserAgreement =>, referencePositionRequired =>, referencePositionValid =>, SLAactive =>, SDIpositiveSelected =>, SDInegativeSelected =>, SDIpositive =>, SDInegative =>, ESRretractRequested =>, brakeTestSelected => "Unit1.Em5.ControlNodes".cm.brakeTest.transferPnPLeftAxisZ.monitoring.brakeSelected, setpointInput =>, activeBrake =>, brakeTestActive => "Unit1.Em5.ControlNodes".cm.brakeTest.transferPnPLeftAxisZ.monitoring.brakeActive, brakeTestResult => "Unit1.Em5.ControlNodes".cm.brakeTest.transferPnPLeftAxisZ.monitoring.brakeResult, brakeTestCompleted => "Unit1.Em5.ControlNodes".cm.brakeTest.transferPnPLeftAxisZ.monitoring.brakeCompleted, externalBrakeRequest =>, currentLoadSign =>, acceptanceTestSLPselected =>, acceptanceTestModeSelected =>, SLSlimit =>)
   END_RUNG
   RUNG wire#powerrail
      I_Contact( "Unit1.Em5.ControlNodes".cm.brakeTest.transferPnPLeftAxisZ.monitoring.error )
   END_RUNG wire#w2
   // the same network as SCL:
   #instLDrv701ControlTransferPnPLeftAxisZ(enable := NOT "Unit1.Em5.ControlNodes".cm.brakeTest.transferPnPLeftAxisZ.monitoring.error,   // "LDrvSafe_SinaTlg701Control"
                           selectBrakeTest := "Unit1.Em5.ControlNodes".cm.brakeTest.transferPnPLeftAxisZ.commands.brakeSelect,
                           startBrakeTest := "Unit1.Em5.ControlNodes".cm.brakeTest.transferPnPLeftAxisZ.commands.brakeStart,
                           hardwareId := "BA060AZSICU3~BA060AZSICU3_X150~BA060AZSIDR14_SIEMENS_teleg,,,_2");
   #instLDrv701StatusTransferPnPLeftAxisZ(enable := NOT "Unit1.Em5.ControlNodes".cm.brakeTest.transferPnPLeftAxisZ.monitoring.error,   // "LDrvSafe_SinaTlg701Status"
                           hardwareId := "BA060AZSICU3~BA060AZSICU3_X150~BA060AZSIDR14_SIEMENS_teleg,,,_2",
                           brakeTestSelected => "Unit1.Em5.ControlNodes".cm.brakeTest.transferPnPLeftAxisZ.monitoring.brakeSelected,
                           brakeTestActive => "Unit1.Em5.ControlNodes".cm.brakeTest.transferPnPLeftAxisZ.monitoring.brakeActive,
                           brakeTestResult => "Unit1.Em5.ControlNodes".cm.brakeTest.transferPnPLeftAxisZ.monitoring.brakeResult,
                           brakeTestCompleted => "Unit1.Em5.ControlNodes".cm.brakeTest.transferPnPLeftAxisZ.monitoring.brakeCompleted);
END_REGION

REGION Network 200: JR Out P&P Right Z-Axis Brake Test Error
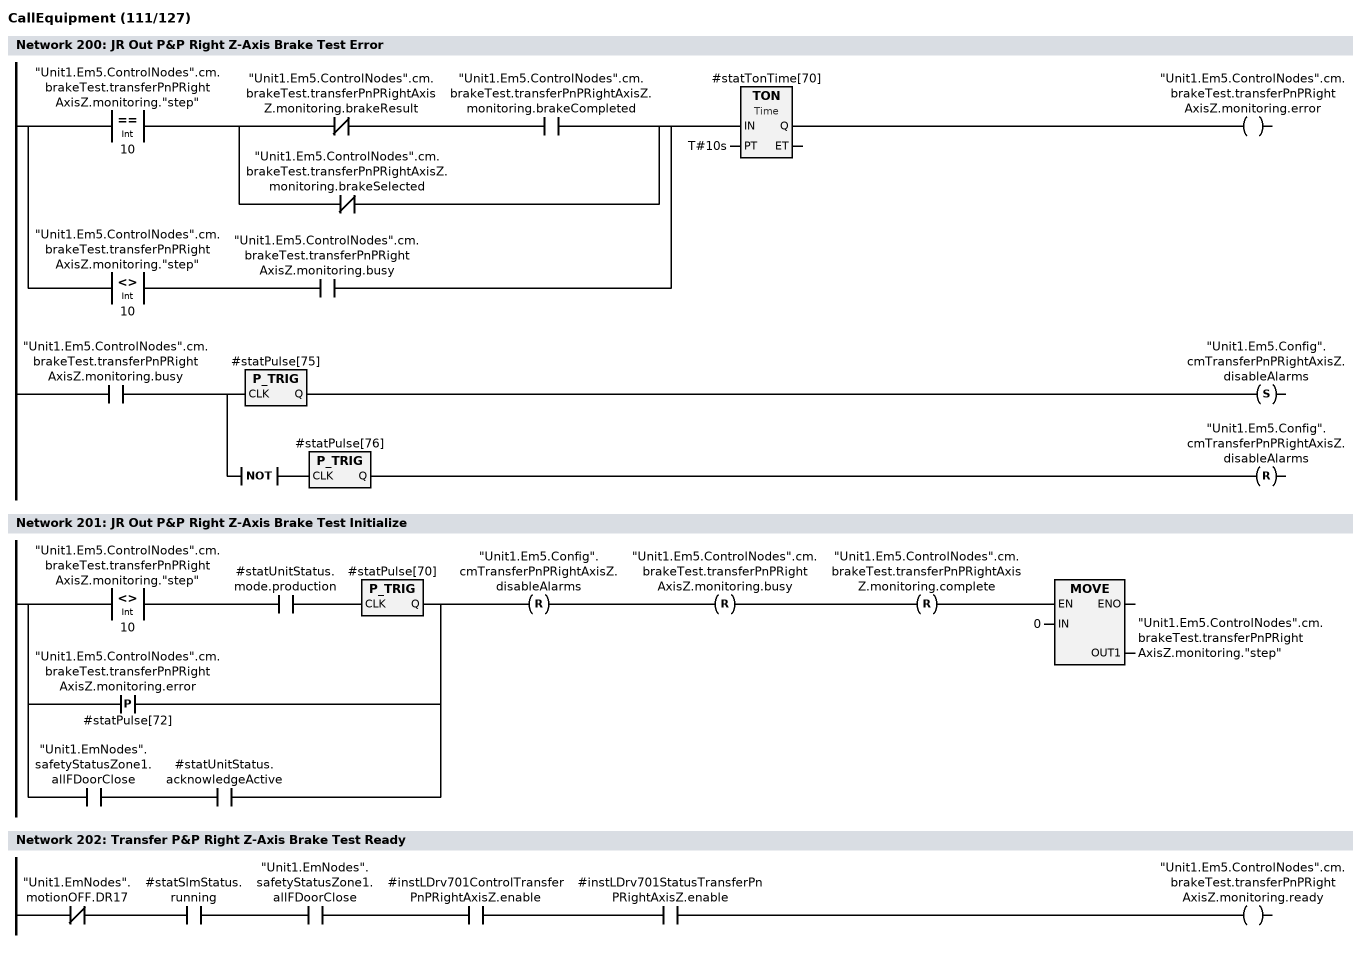
   RUNG wire#powerrail
      { S7_Templates := "SrcType := Int" } EQ_Contact(in1 := "Unit1.Em5.ControlNodes".cm.brakeTest.transferPnPRightAxisZ.monitoring."step", in2 := 10)
      wire#w1
      I_Contact( "Unit1.Em5.ControlNodes".cm.brakeTest.transferPnPRightAxisZ.monitoring.brakeResult )
      Contact( "Unit1.Em5.ControlNodes".cm.brakeTest.transferPnPRightAxisZ.monitoring.brakeCompleted )
      wire#w2
      { S7_Templates := "time_type := Time" } #statTonTime[70].TON(pt := T#10s, et =>)
      Coil( "Unit1.Em5.ControlNodes".cm.brakeTest.transferPnPRightAxisZ.monitoring.error )
   END_RUNG
   RUNG wire#w1
      I_Contact( "Unit1.Em5.ControlNodes".cm.brakeTest.transferPnPRightAxisZ.monitoring.brakeSelected )
   END_RUNG wire#w2
   RUNG wire#powerrail
      { S7_Templates := "SrcType := Int" } NE_Contact(in1 := "Unit1.Em5.ControlNodes".cm.brakeTest.transferPnPRightAxisZ.monitoring."step", in2 := 10)
      Contact( "Unit1.Em5.ControlNodes".cm.brakeTest.transferPnPRightAxisZ.monitoring.busy )
   END_RUNG wire#w2
   RUNG wire#powerrail
      Contact( "Unit1.Em5.ControlNodes".cm.brakeTest.transferPnPRightAxisZ.monitoring.busy )
      wire#w3
      P_Trig( #statPulse[75] )
      S_Coil( "Unit1.Em5.Config".cmTransferPnPRightAxisZ.disableAlarms )
   END_RUNG
   RUNG wire#w3
      Not()
      P_Trig( #statPulse[76] )
      R_Coil( "Unit1.Em5.Config".cmTransferPnPRightAxisZ.disableAlarms )
   END_RUNG
   // the same network as SCL:
   #statTonTime[70].TON(IN := (("Unit1.Em5.ControlNodes".cm.brakeTest.transferPnPRightAxisZ.monitoring."step" = 10) AND ((NOT "Unit1.Em5.ControlNodes".cm.brakeTest.transferPnPRightAxisZ.monitoring.brakeResult AND "Unit1.Em5.ControlNodes".cm.brakeTest.transferPnPRightAxisZ.monitoring.brakeCompleted) OR NOT "Unit1.Em5.ControlNodes".cm.brakeTest.transferPnPRightAxisZ.monitoring.brakeSelected)) OR (("Unit1.Em5.ControlNodes".cm.brakeTest.transferPnPRightAxisZ.monitoring."step" <> 10) AND "Unit1.Em5.ControlNodes".cm.brakeTest.transferPnPRightAxisZ.monitoring.busy),
                        PT := T#10s);
   "Unit1.Em5.ControlNodes".cm.brakeTest.transferPnPRightAxisZ.monitoring.error := #statTonTime[70].Q;
   #_w1 := "Unit1.Em5.ControlNodes".cm.brakeTest.transferPnPRightAxisZ.monitoring.busy AND NOT #statPulse[75];   // rising edge
   #statPulse[75] := "Unit1.Em5.ControlNodes".cm.brakeTest.transferPnPRightAxisZ.monitoring.busy;
   IF #_w1 THEN "Unit1.Em5.Config".cmTransferPnPRightAxisZ.disableAlarms := TRUE; END_IF;
   #_w2 := NOT "Unit1.Em5.ControlNodes".cm.brakeTest.transferPnPRightAxisZ.monitoring.busy AND NOT #statPulse[76];   // rising edge
   #statPulse[76] := NOT "Unit1.Em5.ControlNodes".cm.brakeTest.transferPnPRightAxisZ.monitoring.busy;
   IF #_w2 THEN "Unit1.Em5.Config".cmTransferPnPRightAxisZ.disableAlarms := FALSE; END_IF;
END_REGION

REGION Network 201: JR Out P&P Right Z-Axis Brake Test Initialize
   RUNG wire#powerrail
      { S7_Templates := "SrcType := Int" } NE_Contact(in1 := "Unit1.Em5.ControlNodes".cm.brakeTest.transferPnPRightAxisZ.monitoring."step", in2 := 10)
      Contact( #statUnitStatus.mode.production )
      P_Trig( #statPulse[70] )
      wire#w1
      R_Coil( "Unit1.Em5.Config".cmTransferPnPRightAxisZ.disableAlarms )
      R_Coil( "Unit1.Em5.ControlNodes".cm.brakeTest.transferPnPRightAxisZ.monitoring.busy )
      R_Coil( "Unit1.Em5.ControlNodes".cm.brakeTest.transferPnPRightAxisZ.monitoring.complete )
      Move(in := 0, out1 => "Unit1.Em5.ControlNodes".cm.brakeTest.transferPnPRightAxisZ.monitoring."step")
   END_RUNG
   RUNG wire#powerrail
      P_Contact(operand := "Unit1.Em5.ControlNodes".cm.brakeTest.transferPnPRightAxisZ.monitoring.error, bit := #statPulse[72])
   END_RUNG wire#w1
   RUNG wire#powerrail
      Contact( "Unit1.EmNodes".safetyStatusZone1.allFDoorClose )
      Contact( #statUnitStatus.acknowledgeActive )
   END_RUNG wire#w1
   // the same network as SCL:
   #_w1 := ("Unit1.Em5.ControlNodes".cm.brakeTest.transferPnPRightAxisZ.monitoring."step" <> 10) AND #statUnitStatus.mode.production;
   #_w2 := #_w1 AND NOT #statPulse[70];   // rising edge
   #statPulse[70] := #_w1;
   #_w3 := "Unit1.Em5.ControlNodes".cm.brakeTest.transferPnPRightAxisZ.monitoring.error AND NOT #statPulse[72];   // rising edge of "Unit1.Em5.ControlNodes".cm.brakeTest.transferPnPRightAxisZ.monitoring.error
   #statPulse[72] := "Unit1.Em5.ControlNodes".cm.brakeTest.transferPnPRightAxisZ.monitoring.error;
   IF #_w2 OR #_w3 OR ("Unit1.EmNodes".safetyStatusZone1.allFDoorClose AND #statUnitStatus.acknowledgeActive) THEN
       "Unit1.Em5.Config".cmTransferPnPRightAxisZ.disableAlarms := FALSE;
       "Unit1.Em5.ControlNodes".cm.brakeTest.transferPnPRightAxisZ.monitoring.busy := FALSE;
       "Unit1.Em5.ControlNodes".cm.brakeTest.transferPnPRightAxisZ.monitoring.complete := FALSE;
       "Unit1.Em5.ControlNodes".cm.brakeTest.transferPnPRightAxisZ.monitoring."step" := 0;
   END_IF;
END_REGION

REGION Network 202: Transfer P&P Right Z-Axis Brake Test Ready
   RUNG wire#powerrail
      I_Contact( "Unit1.EmNodes".motionOFF.DR17 )
      Contact( #statSlmStatus.running )
      Contact( "Unit1.EmNodes".safetyStatusZone1.allFDoorClose )
      Contact( #instLDrv701ControlTransferPnPRightAxisZ.enable )
      Contact( #instLDrv701StatusTransferPnPRightAxisZ.enable )
      Coil( "Unit1.Em5.ControlNodes".cm.brakeTest.transferPnPRightAxisZ.monitoring.ready )
   END_RUNG
   // the same network as SCL:
   "Unit1.Em5.ControlNodes".cm.brakeTest.transferPnPRightAxisZ.monitoring.ready := NOT "Unit1.EmNodes".motionOFF.DR17 AND #statSlmStatus.running AND "Unit1.EmNodes".safetyStatusZone1.allFDoorClose AND #instLDrv701ControlTransferPnPRightAxisZ.enable AND #instLDrv701StatusTransferPnPRightAxisZ.enable;
END_REGION

REGION Network 203: Transfer P&P Right Z-Axis Brake Test Commands
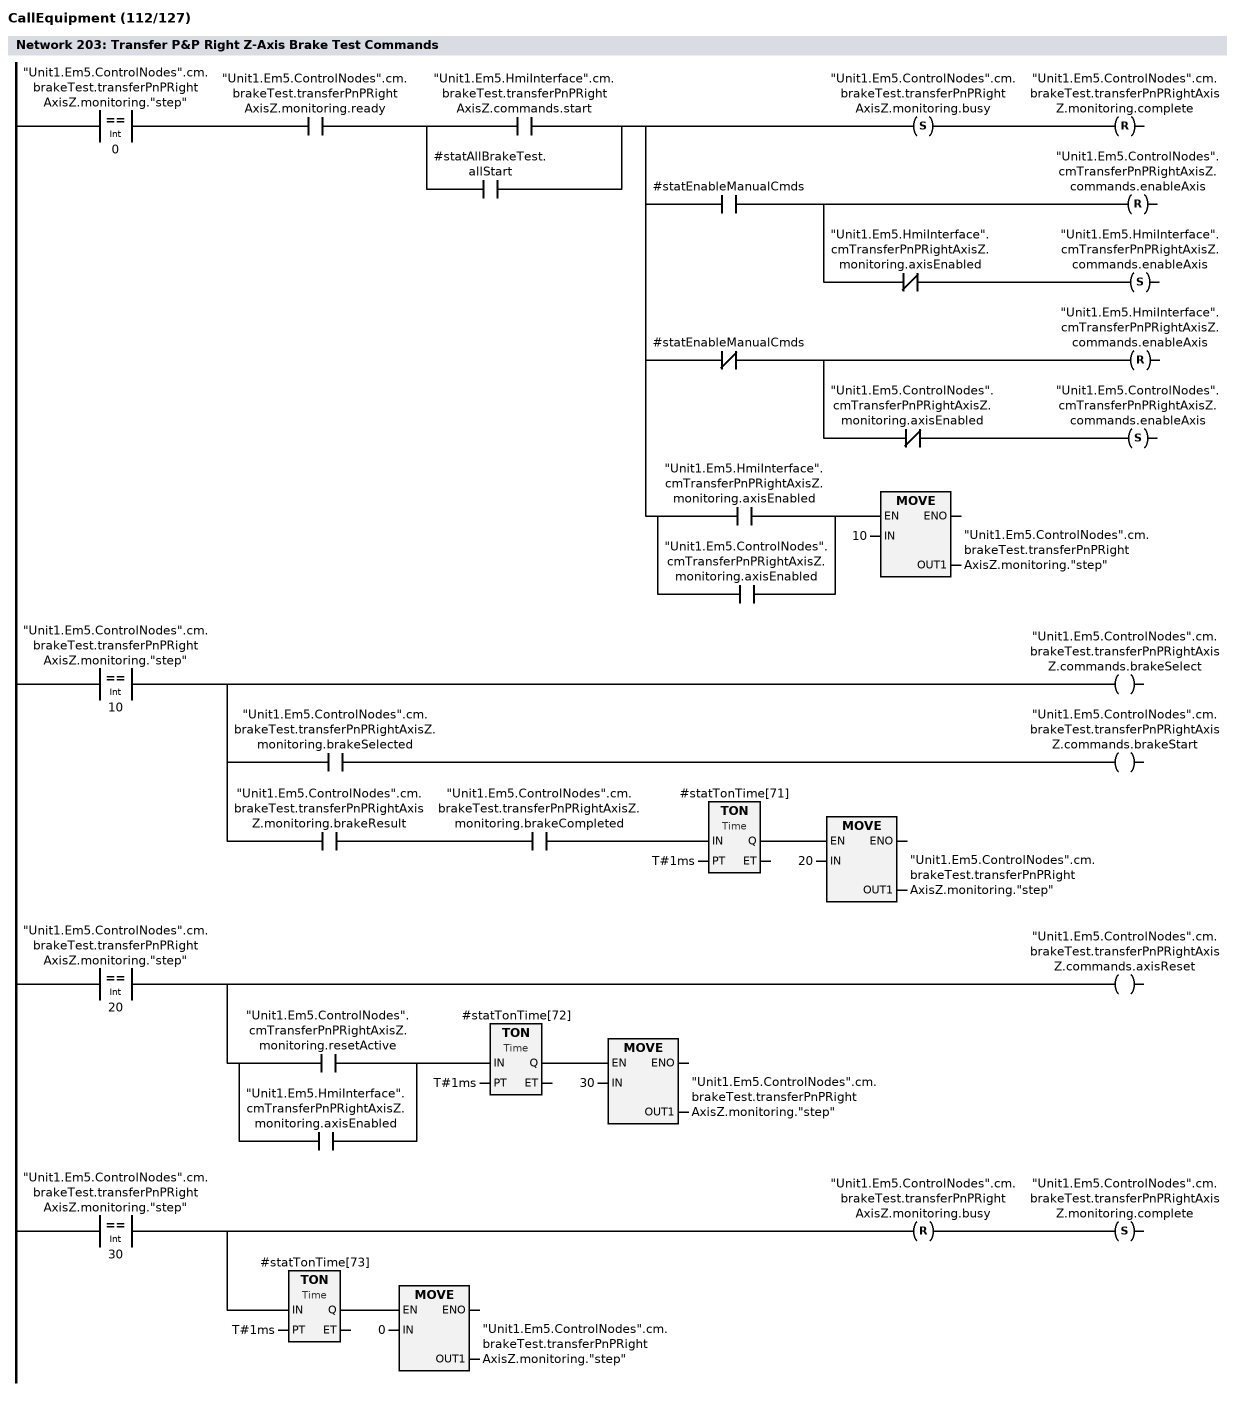
   RUNG wire#powerrail
      { S7_Templates := "SrcType := Int" } EQ_Contact(in1 := "Unit1.Em5.ControlNodes".cm.brakeTest.transferPnPRightAxisZ.monitoring."step", in2 := 0)
      Contact( "Unit1.Em5.ControlNodes".cm.brakeTest.transferPnPRightAxisZ.monitoring.ready )
      wire#w1
      Contact( "Unit1.Em5.HmiInterface".cm.brakeTest.transferPnPRightAxisZ.commands.start )
      wire#w2
      S_Coil( "Unit1.Em5.ControlNodes".cm.brakeTest.transferPnPRightAxisZ.monitoring.busy )
      R_Coil( "Unit1.Em5.ControlNodes".cm.brakeTest.transferPnPRightAxisZ.monitoring.complete )
   END_RUNG
   RUNG wire#w1
      Contact( #statAllBrakeTest.allStart )
   END_RUNG wire#w2
   RUNG wire#w2
      Contact( #statEnableManualCmds )
      wire#w3
      R_Coil( "Unit1.Em5.ControlNodes".cmTransferPnPRightAxisZ.commands.enableAxis )
   END_RUNG
   RUNG wire#w3
      I_Contact( "Unit1.Em5.HmiInterface".cmTransferPnPRightAxisZ.monitoring.axisEnabled )
      S_Coil( "Unit1.Em5.HmiInterface".cmTransferPnPRightAxisZ.commands.enableAxis )
   END_RUNG
   RUNG wire#w2
      I_Contact( #statEnableManualCmds )
      wire#w4
      R_Coil( "Unit1.Em5.HmiInterface".cmTransferPnPRightAxisZ.commands.enableAxis )
   END_RUNG
   RUNG wire#w4
      I_Contact( "Unit1.Em5.ControlNodes".cmTransferPnPRightAxisZ.monitoring.axisEnabled )
      S_Coil( "Unit1.Em5.ControlNodes".cmTransferPnPRightAxisZ.commands.enableAxis )
   END_RUNG
   RUNG wire#w2
      Contact( "Unit1.Em5.HmiInterface".cmTransferPnPRightAxisZ.monitoring.axisEnabled )
      wire#w5
      Move(in := 10, out1 => "Unit1.Em5.ControlNodes".cm.brakeTest.transferPnPRightAxisZ.monitoring."step")
   END_RUNG
   RUNG wire#w2
      Contact( "Unit1.Em5.ControlNodes".cmTransferPnPRightAxisZ.monitoring.axisEnabled )
   END_RUNG wire#w5
   RUNG wire#powerrail
      { S7_Templates := "SrcType := Int" } EQ_Contact(in1 := "Unit1.Em5.ControlNodes".cm.brakeTest.transferPnPRightAxisZ.monitoring."step", in2 := 10)
      wire#w6
      Coil( "Unit1.Em5.ControlNodes".cm.brakeTest.transferPnPRightAxisZ.commands.brakeSelect )
   END_RUNG
   RUNG wire#w6
      Contact( "Unit1.Em5.ControlNodes".cm.brakeTest.transferPnPRightAxisZ.monitoring.brakeSelected )
      Coil( "Unit1.Em5.ControlNodes".cm.brakeTest.transferPnPRightAxisZ.commands.brakeStart )
   END_RUNG
   RUNG wire#w6
      Contact( "Unit1.Em5.ControlNodes".cm.brakeTest.transferPnPRightAxisZ.monitoring.brakeResult )
      Contact( "Unit1.Em5.ControlNodes".cm.brakeTest.transferPnPRightAxisZ.monitoring.brakeCompleted )
      { S7_Templates := "time_type := Time" } #statTonTime[71].TON(pt := T#1ms, et =>)
      Move(in := 20, out1 => "Unit1.Em5.ControlNodes".cm.brakeTest.transferPnPRightAxisZ.monitoring."step")
   END_RUNG
   RUNG wire#powerrail
      { S7_Templates := "SrcType := Int" } EQ_Contact(in1 := "Unit1.Em5.ControlNodes".cm.brakeTest.transferPnPRightAxisZ.monitoring."step", in2 := 20)
      wire#w7
      Coil( "Unit1.Em5.ControlNodes".cm.brakeTest.transferPnPRightAxisZ.commands.axisReset )
   END_RUNG
   RUNG wire#w7
      Contact( "Unit1.Em5.ControlNodes".cmTransferPnPRightAxisZ.monitoring.resetActive )
      wire#w8
      { S7_Templates := "time_type := Time" } #statTonTime[72].TON(pt := T#1ms, et =>)
      Move(in := 30, out1 => "Unit1.Em5.ControlNodes".cm.brakeTest.transferPnPRightAxisZ.monitoring."step")
   END_RUNG
   RUNG wire#w7
      Contact( "Unit1.Em5.HmiInterface".cmTransferPnPRightAxisZ.monitoring.axisEnabled )
   END_RUNG wire#w8
   RUNG wire#powerrail
      { S7_Templates := "SrcType := Int" } EQ_Contact(in1 := "Unit1.Em5.ControlNodes".cm.brakeTest.transferPnPRightAxisZ.monitoring."step", in2 := 30)
      wire#w9
      R_Coil( "Unit1.Em5.ControlNodes".cm.brakeTest.transferPnPRightAxisZ.monitoring.busy )
      S_Coil( "Unit1.Em5.ControlNodes".cm.brakeTest.transferPnPRightAxisZ.monitoring.complete )
   END_RUNG
   RUNG wire#w9
      { S7_Templates := "time_type := Time" } #statTonTime[73].TON(pt := T#1ms, et =>)
      Move(in := 0, out1 => "Unit1.Em5.ControlNodes".cm.brakeTest.transferPnPRightAxisZ.monitoring."step")
   END_RUNG
   // the same network as SCL:
   #_w1 := ("Unit1.Em5.ControlNodes".cm.brakeTest.transferPnPRightAxisZ.monitoring."step" = 0) AND "Unit1.Em5.ControlNodes".cm.brakeTest.transferPnPRightAxisZ.monitoring.ready AND ("Unit1.Em5.HmiInterface".cm.brakeTest.transferPnPRightAxisZ.commands.start OR #statAllBrakeTest.allStart);
   IF #_w1 THEN
       "Unit1.Em5.ControlNodes".cm.brakeTest.transferPnPRightAxisZ.monitoring.busy := TRUE;
       "Unit1.Em5.ControlNodes".cm.brakeTest.transferPnPRightAxisZ.monitoring.complete := FALSE;
   END_IF;
   #_w2 := #_w1 AND #statEnableManualCmds;
   IF #_w2 THEN "Unit1.Em5.ControlNodes".cmTransferPnPRightAxisZ.commands.enableAxis := FALSE; END_IF;
   IF #_w2 AND NOT "Unit1.Em5.HmiInterface".cmTransferPnPRightAxisZ.monitoring.axisEnabled THEN
       "Unit1.Em5.HmiInterface".cmTransferPnPRightAxisZ.commands.enableAxis := TRUE;
   END_IF;
   #_w3 := #_w1 AND NOT #statEnableManualCmds;
   IF #_w3 THEN "Unit1.Em5.HmiInterface".cmTransferPnPRightAxisZ.commands.enableAxis := FALSE; END_IF;
   IF #_w3 AND NOT "Unit1.Em5.ControlNodes".cmTransferPnPRightAxisZ.monitoring.axisEnabled THEN
       "Unit1.Em5.ControlNodes".cmTransferPnPRightAxisZ.commands.enableAxis := TRUE;
   END_IF;
   IF #_w1 AND ("Unit1.Em5.HmiInterface".cmTransferPnPRightAxisZ.monitoring.axisEnabled OR "Unit1.Em5.ControlNodes".cmTransferPnPRightAxisZ.monitoring.axisEnabled) THEN
       "Unit1.Em5.ControlNodes".cm.brakeTest.transferPnPRightAxisZ.monitoring."step" := 10;
   END_IF;
   "Unit1.Em5.ControlNodes".cm.brakeTest.transferPnPRightAxisZ.commands.brakeSelect := "Unit1.Em5.ControlNodes".cm.brakeTest.transferPnPRightAxisZ.monitoring."step" = 10;
   "Unit1.Em5.ControlNodes".cm.brakeTest.transferPnPRightAxisZ.commands.brakeStart := "Unit1.Em5.ControlNodes".cm.brakeTest.transferPnPRightAxisZ.commands.brakeSelect AND "Unit1.Em5.ControlNodes".cm.brakeTest.transferPnPRightAxisZ.monitoring.brakeSelected;
   #statTonTime[71].TON(IN := "Unit1.Em5.ControlNodes".cm.brakeTest.transferPnPRightAxisZ.commands.brakeSelect AND "Unit1.Em5.ControlNodes".cm.brakeTest.transferPnPRightAxisZ.monitoring.brakeResult AND "Unit1.Em5.ControlNodes".cm.brakeTest.transferPnPRightAxisZ.monitoring.brakeCompleted,
                        PT := T#1ms);
   IF #statTonTime[71].Q THEN
       "Unit1.Em5.ControlNodes".cm.brakeTest.transferPnPRightAxisZ.monitoring."step" := 20;
   END_IF;
   "Unit1.Em5.ControlNodes".cm.brakeTest.transferPnPRightAxisZ.commands.axisReset := "Unit1.Em5.ControlNodes".cm.brakeTest.transferPnPRightAxisZ.monitoring."step" = 20;
   #statTonTime[72].TON(IN := "Unit1.Em5.ControlNodes".cm.brakeTest.transferPnPRightAxisZ.commands.axisReset AND ("Unit1.Em5.ControlNodes".cmTransferPnPRightAxisZ.monitoring.resetActive OR "Unit1.Em5.HmiInterface".cmTransferPnPRightAxisZ.monitoring.axisEnabled),
                        PT := T#1ms);
   IF #statTonTime[72].Q THEN
       "Unit1.Em5.ControlNodes".cm.brakeTest.transferPnPRightAxisZ.monitoring."step" := 30;
   END_IF;
   #_w4 := "Unit1.Em5.ControlNodes".cm.brakeTest.transferPnPRightAxisZ.monitoring."step" = 30;
   IF #_w4 THEN
       "Unit1.Em5.ControlNodes".cm.brakeTest.transferPnPRightAxisZ.monitoring.busy := FALSE;
       "Unit1.Em5.ControlNodes".cm.brakeTest.transferPnPRightAxisZ.monitoring.complete := TRUE;
   END_IF;
   #statTonTime[73].TON(IN := #_w4, PT := T#1ms);
   IF #statTonTime[73].Q THEN
       "Unit1.Em5.ControlNodes".cm.brakeTest.transferPnPRightAxisZ.monitoring."step" := 0;
   END_IF;
END_REGION

REGION Network 204: Transfer P&P Right Z-Axis Brake Test Monitoring
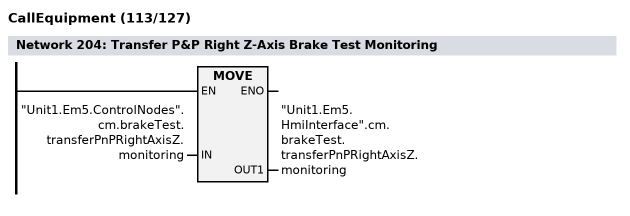
   RUNG wire#powerrail
      Move(in := "Unit1.Em5.ControlNodes".cm.brakeTest.transferPnPRightAxisZ.monitoring, out1 => "Unit1.Em5.HmiInterface".cm.brakeTest.transferPnPRightAxisZ.monitoring)
   END_RUNG
   // the same network as SCL:
   "Unit1.Em5.HmiInterface".cm.brakeTest.transferPnPRightAxisZ.monitoring := "Unit1.Em5.ControlNodes".cm.brakeTest.transferPnPRightAxisZ.monitoring;
END_REGION

REGION Network 205: Call Transfer P&P Right Z-Axis Telegram 701
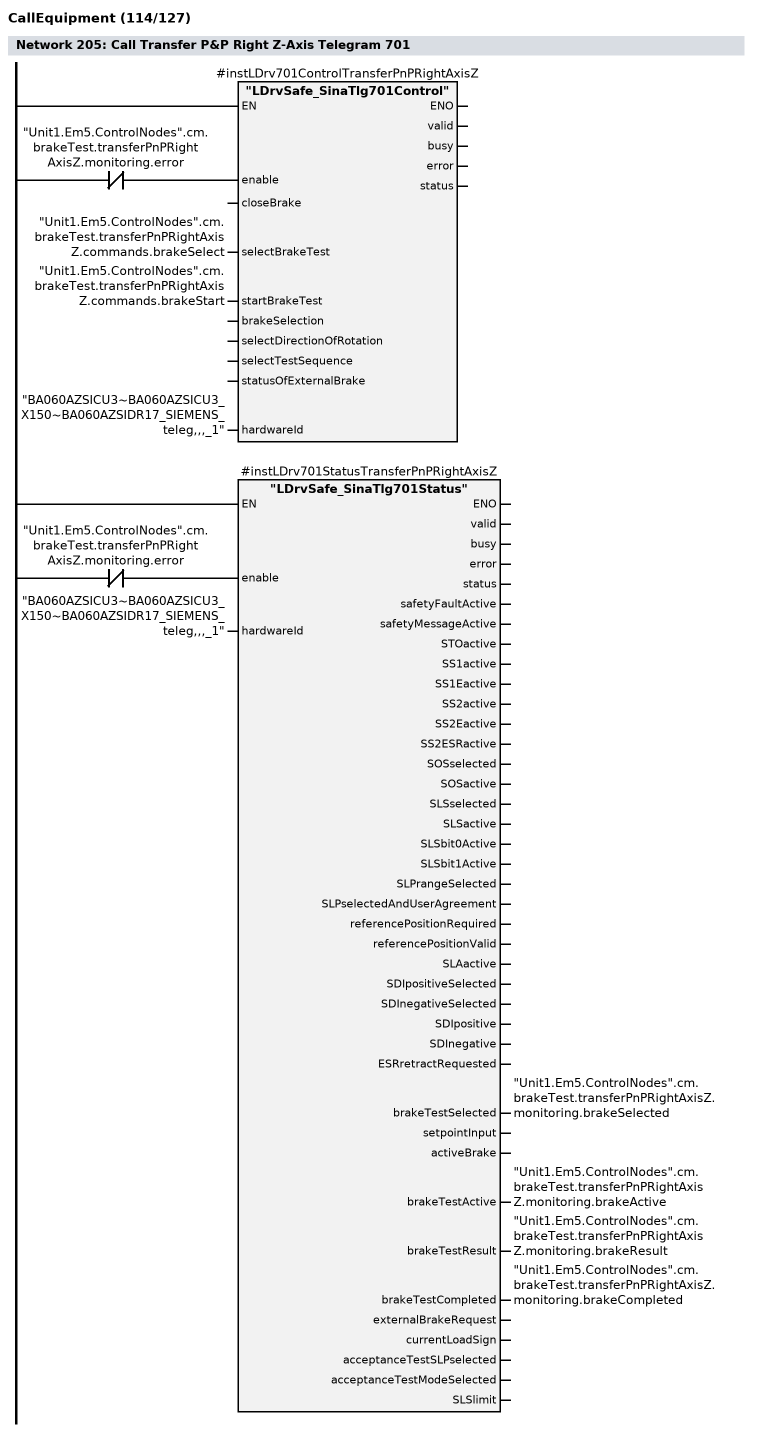
   RUNG wire#powerrail
      #instLDrv701ControlTransferPnPRightAxisZ(enable := wire#w1, closeBrake :=, selectBrakeTest := "Unit1.Em5.ControlNodes".cm.brakeTest.transferPnPRightAxisZ.commands.brakeSelect, startBrakeTest := "Unit1.Em5.ControlNodes".cm.brakeTest.transferPnPRightAxisZ.commands.brakeStart, brakeSelection :=, selectDirectionOfRotation :=, selectTestSequence :=, statusOfExternalBrake :=, hardwareId := "BA060AZSICU3~BA060AZSICU3_X150~BA060AZSIDR17_SIEMENS_teleg,,,_1", valid =>, busy =>, error =>, status =>)
   END_RUNG
   RUNG wire#powerrail
      I_Contact( "Unit1.Em5.ControlNodes".cm.brakeTest.transferPnPRightAxisZ.monitoring.error )
   END_RUNG wire#w1
   RUNG wire#powerrail
      #instLDrv701StatusTransferPnPRightAxisZ(enable := wire#w2, hardwareId := "BA060AZSICU3~BA060AZSICU3_X150~BA060AZSIDR17_SIEMENS_teleg,,,_1", valid =>, busy =>, error =>, status =>, safetyFaultActive =>, safetyMessageActive =>, STOactive =>, SS1active =>, SS1Eactive =>, SS2active =>, SS2Eactive =>, SS2ESRactive =>, SOSselected =>, SOSactive =>, SLSselected =>, SLSactive =>, SLSbit0Active =>, SLSbit1Active =>, SLPrangeSelected =>, SLPselectedAndUserAgreement =>, referencePositionRequired =>, referencePositionValid =>, SLAactive =>, SDIpositiveSelected =>, SDInegativeSelected =>, SDIpositive =>, SDInegative =>, ESRretractRequested =>, brakeTestSelected => "Unit1.Em5.ControlNodes".cm.brakeTest.transferPnPRightAxisZ.monitoring.brakeSelected, setpointInput =>, activeBrake =>, brakeTestActive => "Unit1.Em5.ControlNodes".cm.brakeTest.transferPnPRightAxisZ.monitoring.brakeActive, brakeTestResult => "Unit1.Em5.ControlNodes".cm.brakeTest.transferPnPRightAxisZ.monitoring.brakeResult, brakeTestCompleted => "Unit1.Em5.ControlNodes".cm.brakeTest.transferPnPRightAxisZ.monitoring.brakeCompleted, externalBrakeRequest =>, currentLoadSign =>, acceptanceTestSLPselected =>, acceptanceTestModeSelected =>, SLSlimit =>)
   END_RUNG
   RUNG wire#powerrail
      I_Contact( "Unit1.Em5.ControlNodes".cm.brakeTest.transferPnPRightAxisZ.monitoring.error )
   END_RUNG wire#w2
   // the same network as SCL:
   #instLDrv701ControlTransferPnPRightAxisZ(enable := NOT "Unit1.Em5.ControlNodes".cm.brakeTest.transferPnPRightAxisZ.monitoring.error,   // "LDrvSafe_SinaTlg701Control"
                           selectBrakeTest := "Unit1.Em5.ControlNodes".cm.brakeTest.transferPnPRightAxisZ.commands.brakeSelect,
                           startBrakeTest := "Unit1.Em5.ControlNodes".cm.brakeTest.transferPnPRightAxisZ.commands.brakeStart,
                           hardwareId := "BA060AZSICU3~BA060AZSICU3_X150~BA060AZSIDR17_SIEMENS_teleg,,,_1");
   #instLDrv701StatusTransferPnPRightAxisZ(enable := NOT "Unit1.Em5.ControlNodes".cm.brakeTest.transferPnPRightAxisZ.monitoring.error,   // "LDrvSafe_SinaTlg701Status"
                           hardwareId := "BA060AZSICU3~BA060AZSICU3_X150~BA060AZSIDR17_SIEMENS_teleg,,,_1",
                           brakeTestSelected => "Unit1.Em5.ControlNodes".cm.brakeTest.transferPnPRightAxisZ.monitoring.brakeSelected,
                           brakeTestActive => "Unit1.Em5.ControlNodes".cm.brakeTest.transferPnPRightAxisZ.monitoring.brakeActive,
                           brakeTestResult => "Unit1.Em5.ControlNodes".cm.brakeTest.transferPnPRightAxisZ.monitoring.brakeResult,
                           brakeTestCompleted => "Unit1.Em5.ControlNodes".cm.brakeTest.transferPnPRightAxisZ.monitoring.brakeCompleted);
END_REGION

REGION Network 207: ******************** Control Modules (TwoWayActuator) ********************
END_REGION

REGION Network 208: Reset CMS
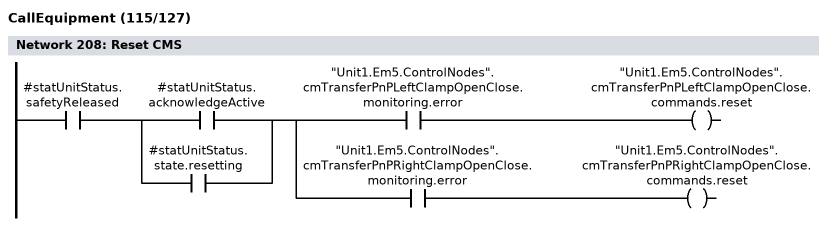
   RUNG wire#powerrail
      Contact( #statUnitStatus.safetyReleased )
      wire#w1
      Contact( #statUnitStatus.acknowledgeActive )
      wire#w2
      Contact( "Unit1.Em5.ControlNodes".cmTransferPnPLeftClampOpenClose.monitoring.error )
      Coil( "Unit1.Em5.ControlNodes".cmTransferPnPLeftClampOpenClose.commands.reset )
   END_RUNG
   RUNG wire#w1
      Contact( #statUnitStatus.state.resetting )
   END_RUNG wire#w2
   RUNG wire#w2
      Contact( "Unit1.Em5.ControlNodes".cmTransferPnPRightClampOpenClose.monitoring.error )
      Coil( "Unit1.Em5.ControlNodes".cmTransferPnPRightClampOpenClose.commands.reset )
   END_RUNG
   // the same network as SCL:
   #_w1 := #statUnitStatus.safetyReleased AND (#statUnitStatus.acknowledgeActive OR #statUnitStatus.state.resetting);
   "Unit1.Em5.ControlNodes".cmTransferPnPLeftClampOpenClose.commands.reset := #_w1 AND "Unit1.Em5.ControlNodes".cmTransferPnPLeftClampOpenClose.monitoring.error;
   "Unit1.Em5.ControlNodes".cmTransferPnPRightClampOpenClose.commands.reset := #_w1 AND "Unit1.Em5.ControlNodes".cmTransferPnPRightClampOpenClose.monitoring.error;
END_REGION

REGION Network 210: Transfer P&P Left Clamp HOME
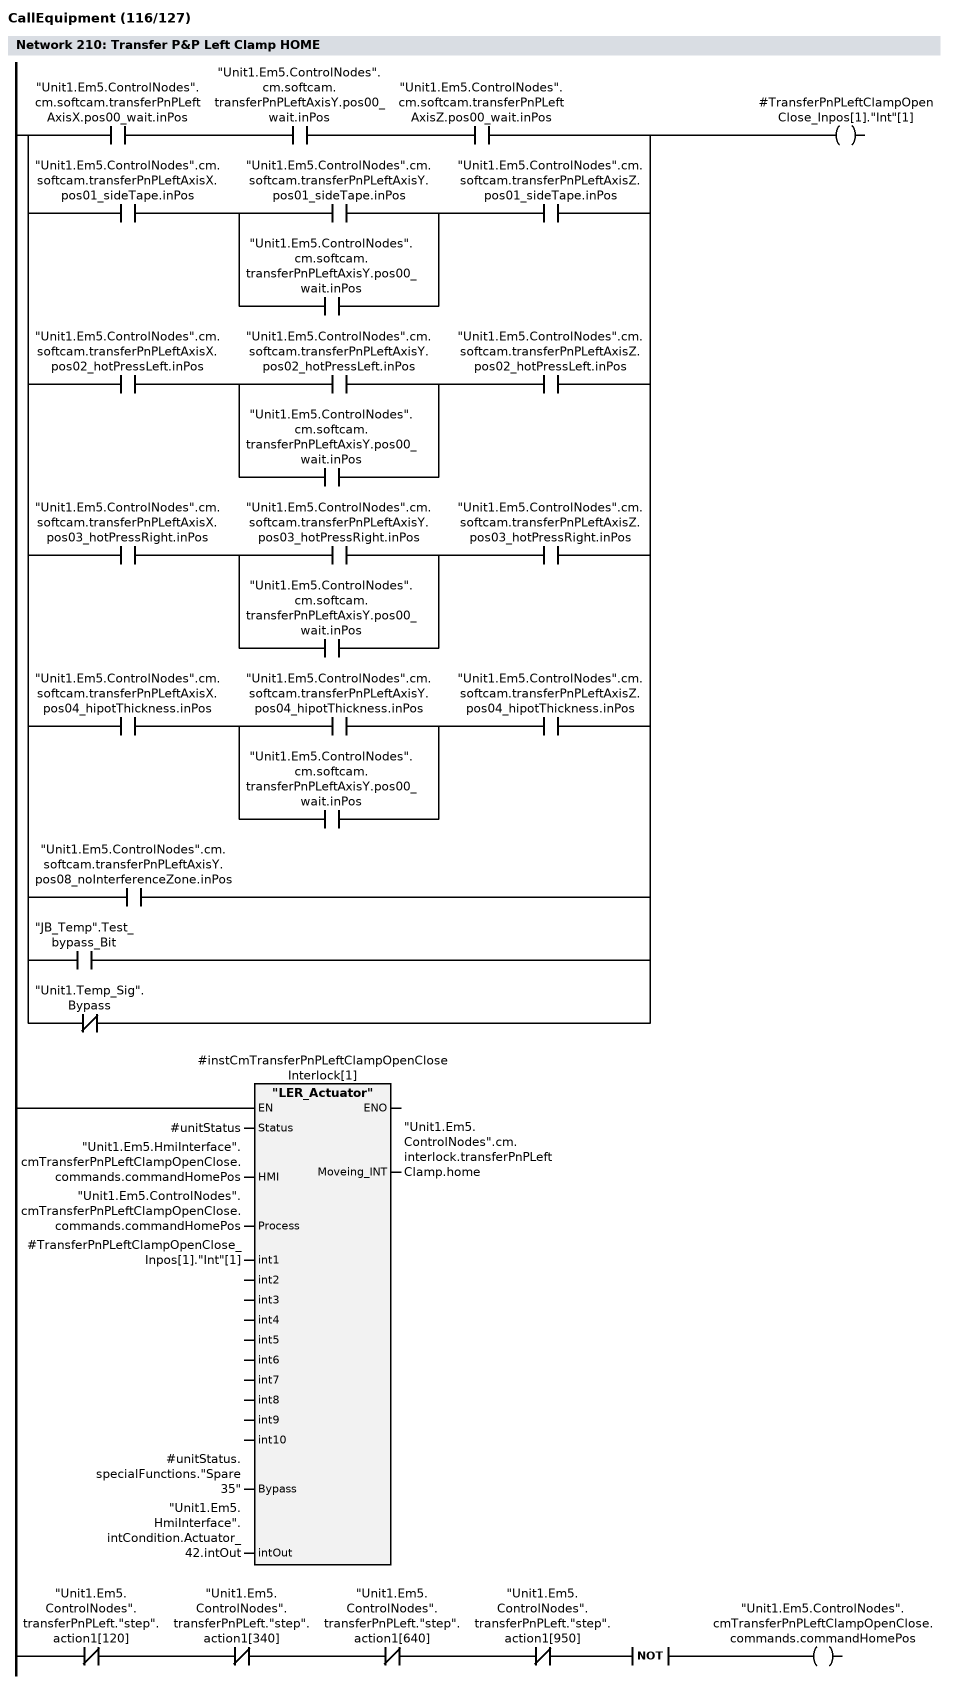
   RUNG wire#powerrail
      Contact( "Unit1.Em5.ControlNodes".cm.softcam.transferPnPLeftAxisX.pos00_wait.inPos )
      Contact( "Unit1.Em5.ControlNodes".cm.softcam.transferPnPLeftAxisY.pos00_wait.inPos )
      Contact( "Unit1.Em5.ControlNodes".cm.softcam.transferPnPLeftAxisZ.pos00_wait.inPos )
      wire#w1
      Coil( #TransferPnPLeftClampOpenClose_Inpos[1]."Int"[1] )
   END_RUNG
   RUNG wire#powerrail
      Contact( "Unit1.Em5.ControlNodes".cm.softcam.transferPnPLeftAxisX.pos01_sideTape.inPos )
      wire#w2
      Contact( "Unit1.Em5.ControlNodes".cm.softcam.transferPnPLeftAxisY.pos01_sideTape.inPos )
      wire#w3
      Contact( "Unit1.Em5.ControlNodes".cm.softcam.transferPnPLeftAxisZ.pos01_sideTape.inPos )
   END_RUNG wire#w1
   RUNG wire#w2
      Contact( "Unit1.Em5.ControlNodes".cm.softcam.transferPnPLeftAxisY.pos00_wait.inPos )
   END_RUNG wire#w3
   RUNG wire#powerrail
      Contact( "Unit1.Em5.ControlNodes".cm.softcam.transferPnPLeftAxisX.pos02_hotPressLeft.inPos )
      wire#w4
      Contact( "Unit1.Em5.ControlNodes".cm.softcam.transferPnPLeftAxisY.pos02_hotPressLeft.inPos )
      wire#w5
      Contact( "Unit1.Em5.ControlNodes".cm.softcam.transferPnPLeftAxisZ.pos02_hotPressLeft.inPos )
   END_RUNG wire#w1
   RUNG wire#w4
      Contact( "Unit1.Em5.ControlNodes".cm.softcam.transferPnPLeftAxisY.pos00_wait.inPos )
   END_RUNG wire#w5
   RUNG wire#powerrail
      Contact( "Unit1.Em5.ControlNodes".cm.softcam.transferPnPLeftAxisX.pos03_hotPressRight.inPos )
      wire#w6
      Contact( "Unit1.Em5.ControlNodes".cm.softcam.transferPnPLeftAxisY.pos03_hotPressRight.inPos )
      wire#w7
      Contact( "Unit1.Em5.ControlNodes".cm.softcam.transferPnPLeftAxisZ.pos03_hotPressRight.inPos )
   END_RUNG wire#w1
   RUNG wire#w6
      Contact( "Unit1.Em5.ControlNodes".cm.softcam.transferPnPLeftAxisY.pos00_wait.inPos )
   END_RUNG wire#w7
   RUNG wire#powerrail
      Contact( "Unit1.Em5.ControlNodes".cm.softcam.transferPnPLeftAxisX.pos04_hipotThickness.inPos )
      wire#w8
      Contact( "Unit1.Em5.ControlNodes".cm.softcam.transferPnPLeftAxisY.pos04_hipotThickness.inPos )
      wire#w9
      Contact( "Unit1.Em5.ControlNodes".cm.softcam.transferPnPLeftAxisZ.pos04_hipotThickness.inPos )
   END_RUNG wire#w1
   RUNG wire#w8
      Contact( "Unit1.Em5.ControlNodes".cm.softcam.transferPnPLeftAxisY.pos00_wait.inPos )
   END_RUNG wire#w9
   RUNG wire#powerrail
      Contact( "Unit1.Em5.ControlNodes".cm.softcam.transferPnPLeftAxisY.pos08_noInterferenceZone.inPos )
   END_RUNG wire#w1
   RUNG wire#powerrail
      Contact( "JB_Temp".Test_bypass_Bit )
   END_RUNG wire#w1
   RUNG wire#powerrail
      I_Contact( "Unit1.Temp_Sig".Bypass )
   END_RUNG wire#w1
   RUNG wire#powerrail
      #instCmTransferPnPLeftClampOpenCloseInterlock[1](Status := #unitStatus, HMI := "Unit1.Em5.HmiInterface".cmTransferPnPLeftClampOpenClose.commands.commandHomePos, Process := "Unit1.Em5.ControlNodes".cmTransferPnPLeftClampOpenClose.commands.commandHomePos, int1 := #TransferPnPLeftClampOpenClose_Inpos[1]."Int"[1], int2 :=, int3 :=, int4 :=, int5 :=, int6 :=, int7 :=, int8 :=, int9 :=, int10 :=, Bypass := #unitStatus.specialFunctions."Spare 35", intOut := "Unit1.Em5.HmiInterface".intCondition.Actuator_42.intOut, Moveing_INT => "Unit1.Em5.ControlNodes".cm.interlock.transferPnPLeftClamp.home)
   END_RUNG
   RUNG wire#powerrail
      I_Contact( "Unit1.Em5.ControlNodes".transferPnPLeft."step".action1[120] )
      I_Contact( "Unit1.Em5.ControlNodes".transferPnPLeft."step".action1[340] )
      I_Contact( "Unit1.Em5.ControlNodes".transferPnPLeft."step".action1[640] )
      I_Contact( "Unit1.Em5.ControlNodes".transferPnPLeft."step".action1[950] )
      Not()
      Coil( "Unit1.Em5.ControlNodes".cmTransferPnPLeftClampOpenClose.commands.commandHomePos )
   END_RUNG
   // the same network as SCL:
   #TransferPnPLeftClampOpenClose_Inpos[1]."Int"[1] := ("Unit1.Em5.ControlNodes".cm.softcam.transferPnPLeftAxisX.pos00_wait.inPos AND "Unit1.Em5.ControlNodes".cm.softcam.transferPnPLeftAxisY.pos00_wait.inPos AND "Unit1.Em5.ControlNodes".cm.softcam.transferPnPLeftAxisZ.pos00_wait.inPos) OR ("Unit1.Em5.ControlNodes".cm.softcam.transferPnPLeftAxisX.pos01_sideTape.inPos AND ("Unit1.Em5.ControlNodes".cm.softcam.transferPnPLeftAxisY.pos01_sideTape.inPos OR "Unit1.Em5.ControlNodes".cm.softcam.transferPnPLeftAxisY.pos00_wait.inPos) AND "Unit1.Em5.ControlNodes".cm.softcam.transferPnPLeftAxisZ.pos01_sideTape.inPos) OR ("Unit1.Em5.ControlNodes".cm.softcam.transferPnPLeftAxisX.pos02_hotPressLeft.inPos AND ("Unit1.Em5.ControlNodes".cm.softcam.transferPnPLeftAxisY.pos02_hotPressLeft.inPos OR "Unit1.Em5.ControlNodes".cm.softcam.transferPnPLeftAxisY.pos00_wait.inPos) AND "Unit1.Em5.ControlNodes".cm.softcam.transferPnPLeftAxisZ.pos02_hotPressLeft.inPos) OR ("Unit1.Em5.ControlNodes".cm.softcam.transferPnPLeftAxisX.pos03_hotPressRight.inPos AND ("Unit1.Em5.ControlNodes".cm.softcam.transferPnPLeftAxisY.pos03_hotPressRight.inPos OR "Unit1.Em5.ControlNodes".cm.softcam.transferPnPLeftAxisY.pos00_wait.inPos) AND "Unit1.Em5.ControlNodes".cm.softcam.transferPnPLeftAxisZ.pos03_hotPressRight.inPos) OR ("Unit1.Em5.ControlNodes".cm.softcam.transferPnPLeftAxisX.pos04_hipotThickness.inPos AND ("Unit1.Em5.ControlNodes".cm.softcam.transferPnPLeftAxisY.pos04_hipotThickness.inPos OR "Unit1.Em5.ControlNodes".cm.softcam.transferPnPLeftAxisY.pos00_wait.inPos) AND "Unit1.Em5.ControlNodes".cm.softcam.transferPnPLeftAxisZ.pos04_hipotThickness.inPos) OR "Unit1.Em5.ControlNodes".cm.softcam.transferPnPLeftAxisY.pos08_noInterferenceZone.inPos OR "JB_Temp".Test_bypass_Bit OR NOT "Unit1.Temp_Sig".Bypass;
   #instCmTransferPnPLeftClampOpenCloseInterlock[1](Status := #unitStatus,   // "LER_Actuator"
                           HMI := "Unit1.Em5.HmiInterface".cmTransferPnPLeftClampOpenClose.commands.commandHomePos,
                           Process := "Unit1.Em5.ControlNodes".cmTransferPnPLeftClampOpenClose.commands.commandHomePos,
                           int1 := #TransferPnPLeftClampOpenClose_Inpos[1]."Int"[1],
                           Bypass := #unitStatus.specialFunctions."Spare 35",
                           intOut := "Unit1.Em5.HmiInterface".intCondition.Actuator_42.intOut,
                           Moveing_INT => "Unit1.Em5.ControlNodes".cm.interlock.transferPnPLeftClamp.home);
   "Unit1.Em5.ControlNodes".cmTransferPnPLeftClampOpenClose.commands.commandHomePos := NOT (NOT "Unit1.Em5.ControlNodes".transferPnPLeft."step".action1[120] AND NOT "Unit1.Em5.ControlNodes".transferPnPLeft."step".action1[340] AND NOT "Unit1.Em5.ControlNodes".transferPnPLeft."step".action1[640] AND NOT "Unit1.Em5.ControlNodes".transferPnPLeft."step".action1[950]);
END_REGION

